# B&R Automation Studio project TD52 (part 84)

### Modul_EngCtr.typ - Package data types
```iecst
(********************************************************************
 * COPYRIGHT -- INNIO Company
 ********************************************************************
 * Package: Opstate_Pkg
 * File: module_Opstate.typ
 * Author: Mario Graus
 * Created: October 19, 2011
 ********************************************************************
 * Data types of package Opstate_Pkg
 ********************************************************************)

TYPE
	IN_EngCtr_Struct : 	STRUCT
		iSt_OpMode : UDINT; (* engine operation mode *) (*OldName: new PV; Cycle:2; *)
		rN_Set_Norm : REAL; (* speed setpoint speed controller related to rN_Nom *) (*OldName: n_soll; Cycle:2;*)
		rN_Set_Norm_TC5 : REAL; (* speed setpoint speed controller related to rN_Nom *) (*OldName: n_soll; Cycle:5;*)
		rP_Act_Norm : REAL; (* actual power related to rP_Nom *) (* OldName: ssPowerEx ; Cycle:2; *)
		rP_Act_Norm_TC5 : REAL; (* actual power related to rP_Nom *) (* OldName: ssPowerEx ; Cycle:5; *)
		bDSyLine : BOOL; (* demand synchline *) (* OldName: M_SYL ; Cycle:2; *)
		bSynchDem : BOOL; (* synchronization demanded *) (* OldName: SynchAnf ; Cycle:2; *)
		rP_Set_Norm : REAL; (* power setpoint related to rP_Nom *) (* OldName: new PV; Cycle:2; *)
		rP_Set_Norm_TC5 : REAL; (* power setpoint related to rP_Nom *) (* OldName: new PV; Cycle:5; *)
		rNOxS_Eng_NOx_Act : REAL; (* actual NOx [ppm] *) (* OldName: usNOx ; Cycle:2; *)
		rNOxS_Eng_Act : REAL; (* actual NOx@x%O2 [mg] *) (* OldName: usNOx_mg ; Cycle:2; *)
		bKLS98_MSF : ARRAY[0..24]OF BOOL; (* knocking sensor measuring signal failure *) (* OldName: bKLS98Fault; Cycle:2; *)
		rKno_IP_Red : REAL; (* timing reduction by knocking *) (* OldName: klreg_dz; Cycle:2; *)
		rCA_Knck_Red : ARRAY[0..24]OF REAL; (* cylinder timing reduction by knocking *) (* OldName: ssKlRegdZZP; Cycle:2; *)
		iIdx_Cyl_Knck_Max : INT; (* cylinder with highest knock signal *) (* OldName: ucKlopfMxZyl; Cycle:2; *)
		rKnck_Intgr : ARRAY[0..24]OF REAL; (* integrated cylinder knock values *) (* OldName: IntKlopf; Cycle:2; *)
		rP_Act_Norm_Filt : REAL; (* actual power related to rP_Nom filtered T=1s  *) (* OldName: PN_GASART; Cycle:2; *)
		rP_Act_Norm_Filt_TC5 : REAL; (* actual power related to rP_Nom filtered T=1s  *) (* OldName: PN_GASART; Cycle:5; *)
		tAB2EC : AmmBase2MM; (* 0 *) (* OldName: new PV; Cycle:2; *)
		tAB2EC_TC5 : AmmBase2MM; (* 0 *) (* OldName: new PV; Cycle:5; *)
		bIgn_Dem : BOOL; (* demand ignition *) (* OldName: ZUEND; Cycle:5; *)
		bIgn_Run : BOOL; (* Ignition system running *) (* OldName: ZIB; Cycle:2; *)
		tOMSS_MAT : HALioDo_Type; (* operation mode selector switch - MANUAL/AUTO/TEST *) (* OldName: BWS_HA; Cycle:2; *)
		rN_IgnIC_Act : REAL; (* Engine speed measured by ignition IC *) (* OldName: ZDGSpeed; Cycle:1; *)
		rN_IgnSAFI_Act : REAL; (* Engine speed measured by ignition SAFI *) (* OldName: ZDGSpeed; Cycle:2; *)
		rT_EG_Cyl : ARRAY[0..24]OF REAL; (* cylinder exhaust gas temperatures *) (* OldName: t_zyl; Cycle:5; *)
		bEng_Dem_Bloc : BOOL; (* blocking release of engine *) (* OldName: ANFBLO; Cycle:2; *)
		tPB2MM : ParaBase2MM_type; (* Messages from parametercheck module parameter are OK *) (* OldName: new PV; Cycle:5; *)
		rP_Nom : REAL; (* nominal electric power [kW], depends on gastype *) (* OldName: PN_GASART; Cycle:2; *)
		rP_Nom_TC6 : REAL; (* nominal electric power [kW], depends on gastype *) (* OldName: PN_GASART; Cycle:6; *)
		rKno_T2s_Red : REAL; (* mixture temp. red. by knocking *) (* OldName: klreg_dt2 ; Cycle:2; *)
		iIdx_Gtyp_Dem : INT; (* actual gassort 1..4 *) (* OldName: gasart; Cycle:2; *)
		iIdx_Gtyp_Dem_TC5 : INT; (* actual gassort 1..4 *) (* OldName: gasart; Cycle:5; *)
		bGasMixingActive : BOOL; (*Gas mixing active for Tecjets *) (* OldName: 	bCrossOver	; Cyclic: ; *)
		tP_Act : ARRAY[0..2]OF HALioAi_Type; (* actual electric power [kW] *) (* OldName: P_IST_OF; Cycle:2; *)
		tSafetyLoop_Eng : HALioDi_Type; (* DI: Safety loop engine *) (* OldName: RUHE; Cycle:5; *)
		tActuator_Ok : HALioDi_Type; (* DI: Actuator okay *) (* OldName: ST_ACT; Cycle:2; *)
		tActuator_Ok_TV1A : HALioDi_Type; (* DI: Actuator okay throttle valve 1A *) (* OldName: DI_F_ACT_TV1A; Cycle:2; *)
		tActuator_Ok_TV1B : HALioDi_Type; (* DI: Actuator okay throttle valve 1B *) (* OldName: DI_F_ACT_TV1B; Cycle:2; *)
		tActuator_Ok_TV2A : HALioDi_Type; (* DI: Actuator okay throttle valve 2A *) (* OldName: DI_F_ACT_TV2A; Cycle:2; *)
		tActuator_Ok_TV2B : HALioDi_Type; (* DI: Actuator okay throttle valve 2B *) (* OldName: DI_F_ACT_TV2B; Cycle:2; *)
		tGCB_On : HALioDi_Type; (* DI generator circuit breaker closed *) (* OldName: GCB_ON ; Cycle:2; *)
		tPr_Ch_P2bFA : HALioAi_Type; (* actual charge pressure before throttle valve, before Flame Arrester*) (* OldName: P2 ; Cycle:2; *)
		tPr_Ch_P2 : HALioAi_Type; (* actual charge pressure before throttle valve *) (* OldName: P2 ; Cycle:2; *)
		tT_EG_Cyl : ARRAY[0..24]OF HALioAi_Type; (* AI cylinder exhaust gas temperatures *) (* OldName: t_zyl; Cycle:2; *)
		tActuator_Ok_CBV1 : HALioDi_Type; (* DI: Actuator okay compressor bypass valve 1 *) (* OldName: DI_F_TBV; Cycle:2; *)
		tActuator_Ok_CBV2 : HALioDi_Type; (* DI: Actuator okay compressor bypass valve 2 *) (* OldName: DI_F_TBV2; Cycle:2; *)
		tActuator_Ok_DAI_A : HALioDi_Type; (* DI: Actuator okay DAI control valve bank A M.05-YCI-104 *)
		tActuator_Ok_DAI_B : HALioDi_Type; (* DI: Actuator okay DAI control valve bank B M.05-YCI-204*)
		tGV1_Open : HALioDo_Type; (* DO: open gas valve 1 *) (* OldName: GASV1; Cycle:2; *)
		tGV2_Open : HALioDo_Type; (* DO: open gas valve 2 *) (* OldName: GASV2; Cycle:2; *)
		tT_EO : HALioAi_Type; (* AI: Engine oil temperature *) (* OldName: OTP_WE; Cycle:2; *)
		rT_Ch_T1LP_Avg : REAL; (*average charge temperature before low-pressure turbocharger (= engine intake air) [deg.C]*) (*OldName:ssIATemp,ANA_ZLTP,tT_InAirER; Cycle:5;*) (* V04.04.00.00 *)
		bAMM_T_Ch_T1LP_Avg : BOOL; (*collective warning - average charge temp. before low-pressure TC (= engine intake air)*) (* V04.04.00.00 *)
		tT_AirIn : HALioAi_Type; (* AI: intake air temperature of humidity sensor [deg.C]*) (* OldName: FEUCHTE_TEMP_WE; Cycle:2; *)
		tHumidity_AirIn : HALioAi_Type; (* AI: intake air relative humiidty of humidity sensor, normed value [0...1]*) (* OldName: FEUCHTE_WE; Cycle:2; *)
		bEng_Dem : BOOL; (* demand engine *) (*OldName:M_AGFD;Cycle:2;*)
		rN_EngAct : REAL; (* *) (* OldName: ; Cycle:2; *)
		rCA_IgnP_CylOffset : ARRAY[0..24]OF REAL; (* Cylinder individual ignition timing point OFFSET *) (* OldName: ZZP_CYL; Cycle: 5;*)
		tPos_Act_WG : HALioAi_Type; (*Wastegate single valve position*)
		tPos_Act_WG_A : HALioAi_Type; (*Wastegate A valve position*) (* OldName: AI_WasteGate_y_Ist_A; Cycle:2; *)
		tPos_Act_WG_B : HALioAi_Type; (*Wastegate B valve position*) (* OldName: AI_WasteGate_y_Ist_A; Cycle:2; *)
		tPF_Act : ARRAY[0..2]OF HALioAi_Type; (* actual cos phi value TC1*) (*ssCosPhi_TC1; Cycle:2; *)
		tI_L1 : ARRAY[0..2]OF HALioAi_Type := [3(0)]; (*Phase current generator I1 *) (*OldName:ssIL1_fast ; Cycle:2; *)
		tI_L2 : ARRAY[0..2]OF HALioAi_Type := [3(0)]; (*Phase current generator I2 *) (*OldName:ssIL2_fast ; Cycle:2; *)
		tI_L3 : ARRAY[0..2]OF HALioAi_Type := [3(0)]; (*Phase current generator I3 *) (*OldName:ssIL3_fast ; Cycle:2; *)
		tF_MMD : ARRAY[0..2]OF HALioAi_Type; (*actual generator frequence *) (* OldName:usFreq_TC1; Cycle:2; *)
		tF_MMD_BusBar : ARRAY[0..2]OF HALioAi_Type; (*frequency busbar*) (*OldName:usSynch2Frequency; Cycle:2*)
		tU_Avg : ARRAY[0..2]OF HALioAi_Type := [3(0)]; (* actual generator average voltage*) (* OldName:ssUAvg_TC1; Cycle:2; 	*)
		tI_Avg : ARRAY[0..2]OF HALioAi_Type := [3(0)]; (* actual generator average current*) (* OldName:ssIAvg_TC1; Cycle:2; 	*)
		tU_L1L2 : ARRAY[0..2]OF HALioAi_Type := [3(0)]; (*generator voltage phase 1_2 [V] *) (*OldName:ssUL1L2 ; Cycle:2; *)
		tU_L2L3 : ARRAY[0..2]OF HALioAi_Type := [3(0)]; (*generator voltage phase 2_3 [V] *) (*OldName: ssUL2L3 ; Cycle:2; *)
		tU_L3L1 : ARRAY[0..2]OF HALioAi_Type := [3(0)]; (*generator voltage phase 3_1 [V] *) (*OldName:ssUL3L1 ; Cycle:2; *)
		tU_L1N : ARRAY[0..2]OF HALioAi_Type := [3(0)]; (*generator voltage phase 1_N [V] *) (*OldName:ssUL1N ; Cycle:2; *)
		tU_L2N : ARRAY[0..2]OF HALioAi_Type := [3(0)]; (*generator voltage phase 2_N [V] *) (*OldName:ssUL2N ; Cycle:2; *)
		tU_L3N : ARRAY[0..2]OF HALioAi_Type := [3(0)]; (*generator voltage phase 3_N [V] *) (*OldName:ssUL3N ; Cycle:2; *)
		rN_IgnSAFI_LastValOK : REAL; (* last sent speed value from one of the SAFI devices *) (* OldName:n_lastValOK; Cycle:1 *)
		tT_Ch_T1HP : HALioAi_Type; (*charge temperature before high pressure TC [deg.C]*) (*OldName: new PV; Cycle:2;*)
		tPr_Ch_P1HP : HALioAi_Type; (*charge pressure p1 before high pressure TC [bar]*) (*OldName: new PV; Cycle:2;*)
		tN_TCHP : HALioAi_Type; (*high pressure turbocharger speed [rpm]*) (*OldName: new PV; Cycle:2;*)
		tN_TCLP : HALioAi_Type; (*low pressure turbocharger speed [rpm]*) (*OldName: new PV; Cycle:2;*)
		tT_EGaTC : HALioAi_Type; (*AI exhaust gas temperature after turbo charger T4 [deg.C] (M.02-TI-001)*) (*OldName:VABK_WE;Cycle:2;*)
		tT_EGbTC : HALioAi_Type; (*AI exhaust gas temperature before turbo charger T3 [deg.C]*) (*OldName:T3_WE;Cycle:2;*)
		tLam_Act : HALioAi_Type; (*actual Lambda value*) (*OldName: new PV; Cycle:2;*)
		iPassLevel : INT; (*pass level actual*) (*OldName:ucPassLevel; Cycle:5;*)
		iCnt_OpHours : DINT; (* operating hours counter *) (*OldName:betrieb_h;Cycle:2;*)
		bP_Ramp_Target_Reached : BOOL; (* ramp of power set value has reached the target value *) (*OldName:new PV;Cycle:2;*)
		tEng_Run : HALioDo_Type; (* engine running *) (*OldName:BTRB,M_BTRB;Cycle:2;*)
		tPos_Act_TV : HALioAi_Type; (* throttle valve position *) (* OldName: AI_Drkl_y_Ist; Cycle:2; *)
		tPos_Act_TV_A1 : HALioAi_Type; (* throttle valve position A1 *) (* OldName: AI_Drkl_y_Ist_A1; Cycle:2; *)
		tPos_Act_TV_A2 : HALioAi_Type; (* throttle valve position A2 *) (* OldName: AI_Drkl_y_Ist_A2; Cycle:2; *)
		tPos_Act_TV_B1 : HALioAi_Type; (* throttle valve position B1 *) (* OldName: AI_Drkl_y_Ist_B1; Cycle:2; *)
		tPos_Act_TV_B2 : HALioAi_Type; (* throttle valve position B2 *) (* OldName: AI_Drkl_y_Ist_B2; Cycle:2; *)
		tPos_Act_CBV_A1 : HALioAi_Type; (* compressor bypass valve position A1 *) (* OldName: AI_Turbo_y_Ist_A1; Cycle:2; *)
		tPos_Act_CBV_A2 : HALioAi_Type; (* compressor bypass valve position A2 *) (* OldName: AI_Turbo_y_Ist_A2; Cycle:2; *)
		tPos_Act_CBV_B1 : HALioAi_Type; (* compressor bypass valve position B1 *) (* OldName: AI_Turbo_y_Ist_B1; Cycle:2; *)
		tPos_Act_CBV_B2 : HALioAi_Type; (* compressor bypass valve position B2 *) (* OldName: AI_Turbo_y_Ist_B2; Cycle:2; *)
		rGT_QualMix_1_2_TC2 : REAL; (*Mixture ratio bet. gas 1 and 2 [%], e.g. value 0.75 =75%*) (* OldName: 	ssMisch1_2	; Cyclic:2; *)
		rGT_QualMix_1_2 : REAL; (*Mixture ratio bet. gas 1 and 2 [%], e.g. value 0.75 =75%*) (* OldName: 	ssMisch1_2	; Cyclic:5; *)
		rGT_RatioMix_TC2 : REAL; (*Gas mixture rate after ramp fub [%], e.g. 0.5 = 50%*) (* OldName: 	ssRatioMix	; Cyclic:2; *)
		rGT_RatioMix : REAL; (*Gas mixture rate after ramp fub [%], e.g. 0.5 = 50%*) (* OldName: 	ssRatioMix	; Cyclic:5; *)
		bDualTJ : BOOL; (*Gas mixing with two TecJets*) (*OldName: bDualTJ; Cycle:2; *)
		rGT_MixSet : REAL; (*Set point for gas mixture rate [0..100%], old	 ssSetMix *) (* OldName: 	ssSetMix	; Cycle:2; *)
		bAMM_Pr_AirStarter_Tank_Lo : BOOL; (* warning starter tank pressure low trigger *)
		bGasTyp1_Act : BOOL; (* gas type 1 active *) (*OldName:AN_GAS1,AW_ZZP1;Cycle:2;*)
		bGasTyp2_Act : BOOL; (* gas type 2 active *) (*OldName:AN_GAS2,AW_ZZP2;Cycle:2;*)
		bGasTyp3_Act : BOOL; (* gas type 3 active *) (*OldName:AN_GAS3,AW_ZZP3;Cycle:2;*)
		bGasTyp4_Act : BOOL; (* gas type 4 active *) (*OldName:AN_GAS4,AW_ZZP4;Cycle:2;*)
		bGasTypMix1_2_Act : BOOL; (* gas type mix 1-2 active *) (*OldName:AN_GAS1_2,AW_ZZP1_2;Cycle:2;*)
		rCA_Ign_Avg : REAL; (*Actual ignition point average*) (*OldName:ZZPAvg; Cycle:;*)
		rKnck_Intgr_Max : REAL; (* maximum integrated knock value *) (* OldName: IntKlopfMx ; Cycle: 2 *)
		tN2_ScavGV_CoOpen : HALioDo_Type; (*DO N2 Gas Valves vommand open*) (*OldName:N2_GASV;Cycle:2*)
		tTBMode : HALioDi_Type; (* DI test bench mode *) (*OldName:CIRCUITUS; Cycle:5;*)
		tGV_Rel : HALioDo_Type; (* DO: Release gas valves *) (*OldName:FG_GASV;Cycle:2;*)
		bGV_On : BOOL; (*Gas valves On*) (*OldName:M_GASV;Cycle:2;*)
		rP_Set_Unred_Norm : REAL; (* unreduzed power setpoint related to rP_Nom *) (* OldName: P_UNRED; Cycle:2; *)
		bPBCSensErr : ARRAY[0..24]OF BOOL; (* error info for PBC *) (* OldName: bPBCSensErr; Cycle:2; *)
		bPBCCompLineCheck : ARRAY[0..24]OF BOOL; (* error info for PBC *) (* OldName: bPBCCompLineCheck; Cycle:2; *)
		bPBCNegVoltCheck : ARRAY[0..24]OF BOOL; (* error info for PBC *) (* OldName: bPBCNegVoltCheck; Cycle:2; *)
		bPBCNegPresCheck : ARRAY[0..24]OF BOOL; (* error info for PBC *) (* OldName: bPBCNegPresCheck; Cycle:2; *)
		bPBCPresSlopeCheck : ARRAY[0..24]OF BOOL; (* error info for PBC *) (* OldName: bPBCPresSlopeCheck; Cycle:2; *)
		bPBCSlowDriftCheck : ARRAY[0..24]OF BOOL; (* error info for PBC *) (* OldName: bPBCSlowDriftCheck; Cycle:2; *)
		bPBCConfNotOK : ARRAY[0..12]OF BOOL; (* error info for PBC *) (* OldName: bPBCConfNotOK; Cycle:2; *)
		bPBCMemBurst : ARRAY[0..24]OF BOOL; (* error info for PBC *) (* OldName: bPBCMemBurst; Cycle:2; *)
		bPBCInvalidPar : ARRAY[0..12]OF BOOL; (* error info for PBC *) (* OldName: bPBCInvalidPar; Cycle:2; *)
		tDAI_V_Opened : HALioDi_Type; (* DAI shut off valve position opened M.05-YCS-001 *)
		tDAI_V_Opened_TC1 : HALioDi_Type; (* DAI shut off valve position opened for task cyclic 1 M.05-YCS-001 *)
		tDAI_V_Closed : HALioDi_Type; (* DAI shut off valve position closed M.05-YCS-001 *)
		tPos_DAI_Act_A : HALioAi_Type; (* AI: Position feedback DAI control valve bank A M.05-YCI-104*)
		tPos_DAI_Act_B : HALioAi_Type; (* AI: Position feedback DAI control valve bank B M.05-YCI-204*)
		tDAI_CB_On : HALioDi_Type; (* DI: DAI curcuit breaker feedback signal *)
		tMS_PBC0 : ARRAY[0..12]OF _tSAFImdatas; (* Pressure based control measuring data 0 *) (* OldName:DMR_md0; Cycle:2 *)
		tMS_PBC1 : ARRAY[0..12]OF _tSAFImdatas; (* Pressure based control measuring data 1 *) (* OldName:DMR_md1; Cycle:2 *)
		tMS_PBC2 : ARRAY[0..12]OF _tSAFImdatas; (* Pressure based control measuring data 2 *) (* OldName:DMR_md2; Cycle:2 *)
		tMS_PBC3 : ARRAY[0..12]OF _tSAFImdatas; (* Pressure based control measuring data 3 *) (* OldName:DMR_md3; Cycle:2 *)
		tMS_PBC4 : ARRAY[0..12]OF _tSAFImdatas; (* Pressure based control measuring data 4 *) (* OldName:DMR_md4; Cycle:2 *)
		tMS_PBC5 : ARRAY[0..12]OF _tSAFImdatas; (* Pressure based control measuring data 5 *) (* OldName:DMR_md5; Cycle:2 *)
		tMS_PBC6 : ARRAY[0..12]OF _tSAFImdatas; (* Pressure based control measuring data 6 *) (* OldName:DMR_md6; Cycle:2 *)
		tMS_PBC7 : ARRAY[0..12]OF _tSAFImdatas; (* Pressure based control measuring data 7 *) (* OldName:DMR_md7; Cycle:2 *)
		tMS_PBC8 : ARRAY[0..12]OF _tSAFImdatas; (* Pressure based control measuring data 8 *) (* OldName:DMR_md8; Cycle:2 *)
		tMS_PBC9 : ARRAY[0..12]OF _tSAFImdatas; (* Pressure based control measuring data 9 *) (* OldName:DMR_md9; Cycle:2 *)
		tMS_PBC10 : ARRAY[0..12]OF _tSAFImdatas; (* Pressure based control measuring data 10 *) (* OldName:DMR_md10; Cycle:2 *)
		tMS_PBC11 : ARRAY[0..12]OF _tSAFImdatas; (* Pressure based control measuring data 11 *) (* OldName:DMR_md11; Cycle:2 *)
		tMS_PBC12 : ARRAY[0..12]OF _tSAFImdatas; (* Pressure based control measuring data 12 *) (* OldName:DMR_md12; Cycle:2 *)
		tMS_PBC13 : ARRAY[0..12]OF _tSAFImdatas; (* Pressure based control measuring data 13 *) (* OldName:DMR_md13; Cycle:2 *)
		tMS_PBC14 : ARRAY[0..12]OF _tSAFImdatas; (* Pressure based control measuring data 14 *) (* OldName:DMR_md14; Cycle:2 *)
		tMS_PBC15 : ARRAY[0..12]OF _tSAFImdatas; (* Pressure based control measuring data 15 *) (* OldName:DMR_md15; Cycle:2 *)
		tMS_PBC16 : ARRAY[0..12]OF _tSAFImdatas; (* Pressure based control measuring data 16 *) (* OldName:DMR_md16; Cycle:2 *)
		tMS_PBC17 : ARRAY[0..12]OF _tSAFImdatas; (* Pressure based control measuring data 17 *) (* OldName:DMR_md17; Cycle:2 *)
		tMS_PBC18 : ARRAY[0..12]OF _tSAFImdatas; (* Pressure based control measuring data 18 *) (* OldName:DMR_md18; Cycle:2 *)
		tMS_PBC19 : ARRAY[0..12]OF _tSAFImdatas; (* Pressure based control measuring data 19 *) (* OldName:DMR_md19; Cycle:2 *)
		tMS_PBC20 : ARRAY[0..12]OF _tSAFImdatasExtend; (* Pressure based control measuring data 20*) (* OldName:DMR_md19; Cycle:2 *)
		tMS_PBC21 : ARRAY[0..12]OF _tSAFImdatasExtend; (* Pressure based control measuring data 21*) (* OldName:DMR_md19; Cycle:2 *)
		tT_GR : HALioAi_Type; (* gas rail temperature *) (* OldName: AI_GRTP; Cycle:2; *)
		tMCB_On : HALioDi_Type; (* DI mains circuit breaker closed *) (*OldName:DI_MCB_ON; Cycle:2;*)
		bScavFinished_TC2 : BOOL; (* scavenging cycle finished  *) (*OldName:SPUEL_AB;Cycle:2;*)
		bScavFinished : BOOL; (* scavenging cycle finished  *) (*OldName:SPUEL_AB;Cycle:5;*)
		iIdx_RSS : INT; (*Index of request selector switch - 0..OFF, 1..ON, 2..REMOTE*)
		iIdx_OMSS : INT; (* inex of operation mode selector switch - 0..OFF, 1..MAN, 2..AUTO, 3..TEST, 4..SCAVENGING *) (*OldName:new PV;Cycle:2;*)
		tT_DAI : HALioAi_Type; (* Air temperature before DAI shut off valve [deg.C] M.05-TI-003*)
		tT_EO_Preheating : HALioAi_Type; (*AI: Oil temperature preheating *) (*OldName: OIL_temp_preheating, AI_M_03_TI_078; Cycle:2*)
		tT_ECW : HALioAi_Type; (* cooling water temperature *) (*OldName:ANA.KWT;Cycle:2;*)
		tT_Ch_T1HP_A : HALioAi_Type; (*charge temperature before high pressure TC A [deg.C]*) (*OldName: ; Cycle: 2;*)
		tT_Ch_T1HP_B : HALioAi_Type; (*charge temperature before high pressure TC B [deg.C]*) (*OldName: ; Cycle: 2;*)
		tPr_Ch_P1HP_A : HALioAi_Type; (*charge pressure p1 before high pressure TC A [bar]*) (*OldName: ; Cycle: 2;*)
		tPr_Ch_P1HP_B : HALioAi_Type; (*charge pressure p1 before high pressure TC B [bar]*) (*OldName: ; Cycle: 2;*)
		tPr_DAI_A : HALioAi_Type; (* Pressure before DAI control valve bank A [bar] M.05-PI-101 *)
		tPr_DAI_B : HALioAi_Type; (* Pressure before DAI control valve bank B [bar] M.05-PI-201 *)
		tPr_DAI_In : HALioAi_Type; (* Pressure before DAI shut off valve [bar] M.05-PI-002 *)
		tPr_EGbHPTC_A : HALioAi_Type; (* AI: Exhaust gas pressure before high-pressure turbocharger A (M.02-PI-152) *) (* OldName: AI_M_02_PI_152	; Cyclic: 2; *)
		tPr_EGbHPTC_B : HALioAi_Type; (* AI: Exhaust gas pressure before high-pressure turbocharger B (M.02-PI-252) *) (* OldName: AI_M_02_PI_252	; Cyclic: 2; *)
		tPr_EGaHPTC_A : HALioAi_Type; (* AI: Exhaust gas pressure after high-pressure turbocharger A  (M.02-PI-153) *) (* OldName: AI_M_02_PI_153	; Cyclic: 2; *)
		tPr_EGaHPTC_B : HALioAi_Type; (* AI: Exhaust gas pressure after high-pressure turbocharger B  (M.02-PI-253) *) (* OldName: AI_M_02_PI_253	; Cyclic: 2; *)
		tPr_EGaLPTC_A : HALioAi_Type; (* AI: Exhaust gas pressure after low-pressure turbocharger A  (M.02-PI-154) *) (* OldName: AI_M_02_PI_154	; Cyclic: 2; *)
		tPr_EGaLPTC_B : HALioAi_Type; (* AI: Exhaust gas pressure after low-pressure turbocharger B  (M.02-PI-254) *) (* OldName: AI_M_02_PI_254	; Cyclic: 2; *)
		tT_EGbHPTC_A : HALioAi_Type; (* AI: Exhaust gas temperature before high-pressure turbocharger A  (M.02-TI-166) *) (* OldName: AI_M_02_TI_166	; Cyclic: 2; *)
		tT_EGbHPTC_B : HALioAi_Type; (* AI: Exhaust gas temperature before high-pressure turbocharger B  (M.02-TI-266) *) (* OldName: AI_M_02_TI_266	; Cyclic: 2; *)
		tT_EGaHPTC_A : HALioAi_Type; (* AI: Exhaust gas temperatur after high-pressure turbocharger A  (M.02-TI-167) *) (* OldName: AI_M_02_TI_167	; Cyclic: 2; *)
		tT_EGaHPTC_B : HALioAi_Type; (* AI: Exhaust gas temperatur after high-pressure turbocharger A  (M.02-TI-267) *) (* OldName: AI_M_02_TI_267	; Cyclic: 2; *)
		tN_TCHP_A : HALioAi_Type; (*high pressure turbocharger speed A [rpm]*) (*OldName: ssTurboSpdA_WE, TRB1_WE, ssTurboSpdA; Cycle: 2;*)
		tN_TCHP_B : HALioAi_Type; (*high pressure turbocharger speed B [rpm]*) (*OldName: ssTurboSpdB_WE, TRB2_WE, ssTurboSpdB; Cycle: 2;*)
		tN_TCLP_A : HALioAi_Type; (*low pressure turbocharger speed A [rpm]*) (*OldName: ssTurboSpd_LP_A_WE, AI_TurboSpd_LP_A, ssTurboSpd_LP_A; Cycle: 2;*)
		tN_TCLP_B : HALioAi_Type; (*low pressure turbocharger speed B [rpm]*) (*OldName: ssTurboSpd_LP_B_WE, AI_TurboSpd_LP_B, ssTurboSpd_LP_B; Cycle: 2;*)
		tF_MMD_Synch2 : ARRAY[0..2]OF HALioAi_Type; (* *) (*OldName:usSynch2Frequency;Cycle:2;*)
		rP_Ramp_IncGrad_All_Norm : REAL; (*gradient for increase of power ramp in grid mode [1/s]*) (*OldName:t_upALL; Cycle:2;*)
		rP_Set_GEN2_Norm : REAL; (* power setpoint for GEN2 *) (*OldName:ssSetpointPowerkW_BDC; Cycle:2;*)
		tFastStartReq : HALioDi_Type; (* DI: Fast Start Required *) (* OldName: DI_FastStartReq; Cycle:2; *)
		tVeryFastStartReq : HALioDi_Type; (* DI: Fast Start Required *) (* OldName: DI_FastStartReq; Cycle:2; *)
		rCA_PI_Dur_COffset : ARRAY[0..24]OF REAL; (* custom PI duration offset *) (* OldName: ssTestBenchOffset; Cycle:2; *)
		tT_EO_Pan : HALioAi_Type; (*engine oil temperature oil pan, M.03-TI-002*) (*OldName:AI_t_OilPan; Cycle:2*)
		rT_Ch_T2s_Avg : REAL; (*filtered 1s Average charge temperature t2' [deg.C]*) (* OldName: new PV ; Cycle: 2 *)
		rT_Ch_T2s_A : REAL; (*filtered 1s charge temperature t2' bank A [deg.C]*) (* OldName: new PV ; Cycle: 2 *)
		rT_Ch_T2s_B : REAL; (*filtered 1s charge temperature t2' bank B [deg.C]*) (* OldName: new PV ; Cycle: 2 *)
		rPr_Ch_P2s_Avg : REAL; (*filtered 1s Average charge pressure p2' [bar]*) (* OldName: new PV ; Cycle: 2 *)
		rPr_Ch_P2s_A : REAL; (*filtered 1s charge pressure p2' bank A [bar]*) (* OldName: new PV ; Cycle: 2 *)
		rPr_Ch_P2s_B : REAL; (*filtered 1s charge pressure p2' bank B [bar]*) (* OldName: new PV ; Cycle: 2 *)
		rPr_Ch_P2s_Avg_UF : REAL; (*unfiltered Average charge pressure p2' [bar]*) (* OldName: new PV ; Cycle: 2 *)
		rPr_Ch_P2s_A_UF : REAL; (*unfiltered Average charge pressure p2' bank A [bar]*) (* OldName: new PV ; Cycle: 2 *)
		rPr_Ch_P2s_B_UF : REAL; (*unfiltered Average charge pressure p2' bank B [bar]*) (* OldName: new PV ; Cycle: 2 *)
		rPr_GR_UF : REAL; (*unfiltered Average gas rail pressure [bar]*) (* OldName: new PV ; Cycle: 2 *)
		rT_Ch_T2s_Avg_UF : REAL; (*unfiltered Average charge temperature t2' [deg.C]*) (* OldName: new PV ; Cycle: 2 *)
		tActuator_Ok_CBV_A : HALioDi_Type; (* DI: Actuator okay compressor by pass valve 1A *) (* OldName: DI_F_ACT_TBV_A; Cycle:2; *)
		tActuator_Ok_CBV_B : HALioDi_Type; (* DI: Actuator okay compressor by pass valve 1B *) (* OldName: DI_F_ACT_TBV_B; Cycle:2; *)
		bDeflagrationPrct : BOOL; (*Deflagration protection*) (* OldName: 	PUFF	; Cyclic: 2; *)
		tPr_Ch_P2s : HALioAi_Type; (*charge pressure p2' after throttle valve [bar]*) (*OldName: AI_PressP2_TC1, ssPressP2WE, pl_ist, LDRIST, ANA.LDRIST; Cycle: 1;*)
		tPr_Ch_P2s_A : HALioAi_Type; (*charge pressure p2' after throttle valve A [bar]*) (*OldName: AI_PressP2s_A_TC1, AIPressP2s_A, ssPressP2s_A, rPressP2s_A; Cycle: 1;*)
		tPr_Ch_P2s_B : HALioAi_Type; (*charge pressure p2' after throttle valve B [bar]*) (*OldName: AI_PressP2s_B_TC1, AIPressP2s_B, ssPressP2s_B, rPressP2s_B; Cycle: 1;*)
		tPr_GR_II : HALioAi_Type; (*AI Gas Pressure in Gas Rail number 2 [bar]*) (* OldName: AIPressGasRail2_TC1; Cyclic: 1; *)
		tPr_GR_I : HALioAi_Type; (*AI Gas Pressure in Gas Rail number 1 [bar] *) (* OldName: AIPressGasRail	; Cyclic: 1; *)
		tActuator_Ok_WG : HALioDi_Type; (* DI: Actuator okay wastegate valve*)
		tActuator_Ok_WG_A : HALioDi_Type; (* DI: Actuator okay wastegate valve A *) (* OldName: DI_F_ACT_EGBV_A; Cycle:2; *)
		tActuator_Ok_WG_B : HALioDi_Type; (* DI: Actuator okay wastegate valve B *) (* OldName: DI_F_ACT_EGBV_B; Cycle:2; *)
		rPr_Knck_Filt : ARRAY[0..24]OF REAL; (* filtred knock signal with containment V2*) (* OldName: knockFilt; Cycle 2;*)
		bMMD_GenAlarmTestOn : BOOL; (*MMD_Gen alarm test On*) (*OldName:newPv; Cycle:2;*)
		tPr_CC : HALioAi_Type; (* AI pressure crank case [bar] *) (*OldName:AI_KGD; Cycle:5*)
		rGMU_Pos_Valve_Prom : ARRAY[0..4]OF REAL; (*Valve Position [%]*) (*OldName: ssTJPos; Cycle: 5*)
		iState_RKS : ARRAY[0..24]OF USINT; (* state for every cylinder, 1 = PBC, 2 = RKS, 3= FTC *) (* OldName: 0; Cycle:2; *)
		rPr_P2s_Knck_Offs : REAL; (* Offset for charge pressure due Knock *) (* OldName: 0; Cycle:2; *)
		rPmax_Knck_Red : ARRAY[0..24]OF REAL; (* cylinder PI duration reduction by knocking *) (* OldName: 0 ; Cycle: 2 *)
		bFastPowRed : BOOL; (* fast power reduction, due knock or glowign *) (*OldName:newPV; Cycle:2;*)
		rPr_Baro_Internal : REAL; (*Internal value for barometric pressure [bar (abs)]*)
		tT_EGaLPTC_A : HALioAi_Type; (*exhaust gas temperature after low pressure turbo charger A (M.02-TI-168)*) (*OldName:t_EGaLPTC_A;Cycle:5*)
		tT_EGaLPTC_A_TC2 : HALioAi_Type; (*exhaust gas temperature after low pressure turbo charger A (M.02-TI-168)*) (*OldName:t_EGaLPTC_A;Cycle:5*)
		tT_EGaLPTC_B : HALioAi_Type; (*exhaust gas temperature after low pressure turbo charger B (M.02-TI-268)*) (*OldName:t_EGaLPTC_B;Cycle:5*)
		tT_EGaLPTC_B_TC2 : HALioAi_Type; (*exhaust gas temperature after low pressure turbo charger B (M.02-TI-268)*) (*OldName:t_EGaLPTC_B;Cycle:5*)
		bT_ECW_RelLoad : BOOL; (*temperature engine cooling water release load*)
		szEng_Motorversion : STRING[17]; (*Engine version *) (*V04.04.00.00*)
		rPr_Leanox_ManSet_Cust : REAL; (*LINK POINT for Jenbacher Technologx Testbench*)
		rLam_Eng_LL_ManSet_Cust : REAL; (*LINK POINT for Jenbacher Technologx Testbench*)
		bLeanox_Man_Cust : BOOL; (*LINK POINT for Jenbacher Technologx Testbench*)
		bPreL_FS_EngStaRel : BOOL; (*prelubrication engine fast start release*)
		rP2s_red_1 : REAL; (*power reduction boost pressure of the limited power of nominal power  *)
		bPreL_FS_Act : BOOL; (*prelubrication engine fast start activated*)
		rAng_MMD_Diff : ARRAY[0..2]OF REAL;
		iIdx_SyOMSS : INT; (* synchronization operating mode selection *) (*OldName:new PV;Cycle:5;*)
		bSimWinMOD_Active : BOOL; (* WinMode simulation active *) (* OldName:new PV; Cycle:5*)
		bSimWinMOD_FastStart : BOOL; (* WinMode fast start of engine*) (* OldName:new PV; Cycle:5*)
		bAMM_Pr_Baro_Internal : BOOL; (*TRUE= don't use IN_EC.rPr_Baro_Internal*) (*V04.05.00.00*)
		bUseCtrCust2_4HumidityCtr : BOOL; (*! new V4.5 2017 !  Option to use CtrCust2 as LLTP controller with humidity function *)
		rCtr_Cust2_W_set : REAL; (*! new V4.5 2017 !  Setpoint Ctr Cust 2 for Japan Option for humidity function *)
		rGMU_Pr_DiffGas : ARRAY[0..4]OF REAL; (*Differential Pressure over device [mbar*10]*)
		bPRamp_GrC_SetErr : BOOL; (* Slow increase power ramp after mains failure active *)
		bFastStartReq_Bus : BOOL; (* TRUE = Command: get ready for fast start *)
		bVeryFastStartReq_Bus : BOOL; (* TRUE = Command: get ready for very fast start *)
		bGT1_SafeDevOK : BOOL; (* release from Gas train 1 *)
		bGT2_SafeDevOK : BOOL; (* release from Gas train 2 *)
		bPCGT_SafeDevOK : BOOL; (* release from prechamber gas train *)
		rP_Ramp_DecGrad_All_Norm : REAL; (*gradient for decrease of power ramp in grid mode [1/s]*)
		bEng_Bloc : BOOL; (* blocking engine *) (*OldName:M_BLOCK;Cycle:2;*)
		bGEN2_UseFastRamp : BOOL; (*Force GEN2 to a faster decreasing Ramp*)
		bServiceMode : BOOL; (*service mode*) (*OldName:bServiceBegin; Cycle:2;*)
		bMainsReturn : BOOL; (* mains return *) (*OldName:NWK; Cycle:5*)
		bT_EOP_RelFS : BOOL; (*Oil temperature release fast start*)
		tPr_Ch_P2HP : HALioAi_Type; (*charge pressure after high-pressure turbocharger [bar] (E.08-PI-004)*)
		tMnsOk : HALioDi_Type; (*DI mains ok	*) (*OldName:DI_MNS_OK;Cycle:2*)
		rU_Ign_Max : REAL; (* Maximum Ignition voltage *) (*OldName:AvgVolt; Cycle:;*)
		tT_SCR_CatOut : HALioAi_Type; (*SCR exhaust temperature CAT outlet [deg.C] (P.02-TI-102) (fix prefix data type, changes by HeKo)*) (*OldName: tT_SCR_Out; Cycle: 5;*) (*V04.05.00.00*)
		rNOx_NOxS_EngOut_Avg : REAL; (*NOx sensor at engine outlet average - actual NOx value [ppm]*) (*OldName: newPV; Cycle: 5*)
		bAMM_NOx_NOxS_EngOut_Avg : BOOL; (*NOx feedback signal fault check*)
		rNOx_Em_CatOut_Set : REAL; (*NOx emissions at CAT outlet - setpoint [ppm]*) (*OldName: new PV; Cycle:5*) (*V04.07.00.00*)
		rNOx_Em_EngOut_Set : REAL; (*NOx Setpoint [ppm]*)
		rNOx_NOxS_CatOut_cor : REAL; (*NOx sensor at catalyst outlet - actual NOx value with offset and CEMS correction [ppm]*) (*OldName: new PV; Cycle:5*) (*V04.05.01.00*)
		tFlow_SCR_UreaDosingOut : HALioAi_Type; (*SCR Urea flow rate after dosing [l/h] (P.29-FI-001)*) (*OldName: tFlow_Urea; Cycle: 5;*) (*V04.05.00.00*)
		bSCR_NH3SlipDetected : BOOL; (*NH3 slip out of SCR catalyst detected if = TRUE (-)*)
		bRel_SCR_UDC : BOOL := FALSE; (*SCR Release urea dosing controller (UDC)*) (*V04.05.00.00*)
		rIntSignal : REAL; (*Knockintegrator level KLS90*)
		bRelSy_Customized : BOOL; (*Freigabe Syncronisierungl vo Customized Modul*)
		bGEN2_UsePowtraj_LFSM : BOOL; (*Force GEN2 to faster reaction time in case of FSM/LFSM*)
		tGCB_RT : HALioDo_Type; (* generator circuit breaker release trip  *) (*OldName:DO_GCB_RT; Cycle:5;*)
		bTExh_Mon_UseNarrowWindow : ARRAY[0..24]OF BOOL; (*use narrow threshold for exh temp mon*)
		bSA_VCD_Active : BOOL; (*Enable visualization of VCD parameters for legacy versions*)
		bPBCCPSSat : ARRAY[0..24]OF BOOL; (* Cylinder pressure sensor saturation flag for cyl X *) (* new PV; Cycle: 2*)
		rU_Ign_Max_LimHi : REAL; (* Maximum ignition voltage high limit *)
		tGCB_OGP : HALioDi_Type; (* DI: other generators parallel*)
		bMMD_BB_AlarmTestOn : BOOL; (*MMD_BB  alarm test On*) (*OldName:newPv; Cycle:2;*)
		rU_Ign_Cyl : ARRAY[0..24]OF REAL; (*Ignition voltage for each cylinder*)
		tT_SCR_CatIn_TC2 : HALioAi_Type; (*SCR Exhaust temperature CAT inlet TC2 [degC] (P.02-TI-101)*) (*OldName: new PV; Cycle:5*) (*V04.10.00.00*)
		tT_SCR_CatOut_TC2 : HALioAi_Type; (*SCR Exhaust temperature CAT outlet TC2 [degC] (P.02-TI-102)*) (*OldName: new PV; Cycle:5*) (*V04.10.00.00*)
		tT_EGaCat : HALioAi_Type; (*OXIcat outlet temperature sensor [degC] (P.02-TI-047)*)
		tT_EGbCat : HALioAi_Type; (*OXIcat inlet temperature sensor [degC] (P.02-TI-046)*)
		b_FilterScav_Active : BOOL; (* Activation signal of FGQC from customer *)
		bNoExtendedPrelube : BOOL; (*Extended prelubrication (allows 5min start)*)
		rN_TCHP_HiHi : REAL; (*Interpolated high-pressure turbocharger speed maximum - trip [rpm]*)
		rN_TCLP_HiHi : REAL; (*Interpolated low-pressure turbocharger speed maximum - trip [rpm]*)
		iSource_F_N_OffsSet : INT; (* F/N Setpoint: 0= no setpoint, 1= Droop, 2= External, 3= LSL *)
		rPr_P2s_demand_PCGT : REAL; (* Boost pressure demand for power reduction PCGT [bar(abs)] *)
		rIHR : ARRAY[0..24]OF REAL; (*Integrated heat release [kJ/m2]*)
		bThR_Active : BOOL; (* Thermal reactor active *)
		tThR_Contactor : HALioDo_Type; (* Thermal reactor - Heat transfer from engine status *)
		bThR_RelGas_Tmin : BOOL; (* Thermal reactor - minimum temperature for aux. gas injection reached *)
		bSA_PBCFrozenAltern : ARRAY[0..24]OF BOOL; (*DMR knock signal or IMEP frozen or alternating*)
		iT_EG_CylFault : ARRAY[0..24]OF UINT; (*0 = No fault / bit0 = SAFI re-para active / bit1 = Exhaust gas temperature signal frozen or alternating*) (* new PV; Cycle: 5*)
		iAggrekoEngineVersion : INT; (* engine Version for Agrekko calibration 1 = B, 2 = C, 3 = E *)
		iAggrekoTCConfig : INT; (* engine TA configuration for Agrekko calibration 1 = TA40, 2 = TA45, 3 = TA65, 4 = TA70 *)
		rH2 : REAL; (* Hydrogen concentration volumetric *)
		rH2_Comp : REAL; (* Hydrogen concentration volumetric for H2 compensation function *)
		rHum_GasIn_Abs : REAL; (* absolute humidity gas via customer BUS [g H2O/kg dry gas] *)
		tU_Set_Norm : HALioAo_Type; (* voltage output for island mode [%Unom] *)
		tQ_Act : ARRAY[0..2]OF HALioAi_Type; (*actual reactive power [kVar] *)
		tU_Gen_Exc : HALioAi_Type; (*actual excitation voltage signal, filtered and scaled*)
		bMsg9318_Set : BOOL; (* W9318 cylinder pressure sensor saturation is set *)
		bFS_Rdy_STT_StPurge : BOOL; (*purge state and starter temperature readiness for fast start*)
		iMissfCyl_PurgeCrk : UDINT; (*skip fire order for all cylinders while purging*)
		bEleStarter_Dem_PurgeCrkCylFS : BOOL; (*starter demand during purge cranking cycle for FS preparation*)
		iCAN_WG_us_ident : UDINT; (*CAN WG interface user identifier*)
	END_STRUCT;
	OUT_EngCtr_Struct : 	STRUCT
		tEC2AB : MM2AmmBase; (* 0 *) (* OldName: new PV; Cycle:   *)
		bMisfSend : BOOL; (* TRUE =send misfire CAN message *) (* OldName: 0; Cycle:2; *)
		rP_Red_Misf_Norm : REAL; (* power reduction by misfire *) (* OldName: 0; Cycle:2; *)
		rP_Red_EGT_Norm : REAL; (* power reduction by exhaust gas temp. *) (* OldName: abgas_dp; Cycle:2; *)
		rPos_TV : REAL; (* throttle valve position *) (* OldName: drkl_y; Cycle:2; *)
		rPos_CBV : REAL; (* compressor bypass valve position *) (* OldName: turbo_y; Cycle:2; *)
		bMisfCOn : BOOL; (* Misfire Command On *) (* OldName: 0; Cycle:2; *)
		rRatioMix : REAL; (* gas mixture rate after ramp fub *) (* OldName: 0; Cycle:2; *)
		ulGasFlowN : ARRAY[0..4]OF UDINT; (* setpoint gasflow one gas inject valve *) (* OldName: ulGasFlowN; Cycle:2; *)
		bLeanox_Man : BOOL; (* TRUE = leanox controller in manual *) (* OldName: l_einst_a ; Cycle:2; *)
		rPos_GM_Set_Norm : REAL; (* set point for the gasmixer *) (* OldName: ssPosGasmixerNominal; Cycle:2; *)
		rLam_Eng_LL_Set : REAL; (* Leanox Lambda set point *) (* OldName: ssPosGasmixerNominal; Cycle:2; *)
		rPos_Eng_Gm_Stepper_Set : REAL; (* rated gasmixer position *) (* OldName: usStepperRatedPos ; Cycle:2; *)
		rCA_IgnP_Set : REAL; (* ignitoin timing set point *) (* OldName: W_ZZP ; Cycle:2; *)
		bIP_Red_Reset : BOOL; (* reset of the  ignitoin timing set point reduction *) (* OldName: bResetTimingRed ; Cycle:2; *)
		bSCO_Active : BOOL; (* safety cut out gas valves glow ignition prevention *) (* OldName: SICH_SCHL; Cycle:5; *)
		rT_EPU_EG : ARRAY[0..24]OF REAL; (* engine power unit exhaust gas temperatures *) (* OldName: t_zyl; Cycle:2; *)
		rP_Red_Leanox_Norm : REAL; (* power reduction by leanox *) (* OldName: leanox_dp; Cycle:2; *)
		bLeanox_Active : BOOL; (* TRUE = leanox controller is active *) (* OldName: bLeanoxActive; Cycle:2; *)
		tEC2PB : MM2ParaBase_type; (* Data exchange structure to ParaBase *) (* OldName: new PV; Cycle:5; *)
		tPIopenH : ARRAY[0..12]OF tPIopen; (* PI open point and open duration for high cylinder *) (* OldName: SAFI.tPI.tPIopenH; Cycle:2; *)
		tPIopenL : ARRAY[0..12]OF tPIopen; (* PI open point and open duration for low cylinder *) (* OldName: SAFI.tPI.tPIopenL; Cycle:2; *)
		iMisfCyl : UDINT; (* cylinder misfire parameter *) (* OldName: MissfCyl; Cycle:1; *)
		bMsg3583 : BOOL; (* Warning: Cylinder exhaust gas temperature absolute value high  *) (* OldName: new PV; Cycle:2; *)
		bMsg3584 : BOOL; (*  Warning: Cylinder exhaust gas temperature deviation from average value *) (* OldName: new PV; Cycle:2; *)
		bSCO_Rel_GV1 : BOOL; (* TRUE = Release for gas valve 1 by glow ignition prevention (safety cut out) *) (* OldName: M_GASV1_1; Cycle:2; *)
		bSCO_Rel_GV2 : BOOL; (* TRUE = Release for gas valve 2 by glow ignition prevention (safety cut out) *) (* OldName: M_GASV1_2; Cycle:2; *)
		rT_ChC_Ctr_Wex : REAL; (* temperature charge cooler controler external setpoint *) (* OldName: Wex_GEMREG; Cycle:5; *)
		rCA_Ign_Act : ARRAY[0..24]OF REAL; (*  actual cylinder ignition point  *) (* OldName: ActTiming / ZZPCyl; Cycle:2; *)
		rT_EG_Min : REAL; (* cylinder temperature minimal value [deg.C] *) (* OldName: 0; Cycle:5; *)
		rT_EG_Avg : REAL; (* cylinder temperature average [deg.C] *) (* OldName: 0; Cycle:5; *)
		rT_EG_Max : REAL; (* cylinder temperature maximal value [deg.C] *) (* OldName: 0; Cycle:5; *)
		iNum_Msg3238 : INT; (* Cylinder information for the message 3238 *) (* OldName: new PV; Cycle:5; *)
		iNum_Msg3239 : INT; (* Cylinder information for the message 3239 *) (* OldName: new PV; Cycle:5; *)
		iNum_Msg3285 : INT; (* Cylinder information for the message 3285 *) (* OldName: new PV; Cycle:5; *)
		iNum_Msg3295 : INT; (* Cylinder information for the message 3295 *) (* OldName: new PV; Cycle:5; *)
		tActuator_Rel : HALioDo_Type; (* DO: Actuator release command *) (* OldName: ACTUATOR; Cycle:2; *)
		tActuator2_Rel : HALioDo_Type; (* DO: Actuator release command *) (* OldName: ACTUATOR2; Cycle:2; *)
		tPos_TV : HALioAo_Type; (* throttle valve position *) (* OldName: drkl_y; Cycle:2; *)
		tPos_TV_A1 : HALioAo_Type; (* throttle valve position A1 *) (* OldName: ssDrkl_y_Soll_A1; Cycle:2; *)
		tPos_TV_A2 : HALioAo_Type; (* throttle valve position A2 *) (* OldName: ssDrkl_y_Soll_A2; Cycle:2; *)
		tPos_TV_B1 : HALioAo_Type; (* throttle valve position B1 *) (* OldName: ssDrkl_y_Soll_B1; Cycle:2; *)
		tPos_TV_B2 : HALioAo_Type; (* throttle valve position B2 *) (* OldName: ssDrkl_y_Soll_B2; Cycle:2; *)
		tPos_CBV : HALioAo_Type; (* compressor bypass valve position *) (* OldName: turbo_y; Cycle:2; *)
		tPos_CBV34 : HALioAo_Type; (* compressor bypass valve position *) (* OldName: turbo_y; Cycle:2; *)
		tPos_CBV_A1 : HALioAo_Type; (* compressor bypass valve position A1 *) (* OldName: ssTurbo_y_Soll_A1; Cycle:2; *)
		tPos_CBV_A2 : HALioAo_Type; (* compressor bypass valve position A2 *) (* OldName: ssTurbo_y_Soll_A2; Cycle:2; *)
		tPos_CBV_B1 : HALioAo_Type; (* compressor bypass valve position B1 *) (* OldName: ssTurbo_y_Soll_B1; Cycle:2; *)
		tPos_CBV_B2 : HALioAo_Type; (* compressor bypass valve position B2 *) (* OldName: ssTurbo_y_Soll_B2; Cycle:2; *)
		rP_Red_HiCtr_Norm : REAL; (* power reduction by high level controller related to rP_Nom  *) (* OldName: new PV; Cycle:5; *)
		rP_Red_Hum_Norm : REAL; (* power redutcion by humidity related to rP_Nom  *) (* OldName: new PV; Cycle:5; *)
		rP_Red_PBC_Norm : REAL; (* power redutcion by PBC related to rP_Nom  *) (* OldName: ssPowerRedDMR; Cycle:2; *)
		ulMonGasFlow : ARRAY[0..4]OF UDINT; (* minimum flow for monitoring *) (* OldName: ulMonGasFlow; Cycle: 2 *)
		mp_a : ARRAY[0..4]OF _tMeasurePoint; (* leanox line meassure point 1 *) (* OldName: mp_a; Cycle: 2 *)
		rPos_Set_WG_Norm : REAL; (* normed position setpoint for wastegate *) (* OldName: ssPos_WG; Cycle: 2 *)
		tWG_Dem : HALioDo_Type; (* waste gate position *)
		tWG_A_Dem : HALioDo_Type; (* waste gate position A *) (* OldName: DO_Act_WG1; Cycle:2; *)
		tWG_B_Dem : HALioDo_Type; (* waste gate position B *) (* OldName: DO_Act_WG2; Cycle:2; *)
		tPos_Set_WG : HALioAo_Type; (* waste gate valve position A *)
		tPos_Set_WG_A : HALioAo_Type; (* waste gate valve position A *) (* OldName: ssPos_WG; Cycle:2; *)
		tPos_Set_WG_B : HALioAo_Type; (* waste gate valve position B *) (* OldName: ssPos_WG; Cycle:2; *)
		r_PhaseAng : REAL := 0.0; (*mechanical phase angle in degree*) (*OldName: fPhaseAngle;*)
		bGrC_Event : BOOL; (* Grid Code Event*) (*OldName: bGridCodeEvent;*)
		rLam_EKF_Est : REAL; (* estimated lambda from ekf *)
		tGrC_DCon : HALioDo_Type; (* DO: FALSE = Disconnect from Grid due to GridCode Event*) (* OldName: bDO_GRIDCODE_DCON_TC1; Cycle:2; *)
		rP_Red_Knck_Opti_Norm : REAL; (* power redutcion by  timing point optimizing related to rP_Nom  *) (* OldName: klreg_opti_dp; Cycle:2; *)
		bMsg3586 : BOOL; (*Warning: Mains failure maintenance request *)
		bGrC_HBErr_AUS : BOOL := FALSE; (*TRUE = Stoerung HB A1129 deaktiviert ueber GCEvent*) (*OldName: bGC_HBErr_AUS;*)
		bSG_FPR : BOOL; (* Special Gas: Fast Power Reduction *) (* OldName: bPredMessage; Cycle:2; *)
		rP_Red_SG_Norm_Pred : REAL; (* power reduction by glow ignition max number exceeded*)
		rP_Red_SG_Norm_FPR : REAL; (* power reduction by glow ignition*)
		bSG_Eng_Block_EGT : BOOL; (* W3529 - Blockierung für x[min] nach 30min Betrieb (Sondergas) *) (* OldName: bBLOCK_ABGTEMP; Cycle:2; *)
		bFastStart : BOOL; (*Engine stopped and ready for fast start*) (* OldName: bFastStart; Cycle:5; *)
		bBDC_Emergency_OFF : BOOL; (* Trip: BDC emergency OFF*) (* OldName: bBDC_Emergency_OFF; Cycle:2; *)
		rP_GEN2_Norm : REAL; (* normed power trajectory from Gen2 controller *) (* Oldname: P_d; Cycle: *)
		iIdx_ContGen : INT; (*Controller generation 1=Standard / 2=NTI *) (* Oldname: ucContGen; Cycle: *)
		ti_MisfShutDown : TIME; (* Engine is shuting down in X second because of misfire*) (* Oldname: new PV; Cycle: 2 *)
		bGen2_Act : BOOL; (* TRUE = Gen2 Controller active*) (* Oldname: BDC_ON; Cycle: 2 *)
		bTrip_IPC_MSF : BOOL; (* Trip: A2214 Cylinder pressure sensor measuring signal failure Prio2*) (* OldName: bAKnockSigErr_DMR; Cycle:2; *)
		bIPC_MSF : ARRAY[0..24]OF BOOL; (* in-cylinder pressure sensor measuring signal failure *) (* OldName: bDMRFault; Cycle: 2 *)
		rPr_CPP : ARRAY[0..24]OF REAL; (* cylinder peak pressure *) (* OldName: DruckMax; Cycle: 2 *)
		rPr_49bfTDC : ARRAY[0..24]OF REAL; (* cylinder pressure 49deg. before TDC *) (* OldName: rP_49bfTDC; Cycle: 2 *)
		rPr_49afTDC : ARRAY[0..24]OF REAL; (* cylinder pressure 49deg. after TDC *) (* OldName: rP_49afTDC; Cycle: 2 *)
		rPr_Knck : ARRAY[0..24]OF REAL; (* knock pressure *) (* OldName: Klopfen; Cycle: 2 *)
		rPr_IMEP : ARRAY[0..24]OF REAL; (* Indicated Mean Effective Pressure *) (* OldName: IndiMitDr; Cycle: 2 *)
		rCA_MFBvar : ARRAY[0..24]OF REAL; (* 50% of fuel mass burned *) (* OldName: UmsatzpunktL; Cycle: 2 *)
		rCA_PI_Dur : ARRAY[0..24]OF REAL; (* PI duration *) (* OldName: new PV ; Cycle: 2 *)
		bGlowIgn : ARRAY[0..24]OF BOOL; (* glow ignition *) (* OldName: Gluehzuend; Cycle: 2 *)
		bMisf_I : ARRAY[0..24]OF BOOL; (* missfire detection 10deg. after TDC *) (* OldName: Aussetzer; Cycle: 2 *)
		bMisf_II : ARRAY[0..24]OF BOOL; (* missfire detection 40deg. after TDC *) (* OldName: Misf_II; Cycle: 2 *)
		rPr_Leanox_Set : REAL; (* Setpoint boost pressure *) (* Oldname: pl_soll; Cycle: 2*)
		bEng_Bloc_EC : BOOL; (* blocking engine from EC Modul *) (*OldName: new PV;Cycle:2;*)
		bLimpHomeCyl : ARRAY[0..24]OF BOOL; (* Cylinder in Limp Home *) (* OldName: bLimpHomeCyl; Cycle: 2 *)
		bTimingRedActMx : ARRAY[0..24]OF BOOL; (* *) (* OldName: bTimingRedActMx; Cycle: 2 *)
		bPBC_Event_GC : BOOL; (* PBCMem trigger for GridCode event *) (* OldName: new PV; Cycle:2; *)
		bPBC_Event_Misf : BOOL; (* PBCMem trigger for Misfire event *) (* OldName: new PV; Cycle:2; *)
		bGrC_VoltageLow : BOOL; (* TRUE if voltage is below limit *) (* OldName: bGridCodeVoltageLow; Cycle:5; *)
		bGrC_CurrentChange : BOOL; (* TRUE if generator current change is above limit *) (* OldName: bGridCodeCurrentChange; Cycle:2; *)
		bGrC_SpeedChange : BOOL; (* TRUE if Grid Code event speed change is detected *) (* OldName: bGridCodeSpeedChange; Cycle:2; *)
		rDur_Map_Offs : ARRAY[0..24]OF REAL; (* Duration Map offset *) (* OldName: new PV; Cycle: 2 *)
		rDur_PID_Offs : ARRAY[0..24]OF REAL; (* Duration controller offset *) (* OldName: new PV; Cycle: 2 *)
		rCQ : ARRAY[0..24]OF REAL; (* Combustion Quality*) (* OldName: new PV; Cycle: 2 *)
		rCQ_Max : ARRAY[0..24]OF REAL; (* Combustion Quality*) (* OldName: new PV; Cycle: 2 *)
		bFastRamp_Rel : BOOL; (* release fast load ramp  *) (* OldName: bFreigabeSchnelleRampe; Cycle:2; *)
		bLR_GasStop : BOOL; (*close gas valve to react on a load rejection by the GCB and force  actuators (open CBP, close TV)*)
		rPmax_Offset_Coef_a : REAL; (* coefficient for the pmax offset calculation*)
		rPmax_Offset_Coef_b : REAL; (* coefficient for the pmax offset calculation*)
		iNum_KnckFiltEngCyc : INT; (* Engine cycles for knock containment V2*) (* OldName: newPV; Cycle: 2;*)
		bType6_Update_Rel : BOOL; (* Enables Type6 Engine controls Update (100% Loadrejection, Island mode etc..) *) (*OldName:newPv; Cycle:5;*)
		iIdx_PI_Bal_State : USINT; (* State of Balancer *) (* OldName: ucBal_State; Cycle: 2 *)
		rDur_BAL_SumCor : REAL; (* Balancer: sum correction of PI Duration in [deg.CA]*) (* OldName: new PV; Cycle: 2 *)
		rPr_PMaxOffs_BAL_SumCor : REAL; (* Balancer: sum correction of PMax Offset in [%]*) (* OldName: new PV; Cycle: 2 *)
		bFreezeOptiCyl : ARRAY[0..24]OF BOOL; (* optimizer frozen *) (* OldName: new PV; Cycle: 2 *)
		bPBC_Mon_Active : BOOL; (* monitoring for sensor failure active? *) (* OldName: new PV; Cycle: 2 *)
		bPBC_SensF : ARRAY[0..24]OF BOOL; (* Sensor failure *) (* OldName: new PV; Cycle: 2 *)
		bHiContrCyl : ARRAY[0..24]OF BOOL; (* HiCtr interference on cylinder *) (* OldName: bHiContrCyl; Cycle: 2 *)
		rT_EG_LimMax : REAL; (* exhaust gas temperature limit *) (* OldName: new PV; Cycle: 2 *)
		rVol_TotalGas_Norm : REAL; (*Total gas volume flow [Nm3/h]*) (* OldName: new PV; Cycle: 2 *)
		rPr_CPP_Filt : ARRAY[0..24]OF REAL; (* filtred cylinder peak pressure containment V3 *) (* OldName: newPV; Cycle: 2;*)
		tiSFIKW_OffDelay : TIME; (* Hold On Delay for SFIKW Bit, default 100ms*) (* OldName: newPV; Cycle: 2;*)
		bTripCyl : ARRAY[0..24]OF BOOL; (* Cylinder Trip Information *) (* OldName: newPV; Cycle: 2 *)
		bSkipCylAct : ARRAY[0..24]OF BOOL; (* Cylinder Skip Information *) (* OldName: newPV; Cycle: 2 *)
		rP_Ramp_FS_Norm : REAL; (* gas specific fast start ramp from EC *) (*OldName:new PV;Cycle:2;*)
		bLimpHomeCylTrip : ARRAY[0..24]OF BOOL; (* Cylinder Trip because Limp Home *) (* OldName: bLimpHomeCylTrip; Cycle: 2 *)
		bPFPDR_Act : BOOL; (* PFPDR active *) (* OldName: new PV; Cycle: 2 *)
		bPFPDR_Knck_Slow : BOOL; (* PFPDR slow knock time *) (* OldName: new PV; Cycle: 2 *)
		rCA_IP_StartOffs : REAL; (* FS IP Offset *) (* OldName: newPV; Cycle: 2;*)
		rCA_IP_EGTCtr_Offs : REAL; (* FS IP Offset from EGTCtr *) (* OldName: newPV; Cycle: 2;*)
		bFS_IP_Offs_Trip : BOOL; (* fast start IP Offset trips because of EGT *) (* OldName: newPV; Cycle: 2;*)
		rCA_IP_Set_Raw : REAL; (* ignitoin timing set point raw (without 0.5deg./s ramp)*) (* OldName: newPV ; Cycle:2; *)
		bTP_GrC_Event : BOOL;
		rCoV100 : ARRAY[0..24]OF REAL; (*CoV [cylinder*)
		rCoV_Med : REAL;
		rCoV_min : REAL;
		rCoV_max : REAL;
		rCoV_Avg : REAL;
		rCoV_Set : REAL;
		rCA_MFB_Set : REAL;
		bsy_lfg_SG : BOOL;
		bGridCode_ON : BOOL; (*any dyn. GridCode function activated*)
		bPIOptiChange : BOOL; (* time pulse after a change of the PI optimizer *) (* OldName: newPV ; Cycle:2; *)
		rEta_Gen : REAL; (* eta generator *) (* OldName: rEta_Gen; Cycle: 2 *)
		rEta_Eng : REAL; (* eta engine *) (* OldName: rEta_Eng; Cycle: 2 *)
		rVE_Eng : REAL; (* Volumetric Efficiency *) (* OldName: rLieferGMotor; Cycle: 2 *)
		bPermPreLube_Dem : BOOL; (* Demand permanent prelubification to AuxiliariesGeneral *)
		rP_Ramp_max_BR6_FC : REAL; (* maximum loadramp allowed for type 6 in FC mode *)
		bFS_Act : BOOL; (* FastStart activated (enabled and required from customer) *)
		rPumpQuotient : REAL; (*korriegierte Gasmenge bezogen auf Gesamtgasmenge für Pumperkennung*)
		rP_el_max_red : REAL; (* Calculated power for power reduction GR [kW] *)
		bPBC_Active : BOOL; (* PBC is active, since activation power is reached *)
		iNum_CPP_Int : ARRAY[0..24]OF INT; (* Cylinder peak pressure integrator level *) (* OldName:new PV; Cycle: *)
		rP_Red_CppInt_Norm : REAL; (* Power reduction by Cylinder Peak Pressure Integrator *) (*OldName: newPV; Cycle: 5; *)
		rNFlow_ESC_UreaOffs : REAL; (* Urea controller offset from Emission Supervisory Controller (ESC) controller (l/h) *)
		rCF_ESC_UreaNFlow : REAL; (* Urea controller gain correction factor send from ESC (-) *)
		rNOx_ESC_CatOut_Set : REAL; (* Reference NOx at SCR output from ESC (ppm) *)
		bESC_enable : BOOL; (* enable ESC *)
		tReady4FastStart : HALioDo_Type; (* Engine ready for fast start *)
		tReady4VeryFastStart : HALioDo_Type; (* Engine ready for very fast start *)
		r_PhaseAng_Stat : REAL; (* statischer Polradwinkel [deg.el] *) (* OldName: r_PolarWheelAng_GC; Cycle: 2 *)
		bLOX_Limit_OpMsg : BOOL; (*Prevent LOX-Limit by misfire detection*)
		bBloc_SY_FS : BOOL; (* TRUE = SY Blockieren -> warten um Turbo aufzuheizen *)
		rLamSteadyState : REAL; (* Steady State Lambda - Ausgang GEN2 *)
		bGT_Check4FastStart : BOOL; (* Start gas train check to prepare for fast start *)
		bReady4VeryFastStart : BOOL; (* Ready for very fast start *)
		bReady4FastStart : BOOL; (* Ready for fast start *)
		bVeryFastStart_Prep : BOOL; (* very fast start preperation running *)
		bFastStart_Prep : BOOL; (* fast start preperation running *)
		bGen2_NetP_ena : BOOL; (* GEN2 controller for grid mode activated *)
		bGen2_island_ena : BOOL; (* GEN2 controller for island mode activated *)
		bFastStart_ready_running : BOOL; (*Engine ready for fast start (engine stopped) OR fast start in action (until target load reached for the first time) *)
		iFastStart : USINT; (* Type of Start: 0=normal start, 1=fast start, 2=very fast start, 5=5min start *)
		rCA_IgnP_Avg : REAL; (*Average ITP [deg./KW]*)
		bZylAusfallTP : BOOL; (* 1s long pulse if a cylinder starts burning again *)
		rPr_P2s_RefOffs_ESC : REAL; (*Offset for actual boost pressure reference value send to Gen2 controller to lean out and run on lower Nox levels (bar)*)
		rCA_IP_Offs_ESC : REAL; (*Offset for actual global ignition timing reference value send to IT controller to operate engine close to exhaust temperature limits for fast SCR heating during cold and warm start (CAD)*)
		bLimpHomeCylRKS : ARRAY[0..24]OF BOOL; (* Cylinders in LimpHomeRKS *) (* OldName: newPV; Cycle: 2;*)
		bEGT_Fail : ARRAY[0..24]OF BOOL; (* EGT Sensor failure *) (* OldName: MSAGT ; Cycle: *)
		rT_EO_FS_Perm : REAL; (* minimum engine oil temperature for fast start *)
		rPr_Leanox_Dev : REAL; (* leanox controller deviation [bar] *) (* OldName: ssPressLeanoxError; Cycle: 2 *)
		rMisf_Intgr : REAL; (* integrator electrical misfires [0..1] *) (* OldName: ssMisfInt; Cycle: 2 *)
		rP_Power_Dev : REAL; (* power controller deviation [kW] *) (* OldName: new PV; Cycle: 2 *)
		rN_Speed_Dev : REAL; (* speed controller deviation [rpm] *) (* OldName: new PV; Cycle: 2 *)
		tLL : _tLL_Struct; (* Leanox line for all gas types, including interpolation *)
		xGen2_dbgOut : tGen2Debug;
		tDAI_V_Dem : HALioDo_Type; (* DO: DAI shut off valve open command M.32-YCS-001*)
		tDAI_Dem : HALioDo_Type; (*DO: Demand DAI actuator bank A and B M.05-YCI-104,M.05-YCI-204*)
		tPos_DAI_Set_A : HALioAo_Type; (* AO: Position setpoint DAI control valve bank A M.05-YCI-104*)
		tPos_DAI_Set_B : HALioAo_Type; (* AO: Position setpoint DAI control valve bank B M.05-YCI-204*)
		bLX2_LGM_block : BOOL; (* Blocking signal from LX2 to disable monitoring *)
		bGT_GrC_Bloc : BOOL; (* Block main gastrain in case of grid event *)
		bFastChange : BOOL; (* Special Gas: Fast Gas Quality Change *)
		rPr_P2sGen2_GasQualOffs : REAL; (* GEN2: boost pressure offset gas quality change [bar]*)
		bGCB_DCon_EC : BOOL; (*GCB open command from EngineController *)
		bSkip_active : BOOL; (* static skipfire from Gen2 is active *)
		rP_el_max_red_PCGT : REAL; (* Calculated power for power reduction PCGT [kW] *)
		rLam_PBC : REAL; (* lambda determined by the in cylinder pressure sensor *)
		rLam_LamCtrPBC_ref : REAL; (* lambda reference from lambda controller PBC *)
		bLp_c_Enable : BOOL; (*LEANOX point at low load enabled*)
		bFRT_EPS : BOOL; (* Fault ride trough event in island operation *)
		bGridStat_GridLoss : BOOL; (* Grid status detection: grid loss detected *)
		bLR_ActSat_CBV : BOOL; (* load rejection flag for muting crankcase pressure max trip *)
		bFSync_NarrowSyncWin : BOOL; (* use narrow sync window if fast-sync controller is active *)
		usGasDensN : ARRAY[0..4]OF UINT; (*Nominal gas density for usGasDensN*)
		bLeanOut_H2 : BOOL; (* Active lean out of engine via H2 content *)
		bBlock_WG_CAN_Conf : BOOL; (*WG CAN configuration in progress*)
		rH2_Mix : REAL; (* Hydrogen concentration volumetric for H2 compensation function after gas mixing *)
		iCyl_CombAnomaly : USINT; (* Cylinder no. with combustion anomaly detection *)
		rHum_Mixture_Abs : REAL; (* absolute humidity mixture [g/kg] *)
		bType6L_GEN1_Island : BOOL; (*Activation of T6 GEN1 island controller improvements for L-version SSTC 23bar BMEP*)
		bLR_Act_DBOV : BOOL; (* load rejection flag for activating dome blow off valve *)
		rFlow_VR_TJ : REAL; (*Volume change V-room for pre chamber gas bypass valve [m3/s]*)
		tPos_WG_B : Pos_WG;
		tPos_WG_A : Pos_WG;
		tPos_WG : Pos_WG;
	END_STRUCT;
	Gtyp_Struct : 	STRUCT
		mp_a : ARRAY[0..4]OF _tMeasurePoint; (* leanox line meassure point 1 *) (* OldName: mp_a; Cycle: 2 *)
		mp_b : ARRAY[0..4]OF _tMeasurePoint; (* leanox line meassure point 2 *) (* OldName: mp_b; Cycle: 2 *)
		mp_c : ARRAY[0..4]OF _tMeasurePoint; (* leanox line meassure point 3 *) (* Cycle: 2 *)
		rT_T2_Set : ARRAY[0..4]OF REAL; (* setpoint charge temperature *) (* OldName: tg_soll ; Cycle: 2 *)
		rPr_P2_Dev_Lim : ARRAY[0..4]OF REAL; (* boost perssure deviation maximum *) (* OldName: l_limit ; Cycle: 2 *)
		tLeanox_CDS_Pos : ARRAY[0..4]OF tSimPID_DS_typ; (* PID setting for Leanox *) (* OldName: l_prop / I_int / l_diff / l_tot; Cycle: 2 *)
		tLeanox_CDS_Lam : ARRAY[0..4]OF tSimPID_DS_typ; (* PID setting for Leanox TECJET *) (* OldName: l_prop / I_int / l_diff / l_tot; Cycle: 2 *)
		rP_Ramp_IncGrad_Norm : ARRAY[0..4]OF REAL; (* gradient for increase of power ramp in grid mode *) (* OldName: t_up ; Cycle: 2 *)
		rP_Ramp_DecGrad_Norm : ARRAY[0..4]OF REAL; (* gradient for decrease of power ramp in grid mode *) (* OldName: t_down ; Cycle: 2 *)
		rPos_TV_Opt : ARRAY[0..4]OF REAL; (* optimum throttle valve position *) (* OldName: ssDKOpt ; Cycle: 2 *)
		rPos_Gm_Power_Offs : ARRAY[0..4]OF REAL; (* gasmixer position offset for power mode *) (* OldName: ssPOffs ; Cycle: 2 *)
		rPos_Gm_Speed_Offs : ARRAY[0..4]OF REAL; (* gasmixer position offset for speed mode *) (* OldName: ssNPOffs ; Cycle: 2 *)
		rGm_CR_Speed : ARRAY[0..4]OF REAL; (* gasmixer control range for idle controller *) (* OldName: gm_pos_dif ; Cycle: 2 *)
		rLam_CR_Speed : ARRAY[0..4]OF REAL; (* Para: Lambda control range for idle controller *) (* OldName: gm_pos_dif ; Cycle: 2 *)
		rP_Nom_Gastype : ARRAY[0..4]OF REAL; (* engine nominal power *) (* OldName: p_nenn ; Cycle: 2 *)
		tgm_zltp_st : ARRAY[0..4]OF _tRLinear; (* scale gasmixer pos. dep. airtemp. *) (* OldName: gm_zltp_st ; Cycle: 2 *)
		tlam_zltp_st : ARRAY[0..4]OF _tRLinear; (* scale lambda pos. dep. airtemp. *) (* OldName: gm_zltp_st ; Cycle: 2 *)
		tgm_olt_st : ARRAY[0..4]OF _tRLinear; (* scale gasmixer pos. dep. oiltemp. *) (* OldName: 0; Cycle: 2 *)
		tlam_olt_st : ARRAY[0..4]OF _tRLinear; (* scale lambda pos. dep. oiltemp. *) (* OldName: 0; Cycle: 2 *)
		rPr_Leanox_Offset_Isand : ARRAY[0..4]OF REAL; (* boost pressure offset for island mode *) (* OldName: 0; Cycle: 2 *)
		rCA_Ign_OP_Start : ARRAY[0..4]OF REAL; (*  ingnition point for start mode *) (* OldName: zzp_start ; Cycle: 2 *)
		rCA_Ign_OP_Power : ARRAY[0..4]OF REAL; (* ingnition point for power mode *) (* OldName: zzp ; Cycle: 2 *)
		rCA_Ign_OP_Speed : ARRAY[0..4]OF REAL; (* ingnition point for speed mode *) (* OldName: zzp_insel ; Cycle: 2 *)
		rGEN2_ITislandLoLoad : ARRAY[0..4]OF REAL; (* ignition point for low loads w. GEN2 control*)
		rCA_Ign_OP_Min : ARRAY[0..4]OF REAL; (* minimum allowed ingnition point *) (* OldName: kl_zzp ; Cycle: 2 *)
		rCA_Ign_OP_Max : ARRAY[0..4]OF REAL; (* maximum allowed ingnition point *) (* OldName: ssMinKlZZP; Cycle: 2 *)
		rCA_Ign_OP_Delta_KL : ARRAY[0..4]OF REAL; (* maximum allowed delta ingnition point for knocking *) (* OldName: ssDZZPKL ; Cycle: 2 *)
		rCA_Ign_OP_Delta_Opt : ARRAY[0..4]OF REAL; (* maximum allowed delta ingnition point for knocking *) (* OldName: ssDZZPOpt ; Cycle: 2 *)
		rLam_TJ_Power_Offs : ARRAY[0..4]OF REAL; (* lambda offset for power mode *) (* OldName: ssPOffs ; Cycle: 2 *)
		rLam_TJ_Speed_Offs : ARRAY[0..4]OF REAL; (* lambda offset for speed mode *) (* OldName: ssNPOffs ; Cycle: 2 *)
		rLam_Start_Offs : ARRAY[0..4]OF REAL; (* Para: Lambda start offset *) (* OldName: ssStartLambdaOffset; Cycle: 2 *)
		rLHV : ARRAY[0..4]OF REAL; (* Para: Lower Heating Value *) (* OldName: rHu; Cycle: 2 *)
		rStdGD : ARRAY[0..4]OF REAL; (* Para: Standard Gas Density *) (* OldName: rRohgas; Cycle: 2 *)
		rMinAirReq : ARRAY[0..4]OF REAL; (* Para: Minimal Air Required *) (* OldName: rlmin; Cycle: 2 *)
		rHCR : ARRAY[0..4]OF REAL; (* Para: Heat Capacity Ratio *) (* OldName: rKappa; Cycle: 2 *)
		rP_Leanox_Act_SP : ARRAY[0..4]OF REAL; (* Leanox activation switching point *) (* OldName: lox_st ; Cycle: 2 *)
		rMin_Air_Ratio : ARRAY[0..4]OF REAL; (* min. required air rate of gassort  *) (* OldName: uslmin ; Cycle: 2 *)
		usHu : ARRAY[0..4]OF UINT; (* caloric value of gassort *) (* OldName: usHu; Cycle: 2 *)
		rPr_P2s_Set_LX_0kW : ARRAY[0..4]OF REAL; (* Para: Charging pressure setpoint at 0kW *) (*OldName: ssResPara198; Cycle:2*)
		rP_Red_Leanox_Start : ARRAY[0..4]OF REAL; (* Start of power reduction LEANOX deviation *)
		rCA_SCR_IP_Max_Offset : ARRAY[0..4]OF REAL; (*SCR Inlet Temperature IP Control - Maximum IP advanced offset gas type [num gastype] [degCA]*)
		usGasDensN : ARRAY[0..4]OF UINT; (*Nominal gas density *)
		rLam_Start_Min : REAL; (* Para: Lambda start minimum *)
	END_STRUCT;
	Para_Struct : 	STRUCT  (* eng_ctr *)
		bMisfCont : BOOL; (*PARA [11063]: TRUE = misfire control active *) (* OldName: bMisfCont ; Cycle: 2 *)
		bLIVC : BOOL; (*PARA [11062]: TRUE = Release LIVC controller *) (* OldName: bLIVC ; Cycle: 2 *)
		tCBV_CDS_Idle : tSimPID_DS_typ; (*PARA [11204..11207,12392,12393]: PID setting for compressor bypass valve: Idle *) (* OldName: 0; Cycle: 2 *)
		tCBV_CDS_Power : tSimPID_DS_typ; (*PARA [11208..11211,12394,12395]: PID setting for compressor bypass valve: Power *) (* OldName: tp; Cycle: 2 *)
		tCBV_CDS_Speed : tSimPID_DS_typ; (*PARA [11214..11217,12396,12397]: PID setting for compressor bypass valve: Speed *) (* OldName: tnp ; Cycle: 2 *)
		tTV_CDS_Idle : tSimPID_DS_typ; (*PARA [11277..11280,12385,12386,12437]: PID setting for throttle valve: Idle *) (* OldName: n ; Cycle: 2 *)
		tTV_CDS_Power : tSimPID_DS_typ; (*PARA [11281..11284,12387,12389]: PID setting for throttle valve: Power *) (* OldName: p ; Cycle: 2 *)
		tTV_CDS_Speed : tSimPID_DS_typ; (*PARA [11285..11288,12388,12390]: PID setting for throttle valve: Speed *) (* OldName: np ; Cycle: 2 *)
		rN_EngNom : REAL; (*PARA [12128]: nominal speed *) (* OldName: n_nenn ; Cycle: 2 *)
		bTSTC_Exist : BOOL; (*PARA [10018]: TRUE = two stage turbo charger is assembled *) (* OldName: 0; Cycle: 2 *)
		bTJ_Exist : BOOL; (*PARA [11400]: TRUE=gas inject valves are active *) (* OldName: bTecJetOn ; Cycle: 2 *)
		rMin_Air_Ratio : ARRAY[0..4]OF REAL; (*PARA [11156..11159]: min. required air rate of gassort  *) (* OldName: uslmin ; Cycle: 2 *)
		iN_GMU_Devices : INT; (*PARA [11352]: Number of installed gas metering devices*) (*OldName: ucNrOfTJ; Cycle: 5*)
		mp_a : ARRAY[0..4]OF _tMeasurePoint; (*PARA: leanox line meassure point 1 *) (* OldName: mp_a; Cycle: 2 *)
		mp_b : ARRAY[0..4]OF _tMeasurePoint; (*PARA: leanox line meassure point 2 *) (* OldName: mp_b; Cycle: 2 *)
		mp_c : ARRAY[0..4]OF _tMeasurePoint; (*PARA: leanox line meassure point 3 *) (* Cycle: 2 *)
		rT_T2_Set : ARRAY[0..4]OF REAL; (*PARA [11195..11198]: setpoint charge temperature *) (* OldName: tg_soll ; Cycle: 2 *)
		scDreh : SINT; (*PARA [11201]: factor for speed compensation *) (* OldName: scDreh; Cycle: 2 *)
		ucLiefer : USINT; (*PARA [11289]: volumetric efficiency *) (* OldName: ucLiefer; Cycle: 2 *)
		rP_Eng_Frict : REAL; (*PARA [11161]: engine friction power *) (* OldName: ssPreib ; Cycle: 2 *)
		rN_Start_Trig : REAL; (*PARA [12092]: start up speed trigger value *) (* OldName: n_start; Cycle: 2 *)
		usHu : ARRAY[0..4]OF UINT; (*PARA [11291..11294]: caloric value of gassort *) (* OldName: usHu; Cycle: 2 *)
		rGen_Inertia : REAL; (*PARA [11131]: generator inertia *) (* OldName: JGenerator ; Cycle: 2 *)
		rPr_P2_Dev_Lim : ARRAY[0..4]OF REAL; (*PARA [11183..11186]: boost perssure deviation maximum *) (* OldName: l_limit ; Cycle: 2 *)
		rP_Leanox_Act_SP : ARRAY[0..4]OF REAL; (*PARA [11163..11166]: Leanox activation switching point *) (* OldName: lox_st ; Cycle: 2 *)
		tLeanox_CDS : ARRAY[0..4]OF tSimPID_DS_typ; (*PARA: PID setting for Leanox *) (* OldName: l_prop / I_int / l_diff / l_tot; Cycle: 2 *)
		tLeanox_CDS_TJ : ARRAY[0..4]OF tSimPID_DS_typ; (*PARA: PID setting for Leanox TECJET *) (* OldName: l_prop / I_int / l_diff / l_tot; Cycle: 2 *)
		rP_Ramp_IncGrad_Norm : ARRAY[0..4]OF REAL; (*PARA 12104..12107[]: gradient for increase of power ramp in grid mode *) (* OldName: t_up ; Cycle: 2 *)
		rP_Ramp_DecGrad_Norm : ARRAY[0..4]OF REAL; (*PARA [12100..12103]: gradient for decrease of power ramp in grid mode *) (* OldName: t_down ; Cycle: 2 *)
		rPos_TV_Opt : ARRAY[0..4]OF REAL; (*PARA [11179..11182]: optimum throttle valve position *) (* OldName: ssDKOpt ; Cycle: 2 *)
		bDrehzkorr : BOOL; (*PARA [11049]: TRUE=speed compensation on *) (* OldName: bDrehzkorr ; Cycle: 2 *)
		rPos_Gm_Power_Offs : ARRAY[0..4]OF REAL; (*PARA [11169..11172]: gasmixer position offset for power mode *) (* OldName: ssPOffs ; Cycle: 2 *)
		rPos_Gm_Speed_Offs : ARRAY[0..4]OF REAL; (*PARA [11173..11176]: gasmixer position offset for speed mode *) (* OldName: ssNPOffs ; Cycle: 2 *)
		bLeanox_Speed_Exist : BOOL; (*PARA [11060]: TRUE=leanox in island mode active *) (* OldName: lox_np_akt ; Cycle: 2 *)
		rGm_CR_Speed : ARRAY[0..4]OF REAL; (*PARA [11132..11135]: gasmixer control range for idle controller *) (* OldName: gm_pos_dif ; Cycle: 2 *)
		rLam_CR_Speed : ARRAY[0..4]OF REAL; (*PARA [12447..12450]: Lambda control range for idle controller *) (* OldName: gm_pos_dif ; Cycle: 2 *)
		rP_Nom_Gastype : ARRAY[0..4]OF REAL; (*PARA [12096..12099]: engine nominal power *) (* OldName: p_nenn ; Cycle: 2 *)
		rLeanoxRamp : REAL; (*PARA [11290]: Ramp for Leanox deviation power reduction *) (* OldName: ucPerLeanoxRamp; Cycle: 2 *)
		bZZPKorr : BOOL; (*PARA [11066]: TRUE = timing point controller on *) (* OldName: 0; Cycle: 2 *)
		bt2Korr : BOOL; (*PARA [11065]: TRUE = mixture temp. comp. On *) (* OldName: 0; Cycle: 2 *)
		bSKompFact : BOOL; (*PARA [11064]: TRUE = special speed compensation on *) (* OldName: 0; Cycle: 2 *)
		ssnKompFact : INT; (*PARA [11202]: Correction factor for Leanox speed compensation *) (* OldName: 0; Cycle: 2 *)
		rP_P2sRedIP_SP_Norm : REAL; (*PARA [11203]: switch point power p2`comp.via ITP *) (* OldName: ssPZZPmin; Cycle: 2 *)
		bLeanoxPRED : BOOL; (*PARA [11061]: TRUE = power reduction is activ *) (* OldName: 0; Cycle: 2 *)
		rNOxS_Eng_Set : REAL; (*PARA [????]: set point NOx@x%O2 [mg] *) (* OldName: ssNOX_SOLL ; Cycle: 2 *)
		rTD_LeanoxC_PowerMode : REAL; (*PARA [11199]: time delay for leanox controller after switching to power mode *) (* OldName: LLDT2 ; Cycle: 2 *)
		rTD_LeanoxC_Start : REAL; (*PARA [11200]: time delay for leanox controller after start *) (* OldName: LLDT1 ; Cycle: 2 *)
		rP2s_Comp_Act_SP : REAL; (*PARA [11167]: P2s compensation activation switching point *) (* OldName: ssPtMin ; Cycle: 2 *)
		rT_Eng_Oel_Min : REAL; (*PARA [11194]: minimum Oiltemperatur for Pre-Leanox Operation *) (* OldName: toelmin ; Cycle: 2 *)
		rT_Eng_Oel_Max : REAL; (*PARA [11193]: maximum Oiltemperatur for Pre-Leanox Operation *) (* OldName: toelmax ; Cycle: 2 *)
		rT_Eng_AI_Min : REAL; (*PARA [11192]: minimum Airinlettemperatur for Pre-Leanox Operation *) (* OldName: 0; Cycle: 2 *)
		rT_Eng_AI_Max : REAL; (*PARA [11191]: maximum Airinlettemperatur for Pre-Leanox Operation *) (* OldName: 0; Cycle: 2 *)
		tgm_zltp_st : ARRAY[0..4]OF _tRLinear; (*PARA: scale gasmixer pos. dep. airtemp. *) (* OldName: gm_zltp_st ; Cycle: 2 *)
		tlam_zltp_st : ARRAY[0..4]OF _tRLinear; (*PARA: scale lambda pos. dep. airtemp. *) (* OldName: gm_zltp_st ; Cycle: 2 *)
		tgm_olt_st : ARRAY[0..4]OF _tRLinear; (*PARA: scale gasmixer pos. dep. oiltemp. *) (* OldName: 0; Cycle: 2 *)
		tlam_olt_st : ARRAY[0..4]OF _tRLinear; (*PARA: scale lambda pos. dep. oiltemp. *) (* OldName: 0; Cycle: 2 *)
		rPr_Leanox_Offset_Isand : ARRAY[0..4]OF REAL; (*PARA [13374..13377]: boost pressure offset for island mode *) (* OldName: 0; Cycle: 2 *)
		rCA_Ign_OP_Start : ARRAY[0..4]OF REAL; (*PARA [11127..11130]: ingnition point for start mode *) (* OldName: zzp_start ; Cycle: 2 *)
		rCA_Ign_OP_Power : ARRAY[0..4]OF REAL; (*PARA [11119..11122]: ingnition point for power mode *) (* OldName: zzp ; Cycle: 2 *)
		rCA_Ign_OP_Speed : ARRAY[0..4]OF REAL; (*PARA [11123..11126]: ingnition point for speed mode *) (* OldName: zzp_insel ; Cycle: 2 *)
		rCA_Ign_OP_Min : ARRAY[0..4]OF REAL; (*PARA [11115..11118]: minimum allowed ingnition point *) (* OldName: kl_zzp ; Cycle: 2 *)
		rCA_Ign_OP_Max : ARRAY[0..4]OF REAL; (*PARA [11111..11114]: maximum allowed ingnition point *) (* OldName: ssMinKlZZP; Cycle: 2 *)
		rCA_Ign_OP_Delta_KL : ARRAY[0..4]OF REAL; (*PARA [11103..11106]: maximum allowed delta ingnition point for knocking *) (* OldName: ssDZZPKL ; Cycle: 2 *)
		rCA_Ign_OP_Delta_Opt : ARRAY[0..4]OF REAL; (*PARA [11107..11110]: maximum allowed delta ingnition point for knocking *) (* OldName: ssDZZPOpt ; Cycle: 2 *)
		bIng_IP_Global_Exist : BOOL; (*PARA [11059]: TRUE = global ignition point is used *) (* OldName: bZZPglobal ; Cycle: 2 *)
		rP_Eng_KC_Act_Lim : REAL; (*PARA [11162]: activation power for knock controller *) (* OldName: klopf_akt; Cycle: 2 *)
		bIng_CBVOpt_Exist : BOOL; (*PARA [11058]: TRUE = ignition timing point optimisation for CBV active *) (* OldName: bZZPOpt ; Cycle: 2 *)
		rPos_CBVOpt_Set : REAL; (*PARA [11168]: setpoint for CBV optimisation *) (* OldName: ssTurboOpt ; Cycle: 2 *)
		bKLS98_Active : BOOL; (*PARA [12071]: TRUE = KLS98 active *) (* OldName: kls98_vis; Cycle: 2 *)
		bIgnP_Opt_Exist : BOOL; (*PARA [11057]: TURE =  igniton timing point optimisation is active *) (* OldName: bCylOpt; Cycle: 2 *)
		iMisf_Intgr_Down : INT; (*PARA [11067]: misfire down integrator *) (* OldName: ssMisfDown ; Cycle: 2 *)
		iMisf_Intgr_Up : INT; (*PARA [11068]: misfire up integrator  *) (* OldName: ssMisfUp ; Cycle: 2 *)
		rMisf_Intgr_Limit : REAL; (*PARA [11160]: limit for misfire warning *) (* OldName: Auss_w ; Cycle: 2 *)
		iMisf_Ramp_Grad : INT; (*PARA [11069]: max. power decrease [kW/sec] *) (* OldName: aussetz_li ; Cycle: 2 *)
		bPr_Ch_P2_Exist : BOOL; (*PARA [10134]: TRUE = boost pressure sensor after throttle valve active *) (* OldName: bP2_Act; Cycle: 2 *)
		bSA_Ign_Active : BOOL; (*PARA [12117]: TRUE = SAFI ignition function is enabled/active *) (* OldName: bSAFIIgn_Act; Cycle: 2 *)
		bSA_EG_Active : BOOL; (*PARA [12115]: TRUE = SAFI exh. temp. measur. is enabled/active *) (* OldName: bSAFIExhT_Act; Cycle: 2 *)
		bSA_Active : BOOL; (*PARA [12114]: TRUE = SAFI is enabled/active *) (* OldName: bSAFI_Act; Cycle: 2 *)
		rKno_T2s_Red_Max : REAL; (*PARA [11147]: maximum t2s reduction by knocking   *) (* OldName: kl_dt2; Cycle: 2 *)
		rT_EG_Dev_Lo : REAL; (*PARA [11190]: cylinder temperatur negativ deviation limit *) (* OldName: t_zyl_gr1; Cycle: 2 *)
		rT_EG_Dev_Hi : REAL; (*PARA [11189]: cylinder temperatur positiv deviation limit *) (* OldName: t_zyl_gr2; Cycle: 2 *)
		rT_EG_Abs_Hi_UPR : REAL; (*PARA [11187]: cylinder temperatur maximum upper power range   *) (* OldName: t_zyl_gr3; Cycle: 2 *)
		rT_EG_Abs_Hi_LPR : REAL; (*PARA [11188]: cylinder temperatur maximum lower power range *) (* OldName: t_zyl_gr4; Cycle: 2 *)
		bEGT_Exist : BOOL; (*PARA [11052]: exhaust gas monitoring active *) (* OldName: abgas_a; Cycle: 2 *)
		bEGT_Abs_Hi_Exist : BOOL; (*PARA [11050]: TRUE = exhaust gas temperature maximum monitoring active *) (* OldName: zyl_max_a ; Cycle: 2 *)
		bEGT_Dev_Exist : BOOL; (*PARA [11051]: TRUE = exhaust gas temperature deviation monitoring active *) (* OldName: zyl_abw_a; Cycle: 2 *)
		rLam_TJ_Power_Offs : ARRAY[0..4]OF REAL; (*PARA [11148..11151]: lambda offset for power mode *) (* OldName: ssPOffs ; Cycle: 2 *)
		rLam_TJ_Speed_Offs : ARRAY[0..4]OF REAL; (*PARA [11152..11155]: lambda offset for speed mode *) (* OldName: ssNPOffs ; Cycle: 2 *)
		bSA_PBC_Active : BOOL; (*PARA [12119]: TRUE = SAFI PBC function is enabled/active  *) (* OldName: bSAFIDMR_Act; Cycle: 2 *)
		bSA_KLS_Active : BOOL; (*PARA [12118]: TRUE = SAFI KLS function is enabled/active *) (* OldName: bSAFIKLS_Act; Cycle: 2 *)
		iEng_Motortype : INT; (* PARA: Engine Type *) (* OldName: 0; Cycle: 2 *)
		b_IgnIC_900Active : BOOL; (*PARA [12063]: TRUE = CAN ignition system is used *) (* OldName: 0; Cycle: 0 *)
		bHum_Act : BOOL; (*PARA [12310]: HUMIDITY/LOX COMPENSATION ON/OFF *) (* OldName: bHum_Act; Cycle:2; *)
		bHum_T_Offs_Act : BOOL; (*PARA [12311]: MIXTURE TEMP. OFFSET HUM ACT.  *) (* OldName: bHum_T_Offs_Act; Cycle:2; *)
		bHum_Pred_Act : BOOL; (*PARA [12312]: P REDUCTION HUMIDITY ON/OFF *) (* OldName: bHum_Pred_Act; Cycle:2; *)
		rP_Red_Hum_Lim_Norm : REAL; (*PARA [12313]: P RED. LIMIT FOR HUMIDITY *) (* OldName: iP_Red_Hum_Lim; Cycle:2; *)
		rPr_Offs_Hum_Pactive : REAL; (*PARA [12314]: COMP. VALUE AT P KNOCK MON START *) (* OldName: iPr_Offs_Hum_Pactive; Cycle:2; *)
		rPr_Offs_Hum_Pnom : REAL; (*PARA [12315]: COMPENSATION VALUE AT P NOMINAL *) (* OldName: iPr_Offs_Hum_Pnom; Cycle:2; *)
		rP_Offs_Hum_Pred_Norm : REAL; (*PARA [12316]: HUMIDITY OFFSET *) (* OldName: iP_Offs_Hum_Pred_Norm; Cycle:2; *)
		rT_Hum_Inc_Lim : REAL; (*PARA [12317]: MIXTURE TEMP. MAX RAISE HUM. *) (* OldName: iT_Hum_Inc_Lim; Cycle:2; *)
		rT_Hum_Dev_Tmix_Ticw : REAL; (*PARA [12318]: DEVIATION MIXT.TEMP TO ICWRT *) (* OldName: iT_Hum_Dev_Tmix_Ticw; Cycle:2; *)
		tiTime_Hum_T_Offs : TIME; (*PARA [12319]: MIXT. T. RAISE DEVIATION TIME *) (* OldName: iTime_Hum_T_Offs; Cycle:2; *)
		rPr_Ch_P2sScalMin : REAL; (*PARA [11805]: measure range start charge pressure signal *) (* OldName:anp_pl.y1; Cycle: *)
		rPr_Ch_P2sScalMax : REAL; (*PARA [11804]: measure range end charge pressure signal *) (* OldName:anp_pl.y2; Cycle: *)
		tLeanox_Comp_IgnP : _tRLinear; (*PARA [11273..11276]: leanox setpoint compenstation because of ignition point changes  *) (* OldName: ScaleDZZP; Cycle: 2 *)
		rPos_TV_LimMax : REAL; (*PARA [????]: Throttle valve limit for the maximum position *) (* OldName: ; Cycle:  *)
		rPos_TV_LimMin : REAL; (*PARA [????]: Throttle valve limit for the minimum position *) (* OldName: ; Cycle:  *)
		bExistWasteGate : BOOL; (*PARA [11053]: activation flag for static wastegate control *) (* OldName: bExistWasteGate; Cycle: 2 *)
		rPos_Set_Man_WG_Norm : REAL; (*PARA (saved but no real para) : setpoint of position of the wastegate for the manual adjustment *) (* OldName: ss2stageTC_WG_Set; Cycle: 2 *)
		tLeanox_Comp_ChTmp : _tRLinear; (*PARA [11269..11272]: leanox setpoint compenstation because of charge temperature *) (* OldName: ScaleDPT; Cycle: 2 *)
		bGridCode_Active : BOOL; (*PARA [11055]: Gride Code active *) (* OldName:bGridCode; Cycle: *)
		bGridCodeMonitoringOnly : BOOL; (*PARA [11056]: Grid Code monitoring only active *) (* OldName:bGridCodeMonitoringOnly; Cycle: 2 *)
		rGrC_SpeedChange_Lim : REAL; (*PARA [11141]: Net /Grid Code/Change in speed limit [rpm / s] *) (* OldName: ssGridCodeSpeedChangeLimitsec; Cycle: 2 *)
		rGrC_CurrentChange_Lim : REAL; (*PARA [11137]: Net /Grid Code/Limit current rise [%Inom/s] *) (* OldName: ssGridCodeCurrentChangeLimit; Cycle: 2 *)
		rI_GenNom : ARRAY[0..2]OF REAL; (*PARA [11750..11751]: nominal current generator [1], nominal current grid access point [2] [0..65kA] *) (* OldName:usINennGen; Cycle: 2 *)
		rU_Gen_Nom : ARRAY[0..2]OF REAL; (*PARA [11597..11598]: nominal voltage generator [1], nominal voltage grid access point [2] [70V..65kV] *) (* OldName:usUNennGen; Cycle: 2 *)
		rGrC_Voltage_Lim : REAL; (*PARA [11142]: Grid Code/Undervoltage threshold [0.1%Unom] *) (* OldName: ssGridCodeVoltageLimit; Cycle: 2 *)
		rF_Nom : ARRAY[0..2]OF REAL; (*PARA [11736..11737]: nominal frequency [48..62Hz] *) (* OldName: usFreqNenn[1]; Cycle: 2 *)
		rGrC_AngleSum_Lim : REAL; (*PARA [11136]: Limit angle sum static + dynamic [deg.]*) (* OldName:fAngleSumLIMIT ; Cycle: 2 *)
		rGrC_PoleSlip_Lim : REAL; (*PARA [11140]: Grid Code pole slip limit [rpm/s]*) (* OldName:ssPoleSlipLimit ; Cycle: 2 *)
		rGrC_PolarWheelAngle_Lim : REAL; (*PARA [11139]: Limit Static angle [deg.] *) (* OldName:fPolarWheelAngleLIMIT ; Cycle: 2 *)
		rGrC_XqGen : REAL; (*PARA [11143]: Grid Code generator quadrature-axis reactance (Querreaktanz)*) (* OldName: fXqGen; Cycle: 2  *)
		rGrC_PNom_Lim : REAL; (*PARA [11138]: Limit nominal Power --> if the Power falls below open the GCB *) (* OldName:ssGC_PPROM_LIMIT ; Cycle: 2 *)
		bGrC_CapStop : BOOL; (*PARA [11054]: TRUE = Disconnect from grid at Gridcode-Event when capacitive mode*) (* OldName: ; Cycle: 2 *)
		rKnck_Intgr_Lim : REAL; (*PARA [11146]: Knock integrator limit [%] *) (* OldName: ssTimingRedLimit; Cycle: 2 *)
		rIgnP_Ada_Intv : REAL; (*PARA [11144]: ignition point adaption / interval [deg.CA] *) (* OldName: ssDeltaZZPCylRed; Cycle: 2 *)
		tiIgnP_Red_MI : TIME; (*PARA [11252]: Monitoring interval [min] *) (* OldName: slTimingRedChk; Cycle: 2 *)
		tiIgnP_Opt_Reset : TIME; (*PARA [11250]: Reset time of optimizing [min] *) (* OldName: slZZPCylResetHours; Cycle: 2 *)
		rIgnP_Ada_P : REAL; (*PARA [11145]: Power adaption / interval [%P] *) (* OldName: ssDeltaPELCylRed; Cycle: 2 *)
		tiIgnP_OptP_Reset : TIME; (*PARA [11251]: Reset time of optimizing point red [min] *) (* OldName: slPELCylResetHours; Cycle: 2 *)
		rIgnP_Intgr_Inc : REAL; (* PARA [????]: Increase integration time [s] *) (* OldName: int_up_CylOpt; Cycle: 2 *) (* ======= E *)
		rPr_P2s_CtrLim : REAL; (*PARA [12444]: limit for TV relase *)
		rT_EG_Avg_Dev_Hi : REAL; (*PARA [12297]: cylinder temperatur  average positiv deviation limit [deg.C] *) (* OldName: ssExhTemp_PRed_Lim; Cycle: 2 *)
		bMap_VolEff_Activ : BOOL; (*PARA [12323]: Characteristic map for volumetric efficiency active *) (* OldName: bMap_VolEff; Cycle: 2 *)
		rCBV_Comp_TC : REAL; (*PARA [12324]: time constant for compressor bypass valve compensation *) (* OldName: ustkorr; Cycle: 2 *)
		rCBV_Comp_Amt : REAL; (*PARA [12325]: amount for compressor bypass valve compensation *) (* OldName: ssankorr_no; Cycle: 2 *)
		rCBV_Comp_RedAmt : REAL; (*PARA [12326]: amount reduced for compressor bypass valve compensation *) (* OldName: ssankorr_re; Cycle: 2 *)
		rDN_Up_Lambda_Trig : REAL; (*PARA [12327]: upper engine-speed-delta triggervalue for lambda adaption *) (* OldName: rDN_TRIG_UP_LAMBDA; Cycle: 2 *)
		rDN_Low_Lambda_Trig : REAL; (*PARA [12328]: lower engine-speed-delta triggervalue for lambda adaption *) (* OldName: rDN_TRIG_LOW_LAMBDA; Cycle: 2 *)
		rDP_Up_Lambda_Trig : REAL; (*PARA [12329]: upper power-delta triggervalue for lambda adaption *) (* OldName: rDP_TRIG_UP_LAMBDA; Cycle: 2 *)
		rDP_Low_Lambda_Trig : REAL; (*PARA [12330]: lower power-delta triggervalue for lambda adaption *) (* OldName: rDP_TRIG_LOW_LAMBDA; Cycle: 2 *)
		rCorrFac_DN_NegLambda : REAL; (*PARA [12331]: factor for negative adjustment of lambda via engine-speed-delta *) (* OldName: iK_FACT_DN_NEG_LAMBDA; Cycle: 2 *)
		rCorrFac_DN_PosLambda : REAL; (*PARA [12332]: factor for positive adjustment of lambda via engine-speed-delta *) (* OldName: iK_FACT_DN_POS_LAMBDA; Cycle: 2 *)
		rCorrFac_DP_NegLambda : REAL; (*PARA [12333]: factor for negative adjustment of lambda via power-delta *) (* OldName: iK_FACT_DP_NEG_LAMBDA; Cycle: 2 *)
		rCorrFac_DP_PosLambda : REAL; (*PARA [12334]: factor for positive adjustment of lambda via power-delta *) (* OldName: iK_FACT_DP_POS_LAMBDA; Cycle: 2 *)
		rP_Knck_Act_Hy : REAL; (*PARA [12082]: hyst power start knock control   *) (* OldName: klopf_hys ; Cycle:   *)
		rLam_Start_Offs : ARRAY[0..4]OF REAL; (*PARA [12766..12769]: Lambda start offset *) (* OldName: ssStartLambdaOffset; Cycle: 2 *)
		rLHV : ARRAY[0..4]OF REAL; (*PARA [12750..12753]: Lower Heating Value *) (* OldName: rHu; Cycle: 2 *)
		rStdGD : ARRAY[0..4]OF REAL; (*PARA [12754..12757]: Standard Gas Density *) (* OldName: rRohgas; Cycle: 2 *)
		rMinAirReq : ARRAY[0..4]OF REAL; (*PARA [12758..12761]: Minimal Air Required *) (* OldName: rlmin; Cycle: 2 *)
		rHCR : ARRAY[0..4]OF REAL; (*PARA [12762..12765]: Heat Capacity Ratio (Kappa) *) (* OldName: rKappa; Cycle: 2 *)
		bSA_PI_Active : BOOL; (*PARA [12120]: TRUE = SAFI port injection is enabled/active  *) (* OldName: bSAFIPI_Act; Cycle: 2 *)
		bSel_N2 : BOOL; (*PARA [11312]: Nitrogen scavanging (N2) *) (* OldName: sel_N2; Cycle: 2 *)
		bSel_TwoN2Valves : BOOL; (*PARA [11313]: Two N2 Valves *) (* OldName: sel_TwoN2Valves; Cycle: 2 *)
		bIgn2_Sel_Para : BOOL; (*PARA [12063]: Two ignition systems *) (* OldName: sel_2ignition ; Cycle: 2 *)
		bSG_BackFirePrev : BOOL; (*PARA [12524]: TRUE = backfire prevention activ *) (* OldName: bBackfireIMEP_Pel; Cycle: 2 *)
		bGlowIgnPrevActive : BOOL; (*PARA [12089]: TRUE = glow ignition prevention activ *) (* OldName: sel_GlowIgnPrevent; Cycle: 2 *)
		rLam_SG_Offs : REAL; (*PARA [12495]: Lambda Offset during Fast Power Reduction *) (* OldName: ssSG_lambda_offset  ; Cycle: 2 *)
		rCA_SG_IP_Step : REAL; (*PARA [12496]: Step ITP-Reduction at Pmax detection PBC [deg.CA] *) (* OldName: ssSG_ZZP_step ; Cycle: 2 *)
		ti_SG_EngBlock : TIME; (*PARA [12497]: Block module after run [min] *) (* OldName: ssSG_Blockrun_min; Cycle: 2 *)
		bSG_FPR_Active : BOOL; (*PARA [12498]: Fast power reduction engine (FPR) *) (* OldName: bSG_FPR_aktiv ; Cycle: 2 *)
		bSG_FPR_PBC_Active : BOOL; (*PARA [12499]: Fast power reduction PBC (FPR) *) (* OldName: bSG_DMR_FPR_aktiv; Cycle: 2 *)
		rP_SG_FPR_ActiveLim : REAL; (*PARA [12500]: Power FPR active [kW] *) (* OldName: ssSG_FPR_Paktiv ; Cycle: 2 *)
		rP_SG_FPR_DiffNorm : REAL; (*PARA [12501]: Power difference for detection [%Pnom] *) (* OldName: ssSG_FPR_Peinbruch ; Cycle: 2 *)
		ti_SG_FPR_Diff : TIME; (*PARA [12502]: Time difference for detection [s] *) (* OldName: ssSG_FPR_Teinbruch ; Cycle: 2 *)
		rPr_SG_FPR_P2s_DltLim : REAL; (*PARA [12503]: Limit boost pressure discrepancy [bar/s] *) (* OldName: ssSG_FPR_GW_p2s ; Cycle: 2 *)
		rPos_SG_FPR_TV : REAL; (*PARA [12504]: Throttle flap position FPR *) (* OldName: ssSG_FPR_DKPos ; Cycle: 2 *)
		ti_SG_FPR_TV : TIME; (*PARA [12505]: Time duration FPR [s] *) (* OldName: ssSG_FPR_T ; Cycle: 2 *)
		iNum_SG_FPR_Max : INT; (*PARA [12506]: Max. number FPR during 15min *) (* OldName: ssSG_FPR_max_anz; Cycle: 2 *)
		rP_SG_FPR_LvlNorm : REAL; (*PARA [12507]: Savety Power level when max numbers is exceeded [%Pnom] *) (* OldName: ssSG_FPR_Psave; Cycle: 2 *)
		ti_SG_FPR_PLvlDur : TIME; (*PARA [12508]: Time duration savety power [min] *) (* OldName: ssSG_FPR_T_Psave; Cycle: 2 *)
		bSG_SCO_Active : BOOL; (*PARA [12509]: Emergency Shutdown Engine (ESHUT) *) (* OldName: bSG_SS_aktiv; Cycle: 2 *)
		bSG_SCO_PBC_Active : BOOL; (*PARA [12510]: Emergency Shutdown PBC *) (* OldName: bSG_DMR_SS_aktiv; Cycle: 2 *)
		bSG_SCO_SQ_Ena : BOOL; (*PARA [12523]: Self-reset after shutdown caused by glow ignition *) (* OldName: bSG_SS_SQ ; Cycle: 2 *)
		rP_SG_SCO_ActiveLim : REAL; (*PARA [12511]: Power ESHUT active [kW] *) (* OldName: ssSG_SS_Paktiv; Cycle: 2 *)
		rSG_SCO_SGasMinLim : REAL; (*PARA [12512]: Limit special gas minimum content *) (* OldName: ssSG_SS_minSG; Cycle: 2 *)
		rT_SG_SCO_EG_DevLim : REAL; (*PARA [12513]: Limit positive temperature deviation [deg.C] *) (* OldName: ssSG_SS_Tabw_MW; Cycle: 2 *)
		rT_SG_SCO_EG_DltLim : REAL; (*PARA [12514]: Limit delta Cyl-temperature [deg.C/s] *) (* OldName: ssSG_SS_GWdT; Cycle: 2 *)
		ti_SG_SCO_Dur : TIME; (*PARA [12515]: Time duration gasvalves closed ESHUT [s] *) (* OldName: ssSG_SS_TGASV ; Cycle: 2 *)
		ti_SG_SCO_DurMonDis : TIME; (*PARA [12516]: Time duration monitoring deactivation [s] *) (* OldName: ssSG_SS_TUEBW ; Cycle: 2 *)
		rPos_SG_SCO_TV : REAL; (*PARA [12517]: Throttle flap position ESHUT *) (* OldName: ssSG_SS_DKPos ; Cycle: 2 *)
		ti_SG_SCO_TV : TIME; (*PARA [12518]: Time duration fix throttle flap position [s] *) (* OldName: ssSG_SS_TDKPos ; Cycle: 2 *)
		iNum_SG_SCO_Max : INT; (*PARA [12519]: Max. number of emergency shutdowns *) (* OldName: ssSG_SS_max_anz1 ; Cycle: 2 *)
		ti_SG_SCO_Max : TIME; (*PARA [12520]: Time for max. number of emergency shutdowns [min] *) (* OldName: ssSG_SS_T_max_anz1 ; Cycle: 2 *)
		iNum_SG_SCO_Max_DltT : INT; (*PARA [12521]: Max. number of emergency shutdowns during (30s =dT) *) (* OldName: ssSG_SS_max_anz30s ; Cycle: 2 *)
		ti_SG_SCO_Block : TIME; (*PARA [12522]: ESHUT block time after limit (30s) is exceeded [min] *) (* OldName: ssSG_SS_Tblock_max_anz30s ; Cycle: 2 *)
		iSA_PIValveType : INT; (*PARA [12147]: valve type (1=(BR9) Woodward, 2=(BR9) Hoerbiger, 3=(BR6) Sogav 43, 4=(BR6) Sogav 36), 5= GV40H *) (* OldName: ucPIValveType, bPI_Ventil_Hersteller ; Cycle: 2 *)
		rKno_IP_Red_StP : REAL; (*PARA [12077]: start point for ignition point reduction for knocking *) (* OldName: kl_dz_li; Cycle: 2 *)
		rPr_PBC_Knck_Lim : REAL; (*PARA [12776]: Knock Limit Pressure *) (* OldName: KlopfLimitDMR; Cycle: 2 *)
		rP_PBC_PRed_Norm : REAL; (*PARA [12727]: power reduction PBC sensor failure *) (* OldName: ssDMR_PRed; Cycle: 2 *)
		rPr_CPP_DevLim : REAL; (*PARA [12726]: cylinder peak pressure positive deviation from average*) (* OldName: ssDMR_GWPmaxMW; Cycle: 2 *)
		rPr_CPP_AbsLim : REAL; (*PARA [12728]: limit for cylinder peak pressure *) (* OldName: ssGWPmax; Cycle: 2 *)
		rPr_CPP_AbsLimHi : REAL; (*PARA [14181]: absolute limit for cylinder peak pressure *) (* OldName: ssGWPmax; Cycle: 2 *)
		rPr_CPP_AvgLim : REAL; (*PARA [12738]: mean value limit for cylinder peak pressure *) (* OldName: usMW_Pmax_Limit; Cycle: 2 *)
		iNum_CPP_CycDevLim : INT; (*PARA [12729]: Number stress cycles for pos. Deviation of cylinder peak pressure *) (* OldName: ucAnzCycPmax; Cycle: 2 *)
		iNum_CPP_CycDevLimOK : INT; (*PARA [12730]: Number recovery cycles for pos. Deviation of cylinder peak pressure *) (* OldName: ucAnzCycPmaxOK; Cycle: 2 *)
		rPr_CPP_MSS : REAL; (*PARA [12737]: cylinder peak pressure measurement signal failure lower limit*) (* OldName: usDMRMSS; Cycle: 2 *)
		rPr_IMEP_DevLimMisf : REAL; (*PARA [12731]: mean value deviation limit for IMEP Misfire *) (* OldName: ssParaAbwMWPi_MIS; Cycle: 2 *)
		rPr_IMEP_NegDevLim : REAL; (*PARA [12734]: mean value negative deviation limit for IMEP *) (* OldName: ssParaAbwMWPi; Cycle: 2 *)
		rPr_IMEP_PosDevLim : REAL; (*PARA [12732]: mean value positive deviation limit for IMEP *) (* OldName: ssParaAbwMWPi_Pos; Cycle: 2 *)
		iNum_IMEP_Misf_Lim : INT; (*PARA [12736]: limit for max count of misfire per minute *) (* OldName: ucAnzMisCyl_min; Cycle: 2 *)
		iNum_IMEP_PosDevMax : INT; (*PARA [12733]: Number of engine cycles over IMEP limit *) (* OldName: ucParaAbwPiPosLimit; Cycle: 2 *)
		iNum_IMEP_NegDevMax : INT; (*PARA [12735]: Number of engine cycles below IMEP limit *) (* OldName: ucParaAbwPiNegLimit; Cycle: 2 *)
		rN_EngStart_LimHi : REAL; (* PARA [11296]: speed engine start limit high *) (*OldName:GW_DREHZ; Cycle:5*)
		rN_EngStart_LimHiHi : REAL; (* PARA [11508]: speed engine start limit high high *) (*OldName:GW_HDREHZ; Cycle:5*)
		rMisfCyl_Max_Norm : REAL; (*PARA [12771]: Maximum misfiring cylinders before shutdown [% of cylindernumber]*) (*OldName: ssResPara62, ssResPara199; Cycle:2*)
		ti_OpTi_MisfCyl : TIME; (*PARA [12772]: Maximum operating time with misfiring cylinder *) (*OldName: ssResPara63, ssResPara200; Cycle:2*)
		rP_MisfCtr_SP_Norm : REAL; (*PARA [12773]: Misfire control activation switching point *) (*OldName: ssResPara65 ,ssResPara194; Cycle:2*)
		rP_MisfCtr_Hys_Norm : REAL; (*PARA [12774]: Misfire control deactivation hysterese *) (*OldName: ssResPara66, ssResPara195; Cycle:2*)
		rPr_P2s_Set_LX_0kW : ARRAY[0..4]OF REAL; (*PARA [14201..14204]: Charging pressure setpoint at 0kW *) (*OldName: ssResPara198; Cycle:2*)
		rLam_Start_Min : REAL; (*PARA [12806]: Lambda start minimum *) (*OldName: iLambda_start_min; Cycle:2*)
		bGrC_Prof_Active : ARRAY[0..2]OF BOOL; (*PARA [12874], [12875]: Gridcode voltage profile active *) (*OldName: new PV; Cycle:2*)
		rU_GrC_Prof_Norm : ARRAY[0..2]OF REAL; (*PARA [12877], [12878]: Gridcode voltage profile normalized *) (*OldName: new PV; Cycle:2*)
		ti_GrC_Prof : ARRAY[0..2]OF TIME; (*PARA [12880], [12881]: Gridcode voltage profile time delay *) (*OldName: new PV; Cycle:2*)
		bMFB50Contr_Ena : BOOL; (*PARA [12882]: Enables MFB50 Controller *) (*OldName: new PV; Cycle:2*)
		bP_LoadReject_Active : BOOL; (*PARA [12890]: Load rejection funcitons active *) (*OldName:newPv; Cycle:2;*)
		rP_el_LockTV_Norm : REAL; (*PARA [12884]: ab 4.04 nicht mehr verwendet - Power trigger value to lock the throttle valve in island mode in upper load range *) (*OldName:newPv; Cycle:2;*)
		rP_el_ReleaseTV_Norm : REAL; (*PARA [12885]: ab 4.04 nicht mehr verwendet - Power trigger value to release the throttle valve in island mode *) (*OldName:newPv; Cycle:2;*)
		rPr_CBV_Lock : REAL; (*PARA [12886]: boost pressure to lock the compressor bypass valve in island mode in lower load range *) (*OldName:newPv; Cycle:2;*)
		rPr_CBV_Release : REAL; (*PARA [12887]: boost pressure to release the compressor bypass valve in island mode *) (*OldName:newPv; Cycle:2;*)
		rP_Rot_Norm_Lam_Trig : REAL; (*PARA [12888]: normed rotational power trigger value to trigger the lambda adaption function for type 6 engines *) (*OldName:newPv; Cycle:2;*)
		rKp_P_Rot_Lam : REAL; (*PARA [12889]: proportional gain for the lambda adaption function for type 6 engines *) (*OldName:newPv; Cycle:2;*)
		rPos_CBV_Ref_WG : REAL; (*PARA [13190]: setpoint of position turbobypass valve for wastegate control *) (*OldName:ssPOS_TBPV_SP_WG, rPOS_TBPV_SP_WG; Cycle:2;*)
		bWG_Man : BOOL; (*PARA [13191]: flag for manual adjustment of the wastegate*) (*OldName:bMAN_WG; Cycle:2;*)
		bWG_Check_Ena : BOOL; (*PARA [13404]: Waste gate check anabled *) (*OldName:newPv; Cycle:2;*)
		rPID_EGT_P : REAL; (*PARA [13372]: Exhaust gas temperature controller proportional part *) (*OldName:newPv; Cycle:2;*)
		rPID_EGT_I : REAL; (*PARA [13394]: Exhaust gas temperature controller integral part *) (*OldName:newPv; Cycle:2;*)
		PFPDR : tPFPDR_P; (*PARA [13502..13509]: Peak Fire Pressure Detection Run *) (*OldName:newPv; Cycle:2;*)
		SS : tSS_P; (*PARA [13411..13422]: Steady State Conditions *) (*OldName:newPv; Cycle:2;*)
		FS : tFS_P; (*PARA [13406..13410,13423..13428,14186,14187,14205..14207]: Fast Start *) (*OldName:newPv; Cycle:2;*)
		rCA_AdvTimeLim : REAL; (*PARA [12066]: Advanced ignition timing limit*) (*OldName:AdvTimLi; Cycle:;*)
		rCA_RetTimeLim : REAL; (*PARA [12066]: Retard ignition timing limit*) (*OldName:RetTimLi; Cycle:;*)
		rP_PBC_Act_SP : REAL; (*PARA [13401]: PBC activation switching point *) (*OldName:newPv; Cycle:2;*)
		rP_PBC_Act_Hys : REAL; (*PARA [13402]: PBC activation hysterese *) (*OldName:newPv; Cycle:2;*)
		tiWG_SS_Del : TIME; (*PARA [13405]: State Delay for Wastegate application *) (*OldName:newPv; Cycle:2;*)
		rKno_Int_MinLim : REAL; (*PARA [13460]: lower knock integrator limit for PI Engines *) (*OldName:newPv; Cycle:2;*)
		rN_LamOffs_x1 : REAL; (*PARA [13614]: lambda speed offset, low speed point *) (*OldName:xLCCurve_dLambda_start_tab[1].x; Cycle:2;*)
		rN_LamOffs_x2 : REAL; (*PARA [13615]: lambda speed offset, high speed point *) (*OldName:xLCCurve_dLambda_start_tab[2].x; Cycle:2;*)
		rCA_MFB50_set50 : REAL; (*PARA [13187]: MFB50 setpoint at Pset = 50%Pnom *)
		rCA_MFB50_set100 : REAL; (*PARA [13186]: MFB50 setpoint at Pset = 100%Pnom *)
		rCA_MFB50_ITPOfs_late : REAL; (*PARA [13188]: MFB50 ITP Offset late *)
		rCA_MFB50_ITPOfs_early : REAL; (*PARA [13189]: MFB50 ITP Offset early *)
		rMFB50Ctr_kp : REAL; (*PARA [13323]: MFB50 controller - P component *)
		rMFB50Ctr_ki : REAL; (*PARA [13635]: MFB50 controller - I component *)
		rMFB50_ITP_ratio : REAL; (*PARA [13636]: Ratio ITP/MFB50*)
		bCoVCtr_Act : BOOL; (*PARA [13649]: Activate CoV controller *)
		rCoV_Set50 : REAL; (*PARA [13651]: CoV setpoint at Pset = 50%Pnom *)
		rCoV_Set100 : REAL; (*PARA [13650]: CoV setpoint at Pset = 100%Pnom *)
		rPr_CoV_p2s_Range : REAL; (*PARA [13652]: max. Boost pressure offset CoV controller [mbar]*)
		rCoVCtr_kp : REAL; (*PARA [13653]: CoV controller - P component *)
		rCoVCtr_ki : REAL; (*PARA [13654]: CoV controller - I component *)
		iCBV34_Fun : INT; (*PARA [13655]: choose CBV34 function*)
		rCBV34_Set : REAL; (*PARA [13656]: CVB34 controller - set point *)
		rCBV34_min : REAL; (*PARA [13657]: CVB34 controller - Y min *)
		rCBV34Ctr_kp : REAL; (*PARA [13658]: CVB34 controller - P component *)
		rCBV34Ctr_ki : REAL; (*PARA [13659]: CVB34 controller - I component *)
		rPos_Gm_SG_Offs : REAL; (*PARA [13670]: Gasmixer Offset during fast power reduction or safty cut out *)
		rPos_SG_FPR_CBV : REAL; (*PARA [13669]: CBV Position during fast power reduction *)
		rPos_SG_SCO_CBV : REAL; (*PARA [13671]: CBV Position during safty cut out *)
		iFPRGasRedOpt : INT; (*PARA [13666]: Gas amount reduction at  fast power reduction *)
		rFPRGasRed : REAL; (*PARA [13667]: Gas amount reduction*)
		rFPRGasRedTime : REAL; (*PARA [13668]: Length of reduction of gas amount *)
		bGT_SpecGasActive : BOOL; (* PARA [11374]: Sondergas *)
		bLLLCtr_act : BOOL; (*PARA [13637]: Activate boost pressure idle mode lambda controller *)
		rLLLCtr_delay_Trip : REAL; (*PARA [13645]: Maximum time Lambda limit *)
		rPr_p2s_Win_sy_lfg : REAL; (*PARA [13642]: Boost pressure band for synchronization *)
		rPr_p2s_LLCtr : ARRAY[0..4]OF REAL; (*PARA [13638..13641]: Boost pressure set point for idle mode [bar] [Gastype] *)
		rLLCtr_kp : REAL; (*PARA [13643]: boost pressure idle mode lambda controller - P component *)
		rLLCtr_ki : REAL; (*PARA [13644]: boost pressure idle mode lambda controller - I component *)
		bGridCode_Prof23_Active : BOOL; (*PARA [13185]: Dynamic Grid Code (Profile 2/3) *)
		rKp_LeanoxC_TJ : REAL; (*PARA [13685]: P component idle lambda controller for tecjet engines*)
		rKi_LeanoxC_TJ : REAL; (*PARA [13686]: I component idle lambda controller for tecjet engines*)
		rKp_LeanoxC_GM : REAL; (*PARA [13687]: P component idle lambda controller for gasmixer engines*)
		rKi_LeanoxC_GM : REAL; (*PARA [13688]: I component idle lambda controller for gasmixer engines*)
		rPos_GM_RunUpOffset : REAL; (*PARA [13826]: gas mixer offset for engine start*)
		rN_Eng_RunUpLim : REAL; (*PARA [13825]: speed limit for gas mixer offset*)
		bGEN2_preM_Act : BOOL; (*PARA [13672]: GEN2 controller active pre-mixed engines *)
		rCA_GEN2_fastSt : REAL; (*PARA [13673]: Ignition timing point for cold engine [deg.CA] *)
		rGEN2_PowCtrl_Kp : REAL; (*PARA [13676]: GEN2 controller P component *)
		rGEN2_PowCtrl_Ki : REAL; (*PARA [13677]: GEN2 controller I component *)
		usGasDensN : ARRAY[0..4]OF INT; (*PARA [11353..11356]: Nominal gas density *) (*OldName: usGasDensN; Cycle: 5*)
		bT_EGaLPTC_B_Active : BOOL; (*PARA [11320]: exhaust gas temperature after low pressure turbo charger active*)
		bT_EGaLPTC_A_Active : BOOL; (*PARA [11319]: exhaust gas temperature after low pressure turbo charger active*)
		bSGM_Active : BOOL; (*PARA [12362]: Special Gas Mixer (SGM) active*) (*OldName: bSpecGM; Cycle: 5;*)
		bRej2houseload : BOOL; (*PARA [14079]: Fangen im Eigenbedarf aktiv?*)
		bP2s_Comp_LeanoxDrift : BOOL; (*PARA [13972]: general activation of leanox drift compensation*)
		rP_P2s_Comp_LeanoxDrift_SP : REAL; (*PARA [13977]: leanox drift compensation activation switching point  *)
		tP2s_Comp_LeanoxDrift : _tRLinear; (*PARA [13973..13976]: leanox setpoint compensation because of leanox drift*)
		iOpH_P2s_Comp_LeanoxDrift_Reset : DINT; (*PARA [13978]: reset time of leanox drift function*)
		rCoeff_P2s_Comp_Sector2 : REAL; (*PARA [13979]: dividing factor for second area of leanox drift *)
		iOpH_P2s_Comp_LeanoxDrift_Sec2 : DINT; (*PARA [13980]: operating hours for start second area *)
		iOpH_Nox_Measure_recommend : DINT; (*PARA [13981]: leanox measuremnet recommend *)
		iOpH_Nox_Measure_mandatory : DINT; (*PARA [13982]: leanox measuremnet mandatory *)
		bFastStart_Act : BOOL; (* PARA [14184]: Fast Start package activated *)
		rT_ECW_LimRelLoad : REAL; (*PARA [11945]: temperature engine cooling water limit release load [deg.C]*) (*OldName:GW_LFG; Cycle:5;*)
		rGEN2_BDC_CBV_Kp : REAL; (*PARA [14199]: GEN2 controller BDC CBV P component *)
		rGEN2_BDC_CBV_Ki : REAL; (*PARA [14200]: GEN2 controller BDC CBV I component *)
		rGEN2_BDC_TV_Kp : REAL; (*PARA [14197]: GEN2 controller BDC TV P component *)
		rGEN2_BDC_TV_Ki : REAL; (*PARA [14198]: GEN2 controller BDC TV I component *)
		rScal_Lam_Lean : REAL; (*PARA [14319]: GEN2 scaling magnitude of lean limit*)
		rScal_Lam_Enrich : REAL; (*PARA [14192]: GEN2 scaling magnitude of enrichment*)
		bLam_Offs_Act : BOOL; (*PARA [14193]: GEN2 activation of automatic lambda map offset*)
		bLam_Mon_Act : BOOL; (*PARA [14193]: GEN2 activation OF Lambda monitoring trip*)
		rScal_Lam_Mon_Limit : REAL; (*PARA [14195]: GEN2 Scaling of Lambda monitoring Trip Threshold*)
		rScal_Lam_Mon_Delay : REAL; (*PARA [14196]: GEN2 Lambda monitoring activation delay*)
		iNumCBV : INT; (*PARA [14214]: Number of CBV valves *)
		rOffs_WS_Actuators : REAL; (*PARA [14218]: Offset Worksplit Actuators *)
		bScavBeStart_Active : BOOL; (*PARA [12777]: exhaust gas scavenging before engine start active*) (*OldName:new pv;Cycle:5*)
		bPr_Ch_P2bFA_Exist : BOOL; (*PARA [13478]: sensor charge pressure before flame arrester exist*)
		bPr_Ch_P2HP_Exist : BOOL; (*PARA [13481]: sensor charge pressure after high-pressure turbocharger exist*)
		tiMainsOkDelay : TIME; (*PARA [12216]: mains return delay *) (*OldName:PT_MNS_OK; Cycle:5;*)
		rPI_Dur_CppInt_Offset_Max : REAL; (*PARA [14215]: CPP Integrator Port Injection Duration Reduction Offset maximum [%] *)
		rCA_Ign_CppInt_Offset_Max : REAL; (*PARA [14216]: CPP Integrator CA Ignition Point Timing Reduction Offset maximum [deg.CA] *)
		rP_Red_CppInt_Norm : REAL; (*PARA [14217]: Cylinder Peak Pressure Integrator Power Reduction [% Pnom] *)
		rP_P0_FS : REAL; (*PARA [14353]: P0 for GEN2 controller in case of fast start [% Pnom]*)
		bGEN2island_Act : BOOL; (*PARA [14315]: GEN2 controller active pre-mixed engines in island mode*)
		rGEN2_Lam_offset_Low : REAL; (*PARA [14324]: offset gain lambda GEN2 island low load*)
		rGEN2_Lam_offset_Mid : REAL; (*PARA [14325]: offset gain lambda GEN2 island mid load*)
		rGEN2_Lam_offset_Hi : REAL; (*PARA [14326]: offset gain lambda GEN2 island high load*)
		rGEN2_Lam_Ti_offset : REAL; (*PARA [14327]: offset time constant enrichment GEN2 island *)
		rGEN2_BDC_CBV_Kp_island : REAL; (*PARA [14320]: GEN2 controller BDC CBV P component island *)
		rGEN2_BDC_CBV_Ki_island : REAL; (*PARA [14321]: GEN2 controller BDC CBV I component island*)
		rGEN2_BDC_TV_Kp_island : REAL; (*PARA [14322]: GEN2 controller BDC TV P component island*)
		rGEN2_BDC_TV_Ki_island : REAL; (*PARA [14323]: GEN2 controller BDC TV I component island*)
		rGEN2_OffsetTVLimit : REAL; (*PARA [14341]: GEN2 Offset surge limit for throttle limit*)
		bGEN2_KF_speed : BOOL; (*PARA [????]: turn on / off Kalman filter for speed noise reduction*)
		bGEN2_ActIdle : BOOL; (*PARA [14433]: Gen2 controller active in idle mode after Grid Parallel / Island*)
		bGEN2_250Nox : BOOL; (*PARA [14318]: <250mg/Nm3 NOx version (false: 500mg/Nm3)*)
		rGEN2_fact_Adapt : REAL; (*PARA [14329]: GEN2 island - gain for learning function*)
		rGEN2_fact_Q0 : REAL; (*PARA [14328]: GEN2 island - agressiveness factor*)
		rGEN2_ITislandLoLoad : ARRAY[0..4]OF REAL; (*PARA [14330..14333]: ignition point for low loads w. GEN2 control*) (* OldName: zzp_insel ; Cycle: 2 *)
		rGEN2_ITCtransDelta : REAL; (*PARA [14370]: offset of ignition timing point during transients to avoid knocking*)
		rF_StartIPRed_Norm : REAL; (*PARA [14365]: Start IP reduction due to low frequency [%fnom-norm]*)
		rCA_DeltaIPRed_perHz : REAL; (*PARA [14366]: IP reduction per 1Hz below limit [deg.CA/Hz]*)
		rPowCtrl_rKaw : REAL; (*PARA [14373]: GEN2 controller anti wind up gain*)
		rGEN2_ResetKe : REAL; (*PARA [14372]: Reset of GEN2 island model gain learning function*)
		rGEN2_NthrshSkip : REAL; (*PARA [14371]: Start of skipfire at GEN2: Nominal speed + rGEN2_NthrshSkip *)
		rGen2_fact_LS_FF : REAL; (*PARA [14381]: factor feedforward speed ref to power in GEN2 island control for load sharing*)
		rGen2_delay : REAL; (*PARA [14369]: estimated delay time of gas dosage*)
		rGEN2_fact_R1 : REAL; (*PARA [14368]: GEN2 island - agressiveness factor R[1]*)
		rGEN2_BDC_TV_Kp_island_scalGS : REAL; (*PARA [14342]: GEN2 controller BDC TV P component island - scale Gain Scheduling [0...2]*)
		rGEN2_BDC_CBV_Kp_island_scalGS : REAL; (*PARA [14367]: GEN2 controller BDC CBV P component island - scale Gain Scheduling [0...2]*)
		bLX2_enable : BOOL; (*PARA [14305]: LX2 Main enabling switch parameter*)
		tiLX2_Ctrl_Tn : TIME; (*PARA [14334]: I-time of LX2 Controller [sec]*)
		tiFilterConst_NOx : TIME; (*PARA [14355]: Filter coefficient PT1 - NOx act [sec]*)
		rLX2_SteadyStateFactor : REAL; (*PARA [14356]: LX2 steady state factor*)
		rPr_LX2_OffsetLimit : REAL; (*PARA [14337]: LX2 charge pressure offset limit [mbar]*)
		bDAI_Active : BOOL; (*PARA [14393]: DAI Activate intake assist part (14393) *)
		bDAI_Active_Start : BOOL; (*PARA [14394]: DAI Activate intake assist part (14394) *)
		bDAI_Active_PowRamp : BOOL; (*PARA [14395]: DAI DAI active during load ramp (14395) *)
		bDAI_Active_NetP : BOOL; (*PARA [14396]: DAI active in grid mode (14396) *)
		bDAI_Active_Island : BOOL; (*PARA [14397]: DAI active in isolated mode (14397) *)
		rN_DAI_On : REAL; (*PARA [14398]: DAI activation speed [rpm] *)
		rN_DAI_Off : REAL; (*PARA [14399]: DAI da-activation speed [rpm] *)
		rGain_DAI_Start : REAL; (*PARA [14400]: DAI gain mass flow speed ramp *)
		rGain_DAI : REAL; (*PARA [14401]: DAI gain mass flow *)
		rPr_DAI_In_Hi : REAL; (*PARA [14402]: DAI maximum inlet pressure [bar] *)
		rTExhBound_SensScal : REAL; (*PARA [14424]: Sensitivity factor for tolerace band*)
		bTExhMon_Activation : BOOL; (*PARA [14418]: Exhaust temperature inclination monitoring active*)
		tiDelay_nLPow_dTExhMonAct : TIME; (*PARA [14423]: Delay for reactivation after low load operation*)
		rdT2Exp_MaxDev : REAL; (*PARA [14422]: Maximum positive deviation from median*)
		rFiltTimeCnt_TexhMon : REAL; (*PARA [14421]: Filter constant operation point detection*)
		rdT_Ref_Max_TripNormal : REAL; (*PARA [14420]: Limit for positive deviation from expected value*)
		tiDelay_nGCB_dTExhMonAct : TIME; (*PARA [14419]: Delay for activation after GCB on*)
		rF_OverMp : REAL; (*PARA [14435]: Over frequency in mains parallel operation *)
		tiF_OverMpDel : TIME; (*PARA [14436]: Over frequency delay in mains parallel operation *)
		rF_UnderMp : REAL; (*PARA [14437]: Under frequency in mains parallel operation *)
		tiF_UnderMpDel : TIME; (*PARA [14438]: Under frequency delay in mains parallel operation *)
		rN_Factor_UF_MinP : REAL; (*PARA [14439]: Speed compensation factor underfrequency at half load *)
		rN_Factor_UF_MaxP : REAL; (*PARA [14440]: Speed compensation factor underfrequency at full load *)
		rN_Factor_OF_MinP : REAL; (*PARA [14441]: Speed compensation factor overfrequency at half load *)
		rN_Factor_OF_MaxP : REAL; (*PARA [14442]: Speed compensation factor overfrequency at full load *)
		rT1LP_CBV_Ref_WG_Start : REAL; (* PARA [14455]: start intake temperature for compressor bypass reserve compensation *)
		rGain_T1LP_CBV_Ref_WG : REAL; (* PARA [14456]: gain factor for intake temperature compensation for compressor bypass reserve *)
		rP_Red_Leanox_Start : ARRAY[0..4]OF REAL; (* Start of power reduction LEANOX deviation *)
		bFastGasChange_Active : BOOL; (*PARA [14462]: Fast Gas Quality Change *)
		tiGasQualChange_Delay : TIME; (*PARA [14463]: Time Delay between N2-purging to activation of Fast-Gas-Quality-Change_Function *)
		tiGasQualChange_GlowIgn_Dur : TIME; (*PARA [14464]: Time interval deactivation of Glow-Ignition-Monitoring *)
		tiGasQualChange_CtrFreeze_Dur : TIME; (*PARA [14465]: Timeframe of Fast-Gas-Quality-Change-Function *)
		rLambda_Offset_GasQualChange : REAL; (*PARA [14466]: Lambda offset for Fast-Gas-Quality-Change-Function *)
		bAct_Gen2KeEstimator : BOOL; (* PARA [14498] Activation of Gen2 Ke Estimator for model gain learning*)
		bAct_Gen2KeEstimator_GridP : BOOL; (* PARA [14499] Activation of Gen2 Ke Estimator during GridP Operation for model gain learning*)
		bAct_Gen2TransDetectionKeEst : BOOL; (* PARA [14500] GEN2-island: Activation transient detection for engine model estimation function *)
		rCA_Ign_Act_GrC : REAL; (*PARA [14511]: IP during an FRT event [deg.CA]*)
		ti_TOF_Ign_Act_GrC : TIME; (*PARA [14512]: IP during an FRT event; time duration [s]*)
		rGasFlowDec_MaxP_Prct_GrC : REAL; (*PARA [14513]: Gas dosage multiplication factor at full load druing an FRT event [-]*)
		rGasFlowDec_MinP_Prct_GrC : REAL; (*PARA [14514]: Gas dosage multiplication factor at half load druing an FRT event [-]*)
		tiGasFlowDec_HoldTime_GrC : TIME; (*PARA [14515]: Gas dosage multiplication factor; hold time [ms]*)
		rGasFlowDec_Ramp_GrC : REAL; (*PARA [14516]: Recovery time of gas dosage adaption during an FRT event [ms]*)
		rGasFlowInc_Prct_GrC : REAL; (*PARA [14517]: Gas dosage multiplication factor after an FRT event [-]*)
		rGasFlowInc_Ramp_GrC : REAL; (*PARA [14518]: Recovery time of gas dosage adaption after an FRT event [ms]*)
		bT_SCR_CatIn_Exist : BOOL; (*PARA [13899]: SCR Exhaust temperature CAT inlet active*)
		bT_SCR_CatOut_Exist : BOOL; (*PARA [13902]: SCR Exhaust temperature CAT outlet active*)
		bT_OXIcat_In_Exist : BOOL; (*PARA [14117]: Oxidation Catalyst inlet temperature sensor active*)
		bT_EGaTC_Active : BOOL; (*PARA [11321]: Turbocharger outlet temp. measuring active*)
		rT_SCR_CatIn_Hi : REAL; (*PARA [13900]: SCR Exhaust temperature CAT inlet maximum  [degC]*)
		rT_SCR_bOXI_aTC_Hi : REAL; (*PARA [14942]: SCR Temperature Limit when before OXIcat or after TC sensor used [degC]*)
		bSCR_Active : BOOL; (*PARA [13961]: SCR active*) (*OldName: new PV; Cycle:5*)
		rKp_SCRTCtr : REAL; (* PARA [14563]: SCR Inlet temperature controller proportional factor *)
		rT_SCRTCtr_margin : REAL; (* PARA [14564]: SCR Inlet temperature controller margin [degC]*)
		rF_Under : ARRAY[0..2]OF REAL; (* Para: monitoring limit under frequency *) (* OldName:usUFreq; Cycle: *)
		bN_SpdSetRed_Overload : BOOL; (* PARA [14607] Overload Protection Isolated Operation: Activation Reduction Speed Reference*)
		bCA_ITP_Red_F_Island : BOOL; (* PARA [14611] Overload Protection Isolated Operation: Activation IP adaptation Island *)
		bCorr_LX_GR_Island : BOOL; (* PARA [14612] Activation speed compensation for isolated operation *)
		iSource_F_N_OffsSet : INT; (* PARA [14300] F/N Setpoint: 0= no setpoint, 1= Droop, 2= External, 3= LSL *)
		bGen2_LamMinSy : BOOL; (* PARA [14619] GEN2 lambda limit adaptation after idle operation*)
		bGen2_LamOffsNotSteady : BOOL; (* PARA [14620] GEN2 activation of automatic lambda map offset (non-stationary)*)
		rPr_Gen2P2s_GasQualFactorMax : REAL; (* PARA [14621] GEN2 scaling maximal boost pressure offset for gas quality changes *)
		rPr_Gen2dPTVoffs_x2 : REAL; (* PARA [14633] GEN2 Offset worksplit actuators for transition region *)
		rGen2_FactorRiLQR : REAL; (* PARA [14643] GEN2-island: reduction factor aggressiveness actuators *)
		bLp_c_Ena : BOOL; (* PARA [14575]: LEANOX point at low load enabling switch parameter *)
		iIdx_Ign_LoadProfileOpt : INT; (* PARA [14593]: IP Type9 load dependent profile option: 1=Default, 2=IP retarded in part load for HC interim emission solution *)
		bLamCtrPBC_active : BOOL; (* PARA [14644]: lambda controller PBC activation bit *)
		rGain_LamCtr_Kp : REAL; (* PARA [14645]: proportional gain lambda controller PBC *)
		rGain_LamCtr_Ki : REAL; (* PARA [14646]: integral gain lambda controller PBC *)
		rGain_LamCtr_KAW : REAL; (* PARA [14647]: anti windup gain lambda controller PBC *)
		rLam_LamCtrPBC_Offset_Lim : REAL; (* PARA [14648]: upper and lower limit for lambda controller PBC *)
		rGain_LamPBC_global : REAL; (* PARA [14649]: global coefficient lambda estimation PBC *)
		rGain_LamPBC_power : REAL; (* PARA [14650]: power coefficient lambda estimation PBC *)
		bTrStRed_Ena : BOOL; (*PARA [14613]: TrStRed Main enabling switch parameter*)
		rT_TrStRed_EG_Max_LimMarg : REAL; (*PARA [14615]: margin from max. cyl. temperature for controller setpoint [degC]*)
		rT_EGbTC_LimHi : REAL; (*PARA [11342]: exhaust gas temperature before turbo charger limit high [degC]*)
		bThR_woGas : BOOL; (*PARA [12225]: thermal reactor, select w/o gas injection*)
		rCA_TrStRed_LowLimit : REAL; (*PARA [14614]: control limit TrStRed function - relative ITP [degCA]*)
		rGain_TrStRed_halfLoadLim : REAL; (*PARA [14616]: half load factor for TrStRed function control limit [%]*)
		rFRT_Voltage_Lim : REAL; (* PARA [14722]: Undervoltage threshold in island operation [0.1%Unom] *)
		rFRT_CurrentChange_Lim : REAL; (* PARA [14723]: Limit current rise in island operation [%Inom/s] *)
		rFRT_SpeedChange_Lim : REAL; (* PARA [14724]: Change in speed limit in island operation [rpm/s] *)
		bFRT_Detection_Active : BOOL; (* PARA [14725]: Fault Ride Through Event (Isolated operation) *)
		b_SCR_ITCtrl_Active : BOOL; (*PARA [14636]: SCR Inlet Temperature IP Control Active*)
		rCA_T_SCR_PropGain : REAL; (*PARA [14637]: SCR Inlet Temperature IP Control - Proportional gain [degCA/degC]*)
		rP_SCR_ITCtrl_Off : REAL; (*PARA [14638]: SCR Inlet Temperature IP Control - Maximum power with advanced IP [p.u.]*)
		rCA_SCR_IP_Max_Offset : ARRAY[0..4]OF REAL; (*PARA [14639..14642]: SCR Inlet Temperature IP Control - Maximum IP advanced offset gas type [num gastype] [degCA]*)
		bGridStat_Enable : BOOL; (* PARA [14651]: Grid status dectection activation *)
		rV_Change_Lim : REAL; (* PARA [14652]: Voltage change limit [1/s] *)
		rP_Change_Lim : REAL; (* PARA [14653]: Active power change limit [1/s] *)
		rN_Change_Lim : REAL; (* PARA [14654]: Voltage change limit [rpm/s] *)
		bSEMIC_Active : BOOL; (*PARA [14519]: Ignition controller SEMIC*)
		tiFRT_PowerFix : TIME; (* PARA [14926]: Holding time of power at FRT event [s] *)
		iNum_GT : INT; (*PARA [11403]: Number of gas trains *) (* OldName: 	usNrOfGasTrains 	; Cyclic: ; *)
		bH2_Comp_Active : BOOL; (* PARA [14911]: H2 compensation active *)
		iGastrain_H2_sensor : INT; (* PARA [14912]: Gastrain with H2 sensor *)
		rH2_content_SP : REAL; (* PARA [14913]: Switching point of H2 content *)
		rITP_Comp_H2_prior : REAL; (* PARA [14914]: ITP offset via H2 content before H2 switching point *)
		rITP_Comp_H2_after : REAL; (* PARA [14915]: ITP offset via H2 content after H2 switching point *)
		rPr_P2S_Comp_H2_HL : REAL; (* PARA [14916]: Boost pressure offset via H2 content at half load *)
		rPr_P2S_Comp_H2_FL : REAL; (* PARA [14917]: Boost pressure offset via H2 content at half load *)
		rPr_P2S_Offset_25PrctH2_HL : REAL; (* PARA [14918]: Boost pressure offset at 25% H2 content at half load *)
		rPr_P2S_Offset_25PrctH2_FL : REAL; (* PARA [14919]: Boost pressure offset at 25% H2 content at full load *)
		bHum_Mixture_Act : BOOL; (* PARA [15012]: Humidity compensation plus - including absolute humidity gas *)
		rHum_GasIn_Abs_Backup : REAL; (* PARA [15013]: Absolute humidity gas backup value in case of MSF [g H2O/kg dry gas] *)
		bEng_Act_MSPC : BOOL; (* PARA [15010]: Mixture scavenged pre-chamber *)
		bGEN2_KF_Act : BOOL; (* PARA [15011]: GEN2 - island activation disturbance estimator *)
		rN_Dev_Lim : REAL; (* PARA [14957]: Grid status detection triggers if speed deviation (positive or negative) exceeds limit [%Nnom] *)
		rV_Change_Lim_afterFRT : REAL; (* PARA [14958]: Triggers grid status detection *)
		bSmooth_Isl_Det_Enable : BOOL; (* PARA [14959]: Activates the grid status detection function to detect smooth transitions from grid parallel to island *)
		iSmooth_Isl_Det_Sensitiv : INT; (* PARA [14960]: Sensitivity of grid status detection function to detect smooth transitions from grid parallel to island *)
		bSelectiveBlocking_Enable : BOOL; (* PARA [14961]: Activates the function for selective blocking of grid status detection by grid events *)
		bBypassBlocking_Enable : BOOL; (* PARA [14962]: Activates the function for bypassing the grid event blocking of the grid status detection, if speed deviation exceeds limit *)
		iSensitivity_FRTBlocking : INT; (* PARA [14963]: Sensitivity of selective grid event blocking of grid status detection *)
		rU_Gen_ExcHi : REAL; (*PARA [11592]: excitation voltage high*)
		iSel_Customer : DINT; (*PARA [14950]: 0 = no special, 1 = AB Energy, 2 = Aggreko, 3 = 2G, etc.... *)
		rT_EG_Grad_HiHi : REAL; (*PARA[14964]: Exhaust gas temp. gradient deviation maximum [degC/s]*)
		rVol_Gas_EngInlet : REAL; (* PARA [15017]: Volume between gas valves and engine fuel gas inlet [l] *)
		bRKS_Active	: BOOL; (* PARA [15046]: Redundant Knock System Active with KLS *)
		iWG_Device_Type : USINT; (* PARA [15044]: Waste gate Actuator Type: 0-Default, 1-Analog, 2-CAN *)
		iWG_Device_Qty : USINT; (* PARA [15045]: Number of installed waste gate actuators *)
		rQ_UnderExc_Lim : REAL; (*PARA [13693]: reactive power limit underexcitated [p.u.]*) (*Oldname:newPv;Cycle:5;*)
		rQ_OverExc_Lim : REAL; (*PARA [13694]: reactive power limit overexcitated [p.u.]*) (*Oldname:newPv;Cycle:5;*)
		rS_Nom : REAL; (*PARA [11571]: Nominal Aparent Power (kVA)*)
		rLam_Start_Offset_H2 : REAL; (* PARA [15048]: Start lambda offset at 25% H2 content *)
		bEng_Act_H2 : BOOL; (* PARA [tbd]: H2 engine active *)
		rP_Act_Norm_Backfire : REAL; (* PARA [tbd]: Start Backfire control *)
		rP_Act_Norm_GlowIgn : REAL; (* PARA [tbd]: Start pre-ignition control *)
		rPr_CPP_DevLim_Prct : REAL; (* PARA [tbd]: Factor for pre-ignition detection with cylinder peak fire pressure *)
		rPr_49bfTDC_DevLim_Prct : REAL; (* PARA [tbd]: Factor for pre-ignition detection with p49bTDC *)
		rP_Act_Norm_SkipMax : REAL; (* PARA [tbd]: Switching point for allowed number of skipped cylinders *)
		iNum_CylSkip_Max_P1 : INT; (* PARA [tbd]: Max. allowed number of skipped cylinders due to backfire or pre-ignition below switching point *)
		iNum_CylSkip_Max_P2 : INT; (* PARA [tbd]: Max. allowed number of skipped cylinders due to backfire or pre-ignition after switching point *)
	END_STRUCT;
	tFS_P : 	STRUCT
		ti_Desired : TIME; (* desired time from demand to full load *)
		ti_VFS_Desired : TIME; (* desired time from demand to full load *)
		bLowTransNOx_Ena : BOOL; (* enable low transient NOx *)
		bFastSync : BOOL; (* enable fast synchronization *)
		bFastSpeedUp : BOOL; (* enable fast speed up *)
		tTime_before_SY : TIME; (*Minimum time from demand to synchronisation*)
		rT_delta_Idle_SY : REAL; (*Max. cylinder temperature when waitung in idle as difference to max. limit*)
		bTiStart5min : BOOL; (*5min Start without activated FastStart*)
	END_STRUCT;
	tPFPDR_P : 	STRUCT
		bEna : BOOL; (* Peak Fire Pressure Detection Run enabled? *)
		bAuto_Ena : BOOL; (* Automatic Peak Fire Pressure Detection Run enabled? *)
		iBH_Auto : DINT; (* Automatic Peak Fire Pressure Detection Run starts every x operating hours *)
		rLam_Lim : REAL; (* Maximum allowed lambda decrease during PFPDR *)
		rCA_Offs_Lim : REAL; (* Offset limit for PFPDR Profile (±from nominal timing) *)
		rCA_IP_EGT : REAL; (* Ignition point adaptation due EGT *)
		bAdv_IP_Ena : BOOL; (* advanced IP enabled? *)
		tiSS_Del : TIME; (* State Delay for PFPDR application *) (*OldName:newPv; Cycle:2;*)
	END_STRUCT;
	tSS_P : 	STRUCT
		T2s : tSS_SubPara;
		P2s : tSS_SubPara;
		P_Norm : tSS_SubPara;
		EGT : tSS_SubPara;
		Lam : tSS_SubPara;
		N_Norm : tSS_SubPara;
		P_d_Norm : tSS_SubPara;
		IP : tSS_SubPara;
	END_STRUCT;
	tSS_SubPara : 	STRUCT
		ti_Filt : TIME;
		rAbs : REAL;
		rRel : REAL;
	END_STRUCT;
	tSimPID_DS_typ : 	STRUCT
		ssMethodType : SINT;
		P : REAL; (*Proportional gain*)
		I : REAL; (*Integral gain*)
		wxmin : LREAL; (*minimum input*)
		deadband : LREAL; (*deadband*)
		D : REAL; (*Derivative gain*)
		N : REAL; (*Filter number*)
		umax : REAL; (*Upper saturation level*)
		umin : REAL; (*Lower saturation level*)
		Kt : REAL; (*Tracking Gain*)
		wxmax : LREAL; (*maximum input*)
		mode : USINT; (*Manual*)
		u_man : REAL; (*Manual Value*)
		a : REAL; (*feed forward*)
		invert : BOOL; (*invert*)
		w : REAL; (*reference*)
		x : REAL; (*control variable*)
		reset : BOOL; (*Reset bit*)
		I0 : REAL; (*Integrator value at reset*)
		D0 : REAL; (*Filter value at reset*)
		u : REAL; (*Controller output*)
		up : REAL; (*proportional output*)
		ui : REAL; (*integral output*)
		ud : REAL; (*differential output*)
		u_tr : REAL; (*tracking output*)
		fbk_mode : USINT; (*Anti Windup Feedback Mode*)
		u_fbk : REAL; (*External Anti Windup Feedback*)
	END_STRUCT;
	_tMeasurePoint : 	STRUCT
		P : INT;
		t : REAL;
		w : INT;
		n : INT;
	END_STRUCT;
	_tLinear : 	STRUCT
		x1 : INT;
		y1 : INT;
		x2 : INT;
		y2 : INT;
	END_STRUCT;
	_tRLinear : 	STRUCT
		x1 : REAL;
		y1 : REAL;
		x2 : REAL;
		y2 : REAL;
	END_STRUCT;
	alarmP : 	STRUCT
		ENABLE : BOOL;
		SET : BOOL;
		PTON : TIME;
		RESET : BOOL;
		PRIO : INT;
		TEST : BOOL;
		Q : BOOL;
	END_STRUCT;
	tABMW_time : 	STRUCT
		time : ARRAY[0..2]OF UINT;
	END_STRUCT;
	MM2VIS_Struct : 	STRUCT  (*OPC variables from module to VIS*)
		bMsg1044 : BOOL; (* Trip: Cylinder exhaust gas temperature deviation from average value *) (* OldName: new PV; Cycle: 0 *)
		bMsg1047 : BOOL; (* Trip: Misfiring failure *) (* OldName: AUSS_A; Cycle: 0 *)
		bMsg1049 : BOOL; (* Trip: Cylinder exhaust gas temperature absolute value high *) (* OldName: new PV; Cycle: 0 *)
		bMsg1080 : BOOL; (* Trip: LEANOX controller allowed deviation exceeded *) (* OldName: new PV; Cycle: 0 *)
		bMsg2294 : BOOL; (* Trip: Lambda limit exceeded*) (* OldName: new PV; Cycle: 0 *)
		bMsg1153 : BOOL; (* Trip: Cylinder exhaust gas temperature measuring signal failure *) (* OldName: new PV; Cycle: 0 *)
		bMsg2061 : BOOL; (* Trip: Cylinder 1 exhaust gas temperature measuring signal failure *) (* OldName: new PV; Cycle: 0 *)
		bMsg2062 : BOOL; (* Trip: Cylinder 2 exhaust gas temperature measuring signal failure *) (* OldName: new PV; Cycle: 0 *)
		bMsg2063 : BOOL; (* Trip: Cylinder 3 exhaust gas temperature measuring signal failure *) (* OldName: new PV; Cycle: 0 *)
		bMsg2064 : BOOL; (* Trip: Cylinder 4 exhaust gas temperature measuring signal failure *) (* OldName: new PV; Cycle: 0 *)
		bMsg2065 : BOOL; (* Trip: Cylinder 5 exhaust gas temperature measuring signal failure *) (* OldName: new PV; Cycle: 0 *)
		bMsg2066 : BOOL; (* Trip: Cylinder 6 exhaust gas temperature measuring signal failure *) (* OldName: new PV; Cycle: 0 *)
		bMsg2067 : BOOL; (* Trip: Cylinder 7 exhaust gas temperature measuring signal failure *) (* OldName: new PV; Cycle: 0 *)
		bMsg2068 : BOOL; (* Trip: Cylinder 8 exhaust gas temperature measuring signal failure *) (* OldName: new PV; Cycle: 0 *)
		bMsg2069 : BOOL; (* Trip: Cylinder 9 exhaust gas temperature measuring signal failure *) (* OldName: new PV; Cycle: 0 *)
		bMsg2070 : BOOL; (* Trip: Cylinder 10 exhaust gas temperature measuring signal failure *) (* OldName: new PV; Cycle: 0 *)
		bMsg2071 : BOOL; (* Trip: Cylinder 11 exhaust gas temperature measuring signal failure *) (* OldName: new PV; Cycle: 0 *)
		bMsg2072 : BOOL; (* Trip: Cylinder 12 exhaust gas temperature measuring signal failure *) (* OldName: new PV; Cycle: 0 *)
		bMsg2073 : BOOL; (* Trip: Cylinder 13 exhaust gas temperature measuring signal failure *) (* OldName: new PV; Cycle: 0 *)
		bMsg2074 : BOOL; (* Trip: Cylinder 14 exhaust gas temperature measuring signal failure *) (* OldName: new PV; Cycle: 0 *)
		bMsg2075 : BOOL; (* Trip: Cylinder 15 exhaust gas temperature measuring signal failure *) (* OldName: new PV; Cycle: 0 *)
		bMsg2076 : BOOL; (* Trip: Cylinder 16 exhaust gas temperature measuring signal failure *) (* OldName: new PV; Cycle: 0 *)
		bMsg2077 : BOOL; (* Trip: Cylinder 17 exhaust gas temperature measuring signal failure *) (* OldName: new PV; Cycle: 0 *)
		bMsg2078 : BOOL; (* Trip: Cylinder 18 exhaust gas temperature measuring signal failure *) (* OldName: new PV; Cycle: 0 *)
		bMsg2079 : BOOL; (* Trip: Cylinder 19 exhaust gas temperature measuring signal failure *) (* OldName: new PV; Cycle: 0 *)
		bMsg2080 : BOOL; (* Trip: Cylinder 20 exhaust gas temperature measuring signal failure *) (* OldName: new PV; Cycle: 0 *)
		bMsg2339 : BOOL; (* Trip: Exhaust gas temperature inclination maximum at cylinder head*)
		bMsg3217 : BOOL; (* Warning: Misfiring failure *) (* OldName: new PV; Cycle: 0 *)
		bMsg3238 : BOOL; (* OP Message: Positive deviation of cylinder x from average high *) (* OldName: new PV; Cycle: 0 *)
		bMsg3239 : BOOL; (* OP Message: Negative deviation of cylinder x from average high *) (* OldName: new PV; Cycle: 0 *)
		bMsg3285 : BOOL; (* OP Message: exh. gas temp. measuring signal failure *) (* OldName: new PV; Cycle: 0 *)
		bMsg3295 : BOOL; (* OP Message: max. exhaust temperature *) (* OldName: new PV; Cycle: 0 *)
		bMsg3408 : BOOL; (* Warning: Cylinder exhaust gas temperature positive deviation from average value *) (* OldName: new PV; Cycle: 0 *)
		bMsg3409 : BOOL; (* Warning: Cylinder exhaust gas temperature negative deviation from average value *) (* OldName: new PV; Cycle: 0 *)
		bMsg3542 : BOOL; (* Warning:  Cylinder exhaust gas temperature measuring signal failure *) (* OldName: new PV; Cycle: 0 *)
		bMsg3212 : BOOL; (* Warning: Fuel gas volume too high *) (* OldName: TJ_GASO; Cycle: 0 *)
		bMsg3248 : BOOL; (* OP Message: TECJET fuel gas volume high *) (* OldName: TJ_GASO_B; Cycle: 0 *)
		iMsg3248 : INT; (* ACM:  TECJET fuel gas volume high *) (* OldName: ucTJ_GASO; Cycle: 0 *)
		bMsg3099 : BOOL; (* Trip: Step of fuel gas volume too high *) (* OldName: TJ_GASM; Cycle: 0 *)
		bMsg3247 : BOOL; (* OP Message: TECJET Step of fuel gas volume too high *) (* OldName: TJ_GASM_B; Cycle: 0 *)
		iMsg3247 : INT; (* ACM: TECJET step of gas volume high *) (* OldName: ucTJ_GASM; Cycle: 0 *)
		bMsg2084 : BOOL; (* Warning: LEANOX algorithm failure *) (* OldName: RPSW[3]; Cycle: 0 *)
		bMsg1192 : BOOL; (* Warning: Throttle valve failure *) (* OldName: ST_ACT; Cycle: 0 *)
		bMsg2514 : BOOL; (* Warning: Actuator failure throttle valve A 1 *) (* OldName: DI_F_ACT_TV1A; Cycle: 0 *)
		bMsg2515 : BOOL; (* Warning: Actuator failure throttle valve B 1 *) (* OldName: DI_F_ACT_TV1B; Cycle: 0 *)
		bMsg2516 : BOOL; (* Warning: Actuator failure throttle valve A 2 *) (* OldName: DI_F_ACT_TV2A; Cycle: 0 *)
		bMsg2517 : BOOL; (* Warning: Actuator failure throttle valve B 2 *) (* OldName: DI_F_ACT_TV2B; Cycle: 0 *)
		bMsg9246 : BOOL; (* Warning: Actuator failure waste gate valve *)
		bMsg2522 : BOOL; (* Warning: Actuator failure waste gate valve A *) (* OldName: DI_F_ACT_EGBV_A; Cycle: 0 *)
		bMsg2523 : BOOL; (* Warning: Actuator failure waste gate valve B *) (* OldName: DI_F_ACT_EGBV_B; Cycle: 0 *)
		bMisfSend : BOOL; (* TRUE =send misfire CAN message *) (* OldName: 0; Cycle: 2 *)
		rP_Red_Knck_Norm : REAL; (* power reduction by knocking *) (* OldName: 0; Cycle: 2 *)
		rP_Red_Misf_Norm : REAL; (* power reduction by misfire *) (* OldName: 0; Cycle: 2 *)
		rP_Red_EGT_Norm : REAL; (* power reduction by exhaust gas temp. *) (* OldName: 0; Cycle: 2 *)
		rPos_TV : REAL; (* throttle valve position *) (* OldName: rPos_TV; Cycle: 2 *)
		rPos_Set_TV_A1 : REAL; (* setpoint throttle valve position A1 *) (* OldName: rPos_TV_A1; Cycle: 2 *)
		rPos_Set_TV_A2 : REAL; (* setpoint throttle valve position A2 *) (* OldName: rPos_TV_A2; Cycle: 2 *)
		rPos_Set_TV_B1 : REAL; (* setpoint throttle valve position B1 *) (* OldName: rPos_TV_B1; Cycle: 2 *)
		rPos_Set_TV_B2 : REAL; (* setpoint throttle valve position B2 *) (* OldName: rPos_TV_B2; Cycle: 2 *)
		rPos_Act_TV : REAL; (* actual position throttle valve position *) (* OldName: rPos_TV; Cycle: 2 *)
		rPos_Act_TV_A1 : REAL; (* actual position throttle valve position A1 *) (* OldName: rPos_TV_A1; Cycle: 2 *)
		rPos_Act_TV_A2 : REAL; (* actual position throttle valve position A2 *) (* OldName: rPos_TV_A2; Cycle: 2 *)
		rPos_Act_TV_B1 : REAL; (* actual position throttle valve position B1 *) (* OldName: rPos_TV_B1; Cycle: 2 *)
		rPos_Act_TV_B2 : REAL; (* actual position throttle valve position B2 *) (* OldName: rPos_TV_B2; Cycle: 2 *)
		rPos_CBV : REAL; (* compressor bypass valve position *) (* OldName: rPos_CBV; Cycle: 2 *)
		rPos_Set_CBV_A1 : REAL; (* setpoint compressor bypass valve position A1 *) (* OldName: rPos_CBV_A1; Cycle: 2 *)
		rPos_Set_CBV_A2 : REAL; (* setpoint compressor bypass valve position A2 *) (* OldName: rPos_CBV_A2; Cycle: 2 *)
		rPos_Set_CBV_B1 : REAL; (* setpoint compressor bypass valve position B1 *) (* OldName: rPos_CBV_B1; Cycle: 2 *)
		rPos_Set_CBV_B2 : REAL; (* setpoint compressor bypass valve position B2 *) (* OldName: rPos_CBV_B2; Cycle: 2 *)
		rPos_Act_CBV_A1 : REAL; (* actual position compressor bypass valve position A1 *) (* OldName: rPos_CBV_A1; Cycle: 2 *)
		rPos_Act_CBV_A2 : REAL; (* actual position compressor bypass valve position A2 *) (* OldName: rPos_CBV_A2; Cycle: 2 *)
		rPos_Act_CBV_B1 : REAL; (* actual position compressor bypass valve position B1 *) (* OldName: rPos_CBV_B1; Cycle: 2 *)
		rPos_Act_CBV_B2 : REAL; (* actual position compressor bypass valve position B2 *) (* OldName: rPos_CBV_B2; Cycle: 2 *)
		bMisfCOn : BOOL; (* Misfire Command On *) (* OldName: 0; Cycle: 2 *)
		rRatioMix : REAL; (* gas mixture rate after ramp fub *) (* OldName: 0; Cycle: 2 *)
		ulGasFlowN : ARRAY[0..4]OF UDINT; (* setpoint gasflow one gas inject valve *) (* OldName: ulGasFlowN; Cycle: 2 *)
		rPos_GM_Set_Norm : REAL; (* set point for the gasmixer *) (* OldName: ssPosGasmixerNominal / bp_y; Cycle: 2 *)
		rLam_Eng_LL_Set : REAL; (* Leanox Lambda set point *) (* OldName: ssPosGasmixerNominal / bp_y; Cycle: 2 *)
		rPos_Eng_Gm_Stepper_Set : REAL; (* rated gasmixer position *) (* OldName: usStepperRatedPos; Cycle: 2 *)
		rCA_IgnP_Set : REAL; (* ignitoin timing set point *) (* OldName: W_ZZP ; Cycle: 2 *)
		bIP_Red_Reset : BOOL; (* reset of the  ignitoin timing set point reduction *) (* OldName: bResetTimingRed ; Cycle: 2 *)
		rT_EG_Min : REAL; (* cylinder temperature minimal value [deg.C] *) (* OldName: ZYL_MIN; Cycle: 2 *)
		rT_EG_Avg : REAL; (* cylinder temperature average [deg.C] *) (* OldName: ZYL_AV; Cycle: 2 *)
		rT_EG_Max : REAL; (* cylinder temperature maximal value [deg.C] *) (* OldName: ZYL_MAX; Cycle: 2 *)
		iNum_Msg3238 : INT; (* Cylinder information for the message 3238 *) (* OldName: ucZylABMWP; Cycle: 2 *)
		iNum_Msg3239 : INT; (* Cylinder information for the message 3239 *) (* OldName: ucZylABMWN; Cycle: 2 *)
		iNum_Msg3285 : INT; (* Cylinder information for the message 3285 *) (* OldName: ucZylMSAGT; Cycle: 2 *)
		iNum_Msg3295 : INT; (* Cylinder information for the message 3295 *) (* OldName: ucZylATMA; Cycle: 2 *)
		tActuator_Rel : HALioDo_Type; (* DO: Actuator release command *) (* OldName: ACTUATOR; Cycle: 2 *)
		bSCO_Active : BOOL; (* safety cut out gas valves glow ignition prevention *) (* OldName: SICH_SCHL; Cycle: 5 *)
		rT_EPU_EG : ARRAY[0..24]OF REAL; (* engine power unit exhaust gas temperatures *) (* OldName: t_zyl; Cycle: 2 *)
		rP_Red_Leanox_Norm : REAL; (* power reduction by leanox *) (* OldName: leanox_dp; Cycle: 2 *)
		bMsg3583 : BOOL; (* Warning: Cylinder exhaust gas temperature absolute value high *) (* OldName: 0; Cycle: 0 *)
		bMsg3584 : BOOL; (* Warning: Cylinder exhaust gas temperature deviation from average value *) (* OldName: 0; Cycle: 0 *)
		bMsg3564 : BOOL; (*  Warning: Actuator compressor bypass valves *) (* OldName: 0; Cycle: 0 *)
		bLeanox_Active : BOOL; (* TRUE = leanox controller is active *) (* OldName: bLeanoxActive; Cycle: 2 *)
		rPr_Leanox_Dev : REAL; (* leanox controller deviation [bar] *) (* OldName: ssPressLeanoxError; Cycle: 2 *)
		rP_Power_Dev : REAL; (* power controller deviation [kW] *) (* OldName: new PV; Cycle: 2 *)
		rN_Speed_Dev : REAL; (* speed controller deviation [rpm] *) (* OldName: new PV; Cycle: 2 *)
		rMisf_Intgr : REAL; (* integrator electrical misfires [0..1] *) (* OldName: ssMisfInt; Cycle: 2 *)
		bMisf_Blink : BOOL; (* 0 *) (* OldName: bMisfBlink; Cycle: 0 *)
		bMsg2165 : BOOL; (* B2165 Power limitation by air humidity - low limit *) (* OldName: new PV; Cycle: 0 *)
		bMsg2166 : BOOL; (* B2166 Air humidity charge temperature offset active *) (* OldName: new PV; Cycle: 0 *)
		rT_AirIn : REAL; (* Intake air temperature *)
		rHum_AirIn_Rel : REAL; (* Intake air humidity relative *)
		rHum_AirIn_Abs : REAL; (* Intake air humidity absolute (calculated) *)
		rPr_Eng_P2s_SetMax_filt : REAL; (* charge pressure maximum *)
		rPr_Eng_P2s_Filt : REAL; (* charge pressure *)
		rT_T2_HumOffset : REAL; (* charge temperature offset *)
		rP_Red_Hum_Norm : REAL; (* power reduction humidity [kW] *)
		bECS_Speed : BOOL; (* engine controller state: Speed *)
		bECS_Idle : BOOL; (* engine controller state: Idle *)
		bECS_Power : BOOL; (* engine controller state: Power *)
		rT_T2_Set : REAL; (* setpoint charge temperature *) (* OldName: W_LLTP; Cycle: 0 *)
		rCA_IgnP_Nom : REAL; (* nominal ignition timing set point *) (* OldName: W_ZZPRoh; Cycle: 0 *)
		rPos_Set_WG : REAL; (* waste gate valve position *)
		rPos_Set_WG_A : REAL; (* waste gate valve position A *) (* OldName: ssPos_WG; Cycle:2; *)
		rPos_Set_WG_B : REAL; (* waste gate valve position B *) (* OldName: ssPos_WG; Cycle:2; *)
		rPos_Act_WG : REAL; (* waste gate valve position *)
		rPos_Act_WG_A : REAL; (* waste gate valve position A *) (* OldName: AI_WasteGate_y_Ist_A; Cycle:2; *)
		rPos_Act_WG_B : REAL; (* waste gate valve position B *) (* OldName: AI_WasteGate_y_Ist_A; Cycle:2; *)
		bMsg2328 : BOOL; (*Trip: wastegate measuring signal failure*)
		bMsg3371 : BOOL; (*Trip: wastegate bank A measuring signal failure*)
		bMsg3372 : BOOL; (*Trip: wastegate bank B measuring signal failure*)
		bMsg2329 : BOOL; (*Trip: wastegate set to actual value deviation to high*)
		bMsg3373 : BOOL; (*Trip: wastegate bank A set to actual value deviation to high*)
		bMsg3374 : BOOL; (*Trip: wastegate bank B set to actual value deviation to high*)
		bMsg9392 : BOOL; (*W9392 CAN wastegate bank A actuator failure*)
		bMsg9393 : BOOL; (*W9393 CAN wastegate bank B actuator failure*)
		bMsg9394 : BOOL; (*W9394 CAN wastegate bank A system warning*)
		bMsg9395 : BOOL; (*W9395 CAN wastegate bank B system warning*)
		bMsg2380 : BOOL; (*A2380 CAN wastegate bank A CAN Communication Error*)
		bMsg2381 : BOOL; (*A2381 CAN wastegate bank B CAN Communication Error*)
		bMsg2831 : BOOL; (* B2831 Low Voltage Ride Through Event *)
		bMsg2832 : BOOL; (* B2832 Mains failure + Generator Pole slip *)
		bMsg2833 : BOOL; (* B2833 Mains failure + dynamic rotor angle maximum *)
		bMsg2834 : BOOL; (* B2834 Mains failure + static rotor angle maximum *)
		bMsg2835 : BOOL; (* B2835 Mains failure + leading power factor operation *)
		bMsg2836 : BOOL; (* B2836 Mains failure maintenance request, reserve *)
		bMsg2837 : BOOL; (* B2837 Mains failure + dynamic rotor angle minimum *)
		bMsg2838 : BOOL; (* B2838 Mains failure + electric power to low *)
		bMsg2839 : BOOL; (* B2839 x *)
		bMsg2840 : BOOL; (* B2840 x *)
		bMsg3586 : BOOL; (*Warning: Mains failure maintenance request *)
		bMsg2852 : BOOL; (* B2852 - Turbolader Pumpen*)
		bMsg2141 : BOOL; (* B2141 ignition point reduction by by knocking (diagn.msg RPS) *)
		iMsg3238 : INT; (*ACM: positive deviation from average*)
		iMsg3239 : INT; (*ACM: negative deviation from average*)
		iMsg3285 : INT; (*ACM: sensor fault*)
		iMsg3295 : INT; (*ACM: max. temperature*)
		bMsg2765 : BOOL; (* warning: PI optimizer opening duration offset in limitation *)
		bMsg9373 : BOOL; (* warning: PI-Optimization not allowed *)
		bMsg3268 : BOOL; (* operating message: PI optimizer opening duration offset in limitation *)
		iMsg3268 : INT; (* cylinder number of PI optimizer opening duration offset in limitation *)
		bMsg9078 : BOOL; (* operating message: PI-Optimization not allowed *)
		iMsg9078 : INT; (* cylinder number that blocks the PI-Optimization *)
		ParaEC : Gtyp_Struct;
		rTV_QC : REAL; (*quality criteria throttle valve noise *) (* OldName: d_dk_krit; Cycle:2; *)
		rCBV_QC : REAL; (*quality criteria compressor bypass valve noise *) (* OldName: d_ub_krit; Cycle:2; *)
		rEng_N_QC : REAL; (*quality criteria engine speed noise *) (* OldName: d_n_krit; Cycle:2; *)
		bMsg2841 : BOOL; (* B2841 Emergency shutdown on gas valves 		*)
		bMsg2842 : BOOL; (* B2842 Blocking of emergency shutdown 1 ON 	*)
		bMsg2843 : BOOL; (* B2843 Blocking of emergency shutdown 1 OFF 	*)
		bMsg2844 : BOOL; (* B2844 Blocking of emergency shutdown 2 ON 	*)
		bMsg2845 : BOOL; (* B2845 Blocking of emergency shutdown 2 OFF 	*)
		bMsg2846 : BOOL; (* B2846 Fast power reduction due to auto-ignition *)
		bMsg3585 : BOOL; (* W3585 Auto-ignition rate exceeded *)
		bMsg3529 : BOOL; (* W3529 Blockierung für x[min] nach 30min Betrieb (Sondergas) *)
		bMsg3348 : BOOL; (* A3348 Glow ignition failure *)
		bMsg2283 : BOOL; (* A2283 Backfire prevention *)
		bHiContrCyl : ARRAY[0..24]OF BOOL; (* HiCtr interference on cylinder *) (* OldName: bHiContrCyl; Cycle: 2 *)
		bLimpHomeCyl : ARRAY[0..24]OF BOOL; (* Cylinder in Limp Home *) (* OldName: bLimpHomeCyl; Cycle: 2 *)
		bLimpHomeCylTrip : ARRAY[0..24]OF BOOL; (* Cylinder Trip because Limp Home *) (* OldName: bLimpHomeCylTrip; Cycle: 2 *)
		bSkipCylAct : ARRAY[0..24]OF BOOL; (* Cylinder is skipfiring *) (* OldName: new PV; Cycle:2; *)
		bPI_Bal_Required : BOOL; (* Balancing Required *) (* OldName: bBalRequired; Cycle: 2 *)
		bPI_Opt_Done : BOOL; (* balancing for current load point is done *)
		bPI_Opt_Locked : BOOL; (* balancing for current load point is locked *)
		bPI_Bal_SteadyState : BOOL; (* Steady State  *) (* OldName: bSteadyState; Cycle: 2 *)
		bAut_Opt_Ena : BOOL; (* enable automatic optimization *)
		iIdx_PI_Bal_State : USINT; (* State of Balancer *) (* OldName: ucBal_State; Cycle: 2 *)
		iNum_Msg2814 : INT; (* Cylinder information for the message 2814 *) (* OldName: new PV; Cycle: 2 *)
		bMsg2814 : BOOL; (* B2814: Port Injection duration is too high *) (* OldName: new PV; Cycle: 2 *)
		bMsg9216 : BOOL; (* W9216: Port Injection opening duration is too high *) (* OldName: new PV; Cycle: 2 *)
		bMsg2287 : BOOL; (* A2287: Shutdown by hierarchic controller *) (* OldName: new PV; Cycle: 2 *)
		iNum_Msg2874 : INT; (* Cylinder information for the message 2874*) (* OldName: new PV; Cycle: 2 *)
		bMsg2874 : BOOL; (* B2874 Safety layer sensor failure *) (* OldName: new PV; Cycle: 2 *)
		bMsg2290 : BOOL; (* A2290 Safety layer sensor failure *) (* OldName: new PV; Cycle: 2 *)
		bMsg2262 : BOOL; (* A2262 Cylinder peak pressure high *)
		bMsg2274 : BOOL; (* A2274 Maximum positive deviation of average cylinder peak pressure *)
		bMsg2282 : BOOL; (* A2282 Average cylinder peak pressure maximum *)
		bMsg2808 : BOOL; (* B2808 Maximum positive deviation of average cylinder peak pressure *)
		iNum_Msg2808 : INT; (* B2808 Maximum positive deviation of average cylinder peak pressure *)
		bMsg2826 : BOOL; (* B2826 Cylinder peak pressure high *)
		iNum_Msg2826 : INT; (* B2826 Cylinder peak pressure high *)
		bMsg2588 : BOOL; (* W2588 Cylinder peak pressure high Warning*)
		bMsg2825 : BOOL; (* B2825 Cylinder peak pressure high Warning*)
		iNum_Msg2825 : INT; (* B2825 Cylinder peak pressure high Warning*)
		bMsg2145 : BOOL; (* B2145 Ignition point reduction PBC *)
		iNum_Msg2145 : INT; (* B2145 Cylinder Ignition point reduction PBC *)
		rPr_Knck_Max : REAL; (* Knock pressure maximum *) (* OldName: KlopfenMax; Cycle: 2 *)
		rPr_Knck_Min : REAL; (* Knock pressure minimum *) (* OldName: KlopfenMin; Cycle: 2 *)
		rPr_Knck_Avg : REAL; (* Knock pressure average *) (* OldName: KlopfenAvg; Cycle: 2 *)
		rPr_Knck : ARRAY[0..24]OF REAL; (* Knock pressure *) (* OldName: Klopfen; Cycle: 2 *)
		rPr_CPP_Min : REAL; (* cylinder peak pressure maximum *) (* OldName: PmaxMax; Cycle: 2 *)
		rPr_CPP_Max : REAL; (* cylinder peak pressure minimum *) (* OldName: PmaxMin; Cycle: 2 *)
		rPr_CPP_Avg : REAL; (* cylinder peak pressure average *) (* OldName: PmaxAvg; Cycle: 2 *)
		rPr_CPP : ARRAY[0..24]OF REAL; (* cylinder peak pressure *) (* OldName: DruckMax; Cycle: 2 *)
		rPr_IMEP_Min : REAL; (* Indicated mean pressure maximum *) (* OldName: PmiMax; Cycle: 2 *)
		rPr_IMEP_Max : REAL; (* Indicated mean pressure minimum *) (* OldName: PmiMin; Cycle: 2 *)
		rPr_IMEP_Avg : REAL; (* Indicated mean pressure average *) (* OldName: PmiAvg; Cycle: 2 *)
		rPr_IMEP : ARRAY[0..24]OF REAL; (* Indicated mean pressure *) (* OldName: IndiMiDr; Cycle: 2 *)
		rCA_MFBvar_Min : REAL; (* Mass factor burn 50% maximum *) (* OldName: PvarPMax; Cycle: 2 *)
		rCA_MFBvar_Set : REAL; (* Mass factor burn 50% setpoint*) (* OldName: PvarPMin; Cycle: 2 *)
		rCA_MFBvar_Median : REAL; (* Mass factor burn 50% median*) (* OldName: PvarPMin; Cycle: 2 *)
		rCA_MFBvar_Max : REAL; (* Mass factor burn 50% minimum *) (* OldName: PvarPMin; Cycle: 2 *)
		rCA_MFBvar_Avg : REAL; (* Mass factor burn 50% average *) (* OldName: PvarPAvg; Cycle: 2 *)
		rCA_MFBvar : ARRAY[0..24]OF REAL; (* Mass factor burn 50% *) (* OldName: UmsatzpunktL; Cycle: 2 *)
		rCA_PI_Dur_Min : REAL; (* Port Injection Duration minimum *) (* OldName: usDurationMin; Cycle: 2 *)
		rCA_PI_Dur_Max : REAL; (* Port Injection Duration maximum *) (* OldName: usDurationMax; Cycle: 2 *)
		rCA_PI_Dur_Avg : REAL; (* Port Injection Duration average *) (* OldName: usDurationAvg; Cycle: 2 *)
		rCA_PI_Dur : ARRAY[0..24]OF REAL; (* Port Injection Duration *) (* OldName: 0; Cycle: 2 *)
		rPr_Leanox_Set : REAL; (* Leanox P2' setpoint *) (* OldName: ss_p2s_leanox; Cycle: 2 *)
		iIdx_ContGen : INT; (*Controller generation 1=GEN1 (old version) / 2=GEN2 (Standard)*) (* Oldname: ucContGen; Cycle: 2 *)
		ti_Msg2876 : TIME; (* B2876 Misfire controller shutdown in X min *) (* Oldname: new PV; Cycle: *)
		bMsg2876 : BOOL; (* B2876 Misfire controller shutdown *) (* Oldname: new PV; Cycle: *)
		bMsg2583 : BOOL; (* W2583 Misfire controller shutdown *) (* Oldname: new PV; Cycle: *)
		bMsg2577 : BOOL; (* W2577 Cylinder pressure sensor measuring signal failure *)
		bMsg2802 : BOOL; (* B2802 Cylinder pressure sensor measuring signal failure*)
		iNum_Msg2802 : INT; (* B2802 Cylinder pressure sensor measuring signal failure*)
		bMsg3382 : BOOL; (* A3382 Abgastemperatur Abweichung vom Mittelwert *)
		bMsg2880 : BOOL; (* B2880 Cylinder exhaust gas temperature positive deviation from average value *)
		iNum_Msg2880 : INT; (* B2880 Cylinder exhaust gas temperature positive deviation from average value *)
		bMsg2970 : BOOL; (* B2970 Exhaust gas temperature inclination maximum at cylinder head*)
		iNum_Msg2970 : USINT; (* B2970 Exhaust gas temperature inclination maximum at cylinder head*)
		bMsg2881 : BOOL; (* B2881 Cylinder exhaust gas temperature negative deviation from average value *)
		iNum_Msg2881 : INT; (* B2881 Cylinder exhaust gas temperature negative deviation from average value *)
		bMsg2882 : BOOL; (* B2882 Balancer map deleted *)
		bMsg2883 : BOOL; (* B2883 Balancer map saved *)
		bMsg2849 : BOOL; (* B2849 Misfiring failure PBC *)
		iNum_Msg2849 : INT; (* B2849 Misfiring failure PBC *)
		bMsg2562 : BOOL; (* W2562 monitoring - Air humidity measuring signal failure *)
		bMsg2518 : BOOL; (* W2518: actuator failure turbo bypass valve HP A *)
		bMsg2519 : BOOL; (* W2519: actuator failure turbo bypass valve HP A 2, reserve *)
		bMsg2520 : BOOL; (* W2520: actuator failure turbo bypass valve HP B *)
		bMsg2521 : BOOL; (* W2521: actuator failure turbo bypass valve HP B 2, reserve *)
		iNum_SkipCyl_Act : INT; (* Skipped Cylinder by Engine Controller *) (* OldName: ssHiGlobEng_visSkipCylNr; Cycle:2; *)
		bMsg2894 : BOOL; (* B2894: Engine map is missing *)
		iNum_Msg2894 : INT; (* B2894: Engine map is missing *)
		bMsg9247 : BOOL; (* W3555: wastegate measuring signal failure*)
		bMsg3555 : BOOL; (* W3555: wastegate bank A measuring signal failure*)
		bMsg3556 : BOOL; (* W3556: wastegate bank B measuring signal failure*)
		rPr_49bfTDC_Min : REAL; (* In cylinder pressure 49deg. before TDC maximum *) (* OldName: new PV; Cycle: 2 *)
		rPr_49bfTDC_Max : REAL; (* In cylinder pressure 49deg. before TDC minimum *) (* OldName: new PV; Cycle: 2 *)
		rPr_49bfTDC_Avg : REAL; (* In cylinder pressure 49deg. before TDC average *) (* OldName: new PV; Cycle: 2 *)
		rPr_49bfTDC : ARRAY[0..24]OF REAL; (* In cylinder pressure 49deg. before TDC *) (* OldName: new PV; Cycle: 2 *)
		rCQ : ARRAY[0..24]OF REAL; (* Combustion Quality*) (* OldName: new PV; Cycle: 2 *)
		rCQ_Max : ARRAY[0..24]OF REAL; (* Combustion Quality*) (* OldName: new PV; Cycle: 2 *)
		bMsg2899 : BOOL; (* B2899: Fast start demanded - conditions not met *)
		bMsg2900 : BOOL; (* B2900: Fast start demanded - conditions met *)
		bMsg1293 : BOOL; (* B1293: Engine map automatically loaded *)
		iNum_Msg1293 : INT; (* B1293: Engine map automatically loaded *)
		bMsg9248 : BOOL; (* W3557: wastegate set - act deviation *)
		bMsg3557 : BOOL; (* W3557: wastegate bank A set - act deviation *)
		bMsg3558 : BOOL; (* W3558: wastegate bank B set - act deviation *)
		bType6_Update_Rel : BOOL; (* Enables Type6 Engine controls Update (100% Loadrejection, Island mode etc..) *) (*OldName:newPv; Cycle:5;*)
		bScavDone : BOOL; (* Scavanging done *)
		bT_EO_Ok : BOOL; (* Oil temp okay for fast start *)
		bT_ECW_Ok : BOOL; (* water temp okay for fast start *)
		rT_EGaHPTC : REAL; (* Temperature exhaust gas system *)
		rT_EG_LimMax : REAL; (* exhaust gas temperature limit *)
		rT_ECW_FS_Perm : REAL; (* minimum engine cooling water temperature for fast start *)
		rT_EO_FS_Perm : REAL; (* minimum engine oil temperature for fast start *)
		bFS_Req : BOOL; (* fast start required *)
		rOpt_Out : ARRAY[0..24]OF REAL; (* controller output from optimizer *)
		rOpt_Map : ARRAY[0..24]OF REAL; (* state of map *)
		rOpt_Out_Max : REAL; (* controller output from optimizer max *)
		rOpt_Out_Min : REAL; (* controller output from optimizer min *)
		rOpt_Out_Avg : REAL; (* controller output from optimizer average *)
		rOpt_Map_Max : REAL; (* state of map max *)
		rOpt_Map_Min : REAL; (* state of map min *)
		rOpt_Map_Avg : REAL; (* state of map average *)
		rOpt_Coef_a_Perm : REAL; (* Perm: factor a *)
		rOpt_Coef_b_Perm : REAL; (* Perm: factor b *)
		rOpt_CL_Hi_Perm : REAL; (* Perm: closed loop upper limit *)
		rOpt_CL_Lo_Perm : REAL; (* Perm: closed loop lower limit *)
		rOpt_PmaxOffset_UL_Perm : REAL; (* Perm: Pmax Offset upper limit *)
		rOpt_PmaxOffset_LL_Perm : REAL; (* Perm: Pmax Offset lower limit *)
		bP49_Source_Perm : BOOL; (* Perm: 0=Map, 1=Sensors *)
		rPr_P49_Map : ARRAY[0..24]OF REAL; (* Perm: P49 Map *)
		rPr_CPP_Targ : ARRAY[0..24]OF REAL; (* CPP target for optimizer*)
		rPr_CPP_Offs : ARRAY[0..24]OF REAL; (* CPP offset from p49 map/sensors*)
		rValue_L : REAL;
		rValue_D : REAL;
		rPr_Leanox_T2s : REAL;
		rPr_Leanox_Ign : REAL;
		rPr_Leanox_Hum : REAL;
		rLam_AbsLim : REAL;
		iLam_AbsLim : INT;
		iLam_ExtLim : INT;
		rLam_AIT_EOT : REAL;
		rLam_N_Offs : REAL;
		bMsg1294 : BOOL; (* B1294: performing WG check *)
		bMsg1299 : BOOL; (* B1299: optimizer map changed *)
		bMsg2187 : BOOL; (* B2187: Commissioning mode on *)
		bMsg2897 : BOOL; (* B2897: Boost pressure out of range*)
		bMsg2188 : BOOL; (* B2188: Commissioning mode off *)
		rTi_Targ : REAL; (* Time to reach target load *)
		bMsg2895 : BOOL; (* B2895: PFPDR started *)
		bMsg2896 : BOOL; (* B2896: PFPDR finished *)
		PFPDR : tPFPDR_MM2VIS; (* PFPDR MM2VIS structure *)
		bMsg2189 : BOOL; (* B2189: Lambda limit reached *)
		bNOx_Reached_Ena : BOOL; (* Show NOx Stuff *)
		bLamLimMisf : BOOL;
		rPos_Set_CBV_34 : REAL;
		rCoV100 : ARRAY[0..24]OF REAL; (*CoV [cylinder*)
		rCoV_Med : REAL;
		rCoV_min : REAL;
		rCoV_max : REAL;
		rCoV_Avg : REAL;
		rCoV_Set : REAL;
		rLam_min_GEN2 : REAL;
		rT_EG_Med : REAL; (*Exh Temp Median*)
		bdTExhMon_Act : BOOL; (*Valve fracture monitoring active - exhaust temperature*)
		iNum_Msg2846 : INT;
		bMsg2470 : BOOL; (* W2470: Cylinder IMEP deviation from average value *)
		bMsg2471 : BOOL; (* W2471: PI optimization required *)
		bMsg2929 : BOOL; (* B2929: Cylinder IMEP deviation from average value *)
		iNum_Msg2929 : INT; (* B2929: Cylinder IMEP deviation from average value *)
		bMsg2930 : BOOL; (* B2930: PI optimization required *)
		iNum_Msg2930 : INT; (* B2930: PI optimization required *)
		rPr_Baro_Hum : REAL; (* Barometric Pressure used for humidity functionality [bar] *)
		bMsg2487 : BOOL; (* W2487: Leanox adjustment recommend*)
		bMsg2488 : BOOL; (* W2488: Leanox adjusmtent mandatory*)
		bMsg2937 : BOOL; (* B2937: LEANOX new adjusted*)
		bMsg2938 : BOOL; (* B2938: Combustion chamber cleaning performed*)
		bFS_Ena : BOOL; (* Fast start enabled *)
		bMnsReturn : BOOL; (* Slow increase power ramp after mains failure not active *)
		rGen2_LamLim_Offset : REAL; (* automatic lambda map offset *)
		bMsg2962 : BOOL; (* B2962: Preparing for fast start *)
		bMsg2963 : BOOL; (* B2963: Preparing for very fast start *)
		bMsg2964 : BOOL; (* B2964: Ready for fast start *)
		bMsg2965 : BOOL; (* B2965: Ready for very fast start *)
		bMsg2966 : BOOL; (* B2966: Very fast start demanded - conditions not met *)
		bMsg2967 : BOOL; (* B2967: Very fast start demanded - conditions met *)
		bSS : BOOL; (*steady state for GEN2 control*)
		rPr_p2s_d : REAL; (*desired boost pressure in GEN2 control*)
		rPosTVmin : REAL; (*minimum throttle valve position in GEN2 control*)
		rErrModelGEN2 : REAL; (* indicator for model error of GEN2 island controller*)
		rLam_max_GEN2 : REAL;
		bGEN2_ParaBlocked : BOOL; (*TRUE = GEN2 Parameter nicht editierbar*)
		bMsg2960 : BOOL; (* B2960 Ignition point reduction by Cylinder Peak Pressure Integrator *)
		iNum_Msg2960 : INT; (* B2960 Cylinder Info - Ignition Point reduction by Cylinder Peak Pressure Integrator *)
		rPr_P2s_RefOffs_ESC : REAL; (*Offset for actual boost pressure reference value send to Gen2 controller to lean out and run on lower Nox levels (bar)*)
		rCA_IP_Offs_ESC : REAL; (*Offset for actual global ignition timing reference value send to IT controller to operate engine close to exhaust temperature limits for fast SCR heating during cold and warm start (CAD)*)
		bExistWasteGateSingle : BOOL; (* single flow waste gate existing *)
		bLX2_BPOC_measured : ARRAY[0..10]OF BOOL; (*LX2 BPOC - binary map of already measured points [true->measured]*)
		tiLX2_BPOC_UpdateTime : TIME; (*Update Time of BPOC [sec]*)
		tiLX2_Timer : TIME; (*Timer of Save Logic [sec]*)
		rPr_p2s_LX2 : REAL; (*LX2 boost pressure offset - delta p2s_LX2 [bar]*)
		rPr_p2s_BPOC_LX2 : REAL; (*interpolated delta_p2s from BPOC [bar]*)
		rPr_p2s_Ctrl_LX2 : REAL; (*Output of I-Controler [bar]*)
		bLX2_SS : BOOL; (*Engine in Steady State operation [true->SS]*)
		bLX2_BPOC_enable : BOOL; (*true, if BPOC is used to generate delta_p2s*)
		bLX2_Ctrl_enable : BOOL; (*true, if Controler is enabled*)
		bLX2_SaveBPOC_enable : BOOL; (*true, saveing is enabled*)
		bLX2_Leanox_Engine_Man : BOOL; (*Leanox OR Engine in Manual mode [true->manual mode]*)
		bLX2_Limit : BOOL; (*true, if LX2 is in Saturation*)
		bLX2_ESC : BOOL; (*ESC control active [true->ESC on]*)
		bLX2_active : BOOL; (*Leanox 2.0 active [true->active]*)
		rPr_LX2_BPOC_Y_ScalMin : REAL; (*Scaling minimum LX2*)
		rPr_LX2_BPOC_Y_ScalMax : REAL; (*Scaling maximum LX2*)
		rP_LX2_P_set : REAL; (*Power setpoint related to rP_Nom [%]*)
		rPr_LX2_BPOC : ARRAY[0..10]OF REAL; (*actual BPOC from Permanent Storage [bar]*)
		rPr_LX2_UpperLim : REAL;
		rPr_LX2_LowerLim : REAL;
		rPr_LX2_BPOC_gas1 : ARRAY[0..10]OF REAL; (*actual BPOC gas type 1 from Permanent Storage [bar]*)
		bLX2_BPOC_measured_gas1 : ARRAY[0..10]OF BOOL; (*LX2 BPOC gas type 1 - binary map of already measured points [true->measured]*)
		rPr_LX2_BPOC_gas2 : ARRAY[0..10]OF REAL; (*actual BPOC gas type 2 from Permanent Storage [bar]*)
		bLX2_BPOC_measured_gas2 : ARRAY[0..10]OF BOOL; (*LX2 BPOC gas type 2 - binary map of already measured points [true->measured]*)
		rPr_LX2_BPOC_gas3 : ARRAY[0..10]OF REAL; (*actual BPOC gas type 3 from Permanent Storage [bar]*)
		bLX2_BPOC_measured_gas3 : ARRAY[0..10]OF BOOL; (*LX2 BPOC gas type 3 - binary map of already measured points [true->measured]*)
		rPr_LX2_BPOC_gas4 : ARRAY[0..10]OF REAL; (*actual BPOC gas type 4 from Permanent Storage [bar]*)
		bLX2_BPOC_measured_gas4 : ARRAY[0..10]OF BOOL; (*LX2 BPOC gas type 4 - binary map of already measured points [true->measured]*)
		bMsg9253 : BOOL; (* Leanox 2 saturation - warning *)
		bMsg2986 : BOOL; (* Leanox 2 Active *)
		bMsg2987 : BOOL; (* Leanox 2 Not Active *)
		bMsg2988 : BOOL; (* Leanox 2 Map Reset *)
		bGEN2_Island_ParaBlocked : BOOL; (*TRUE = GEN2 Insel Parameter nicht editierbar*)
		bMsg9288 : BOOL; (* Measuring signal failure, temperature direct air injection *)
		bMsg9289 : BOOL; (* Measuring signal failure, pressure before direct air injection shut off valve  *)
		bMsg9290 : BOOL; (* Measuring signal failure, pressure before direct air injection control valve bank A *)
		bMsg9291 : BOOL; (* Measuring signal failure, pressure before direct air injection control valve bank B *)
		bMsg9292 : BOOL; (* Direct air injection shut off valve failure at closing *)
		bMsg9293 : BOOL; (* Direct air injection shut off valve failure at opening *)
		bMsg9294 : BOOL; (* Direct air injection circuit breaker tripped  *)
		bMsg9295 : BOOL; (* Direct air injection supply pressure below boost pressure *)
		bMsg9296 : BOOL; (* Direct air injection control valve bank A failure  *)
		bMsg9297 : BOOL; (* Direct air injection control valve bank B failure  *)
		bMsg9298 : BOOL; (* Direct air injection pressure before shut off valve high *)
		bMsg9299 : BOOL; (* Direct air injection failure *)
		bMsg9039 : BOOL; (* Direct air injection active *)
		bMsg9040 : BOOL; (* Direct air injection inactive *)
		bMsg9053 : BOOL; (* SCR inlet temperature controller active *)
		bMsg9054 : BOOL; (* SCR inlet temperature controller inactive *)
		rPr_DAI_In : REAL; (* DAI inlet pressure M.05-PI-002 *)
		rPr_DAI_A : REAL; (* DAI pressure control valve bank A M.05-PI-101 *)
		rPr_DAI_B : REAL; (* DAI pressure control valve bank B M.05-PI-201 *)
		rT_DAI : REAL; (* DAI temperature M.05-TI-003 *)
		bDAI_V_Opened : BOOL; (* DAI shut off valve opened M.05-YCS-001 *)
		bDAI_V_Close_Fault : BOOL; (* DAI shut off valve close fault M.05-YCS-001 *)
		bDAI_V_Open_Fault : BOOL; (* DAI shut off valve open fault M.05-YCS-001*)
		rPos_DAI_Act_A : REAL; (* Actual position DAI control valve bank A M.05-YCI-104 *)
		rPos_DAI_Set_A : REAL; (* Set position DAI control valve bank A M.05-YCI-104 *)
		rPos_DAI_Act_B : REAL; (* Actual position DAI control valve bank B M.05-YCI-204 *)
		rPos_DAI_Set_B : REAL; (* Set position DAI control valve bank B M.05-YCI-204 *)
		rFlow_Dem_DAI : REAL; (* Demanded mass flow DAI *)
		bTExhMon_vis : BOOL; (*Activation TExh Mon Para folder in HMI*)
		bMsg9312 : BOOL; (* W9312: Generator frequency too low in mains parallel operation *)
		bMsg9313 : BOOL; (* W9313: Generator frequency too high in mains parallel operation *)
		iCnt_PCGV_class1 : ARRAY[0..24]OF UINT; (*PCGV monitoring: class1 counter for sticking duration 1-10s*)
		iCnt_PCGV_class2 : ARRAY[0..24]OF UINT; (*PCGV monitoring: class2 counter for sticking duration 10-60s*)
		iCnt_PCGV_class3 : ARRAY[0..24]OF UINT; (*PCGV monitoring: class3 counter for sticking duration 60-300s*)
		iCnt_PCGV_class4 : ARRAY[0..24]OF UINT; (*PCGV monitoring: class4 counter for sticking duration 300-3600s*)
		rTi_PCGV_LastStickDur : REAL; (*Last PCGV sticking duration*)
		rTi_PCGV_MeanLastStickEvts : REAL; (*Sticking duration of last 10 PCGV sticking events*)
		bMsg9329 : BOOL; (* W9329: p2 sensor signal for GEN2 controller missing *)
		bMsg2975 : BOOL; (* B2975: Fast-Gas-Quality-Change-Function is running *)
		bMsg9047 : BOOL; (* OM9047: Target load reached*)
		rPr_P2sGen2_GasQualOffs : REAL; (* GEN2: boost pressure offset gas quality change [bar]*)
		bMsg9349 : BOOL; (* W9349: Grid Code FRT functionality contains wrong parameter *)
		bUseTVIdleControl : BOOL; (*TV control enabled*)
		bSav_LDat_P100_Disable : BOOL; (* Disable signal for HMI saving of Leanox reference point 1 *)
		bSav_LDat_P50_Disable : BOOL; (* Disable signal for HMI saving of Leanox reference point 2 *)
		bSav_LDat_P25_Disable : BOOL; (* Disable signal for HMI saving of Leanox reference point 3 *)
		rLam_PBC : REAL; (* Lambda estimated from in-cylinder pressure data *)
		rLam_LamCtrPBC_ref : REAL; (* Lambda reference for PI opening duration calculation *)
		rCA_TrStRed_LowLimit_Act : REAL; (* actual control limit TrStRed function - relative ITP [degCA] *)
		bTrStRed_PFPDR_dis : BOOL; (* PFPDR disable by TrStRed function *)
		bMsg9055 : BOOL; (* B9055: th. reactor start time reduction - operating cycle started *)
		bMsg9056 : BOOL; (* B9056: th. reactor start time reduction - operating cycle completed *)
		bMsg9065 : BOOL; (* B9065: Isolated operation - Grid status detection *)
		bMsg9068 : BOOL; (* B9068 Fault Ride Through Event in island operation *)
		rCA_IPOffs_SCRInTemp : REAL; (*SCR Inlet Temp IP Ctrl - Relative Offset IP*)
		bMsg9071 : BOOL; (* B9071 Low Voltage Ride Through Event simulated *)
		bTrStRed_pause_Disable : BOOL; (* Disable signal for temporary deactivation of TrStRed function from HMI *)
		bMsg2365 : BOOL; (* A2365: Generator pole slip*)
		rGT_H2_Mix : REAL; (* Hydrogen concentration volumetric for H2 compensation function after gas mixing *)
		rPr_Leanox_Offs_H2 : REAL; (* Boost pressure offset H2 content [bar] *)
		rCA_IgnP_Offs_H2 : REAL; (* ITP offset H2 content [deg.CA] *)
		bMsg2768 : BOOL; (* W2738: measuring signal failure gas humidity *)
		rHum_GasIn_Abs : REAL; (* absolute humidity gas via customer BUS [g H2O/kg dry gas] *)
		rHum_Mixture_Abs : REAL; (* absolute humidity mixture [g_H2O/kg_mix] *)
		bMsg9095 : BOOL; (* B9095: GEN2 lambda offset stopped *)
		bMsg9388 : BOOL; (*W9388 Combustion anomaly detection*)
		bMsg9092 : BOOL; (*B9092 Combustion anomaly detection*)
		iNum_Msg9092 : USINT; (*B9092 Combustion anomaly detection*)
		bMsg9407 : BOOL; (* A9407 - Maximum numbers of skipped cylinders exceeded *)
		iWG_CAN_B_SrcAdd : USINT; (*CAN wastegate actuator B source address*)
		iWG_CAN_A_SrcAdd : USINT; (*CAN wastegate actuator A source address*)
		iT_WG_CAN_B : INT;
		rPos_WG_CAN_B_Act : REAL;
		rPos_WG_CAN_B_Set : REAL;
		iSt_WG_CAN_B : USINT;
		iT_WG_CAN_A : INT;
		rPos_WG_CAN_A_Act : REAL;
		rPos_WG_CAN_A_Set : REAL;
		iSt_WG_CAN_A : USINT;
		bSt_WG_CAN_B_Warn : ARRAY[0..11]OF BOOL; (*CAN wastegate B warning information*)
		bSt_WG_CAN_B_Fail : ARRAY[0..4]OF BOOL; (*CAN wastegate B failure information *)
		bSt_WG_CAN_A_Warn : ARRAY[0..11]OF BOOL; (*CAN wastegate A warning information*)
		bSt_WG_CAN_A_Fail : ARRAY[0..4]OF BOOL; (*CAN wastegate A failure information *)
		bCANread_WG_B_Err : BOOL; (*CAN wastegate B communication error*)
		bCANread_WG_A_Err : BOOL; (*CAN wastegate A communication error*)
		iWG_CAN_A_OpH : UDINT := 0; (*CAN wastegate actuator bank A operating time [h]*)
		sWG_CAN_A_SN : STRING[10] := ''; (*CAN wastegate actuator bank A software version*)
		sWG_CAN_A_Sw : STRING[12] := ''; (*CAN wastegate actuator bank A serial number*)
		iWG_CAN_B_OpH : UDINT := 0; (*CAN wastegate actuator bank B operating time [h]*)
		sWG_CAN_B_SN : STRING[10] := ''; (*CAN wastegate actuator bank B software version*)
		sWG_CAN_B_Sw : STRING[12] := ''; (*CAN wastegate actuator bank B serial number*)
		bWG_CAN_B_Learn_On : BOOL := FALSE; (*CAN wastegate B learn state in process*)
		bWG_CAN_A_Learn_On : BOOL := FALSE; (*CAN wastegate A learn state in process*)
		bWG_CAN_B_Config_On : BOOL := FALSE; (* CAN wastegate B EEPROM configuration in progress*)
		bWG_CAN_A_Config_On : BOOL := FALSE; (* CAN wastegate A EEPROM configuration in progress*)
		bWG_CAN_A_LearnConfig_Dis : BOOL := FALSE; (*Disable CAN WG A buttons Learn and Configuration*)
		bWG_CAN_B_LearnConfig_Dis : BOOL := FALSE; (*Disable CAN WG B buttons Learn and Configuration*)
		bWG_CAN_Dem_Man_Dis : BOOL := FALSE; (*Disable CAN WG manual demand button for both banks*)
		bWG_CAN_A_Dem : BOOL := FALSE; (*Wastegate CAN A general demand*)
		bWG_CAN_B_Dem : BOOL := FALSE; (*Wastegate CAN B general demand*)
	END_STRUCT;
	tPFPDR_MM2VIS : 	STRUCT
		Data : tPFPDR_Data; (* Operating Data *)
		iNum_Prof : INT;
		rCA_IP_DR : ARRAY[0..24]OF REAL;
		rCA_IP_EGT : ARRAY[0..24]OF REAL;
		rCA_IP_Lim : ARRAY[0..24]OF REAL;
		iColor_Cyl : ARRAY[0..24]OF INT;
		rLam_Offs : REAL;
		rCA_IP_Offs : REAL;
		bEna : BOOL;
		bAuto_Ena : BOOL;
		bStart_Req : BOOL;
		bDR : BOOL;
		bEGT : BOOL;
		bSS : BOOL;
		rCA_Sum_Corr : REAL;
		iCnt_Prof : INT;
		rDone : REAL;
		iAutoStartHour : INT;
	END_STRUCT;
	VIS2MM_Struct : 	STRUCT  (*OPC variables from VIS to module*)
		rPos_Eng_Gm_ManSet : REAL; (* Gasmixer  manual set point *)
		rLam_Eng_LL_ManSet : REAL; (* Leanox Lambda manual set point *)
		bLeanox_Man : BOOL; (* TRUE = leanox controller in manual *) (* leanox *)
		bSav_LDat_P100 : BOOL; (* save data for Leanox at 100% nominal power *)
		bSav_LDat_P50 : BOOL; (* save data for Leanox at 50% nominal power *)
		bSav_LDat_P25 : BOOL; (* save data for Leanox at ~25% nominal power *)
		iCnt_TC_Surge : DINT; (* turbo charger surge counter --> opteration data *) (* OldName: ssTCSurge_Counter; Cycle:2; *)
		iCnt_GrCEvent : DINT; (* Counter for FRT event --> opteration data *) (* OldName: rCnt_GCEvent_GLOB; Cycle:2; *)
		bPI_Bal_Com : BOOL; (* Comissioning Balancer *) (* OldName: bComissioning_Bal; Cycle: 2 *)
		bPI_Bal_ResetMap : BOOL; (* Reset Duration Map *) (* OldName: bResetMap; Cycle: 2 *)
		bPI_Bal_Man_Req : BOOL; (* Request Manual Balancing *) (* OldName: ucReleaseBalancing; Cycle: 2 *)
		rPr_Leanox_Set_Man : REAL; (* Leanox P2' manual setpoint *) (* OldName: ss_p2s_cmd; Cycle: 2 *)
		rPos_TV_Man : REAL; (* Throttle valve manual setpoint *) (* OldName: new PV; Cycle: 2 *)
		rPos_CBV_Man_A : REAL; (* Compressor bypass valve manual setpoint bank A *) (* OldName: new PV; Cycle: 2 *)
		rPos_CBV_Man_B : REAL; (* Compressor bypass valve manual setpoint bank A *) (* OldName: new PV; Cycle: 2 *)
		bAct_Rel_Man : BOOL; (* Manual actuator valve release *) (* OldName: bManTBP; Cycle: 2 *)
		bRevPowTest : BOOL; (* Test bit for: reverse power *)
		bIP_Red_Reset : BOOL; (* reset of the  ignitoin timing set point reduction *) (* OldName: bResetTimingRed ; Cycle: 2 *)
		bCommMode : BOOL; (* Comm Mode for Engine Controller *)
		bSaveToPerm : BOOL; (* Comm Mode: saves adjustments to Perm *)
		bSave_P49_Map : BOOL; (* Comm Mode: save P49 Map to Perm *)
		bMapSave_Ena : BOOL; (* Comm Mode: enable optimizer map save *)
		bMFB50_On : BOOL; (* Comm Mode: enable MFB50 *)
		rOpt_Coef_a : REAL; (* Comm Mode: factor a *)
		rOpt_Coef_b : REAL; (* Comm Mode: factor b *)
		rOpt_Coef_b_IP : REAL; (* Comm Mode: factor b *)
		rOpt_Coef_c : REAL; (* Comm Mode: factor b *)
		rOpt_Coef_d : REAL; (* Comm Mode: factor d *)
		rOpt_Coef_e : REAL; (* Comm Mode: factor e *)
		rOpt_CL_Hi : REAL; (* Comm Mode: closed loop upper limit *)
		rOpt_CL_Lo : REAL; (* Comm Mode: closed loop lower limit *)
		rOpt_PmaxOffset_UL : REAL; (* Comm Mode: Pmax Offset upper limit *)
		rOpt_PmaxOffset_LL : REAL; (* Comm Mode: Pmax Offset lower limit *)
		bP49_Source : BOOL; (* Comm Mode: 0=Map, 1=Sensors *)
		rPr_P49_Set : ARRAY[0..24]OF REAL; (* Comm Mode: P49 Map *)
		bOpt_CPP_Offs_Set : ARRAY[0..24]OF BOOL; (* Comm Mode: Pmax offset overrule on*)
		rPr_CPP_Offs_Set : ARRAY[0..24]OF REAL; (* Comm Mode: Pmax offset overrule value*)
		PFPDR : tPFPDR_VIS2MM; (* PFPDR VIS2MM structure *)
		bMisfTest : BOOL;
		iCyl_MisfTest : USINT;
		bCompChamb_Clean : BOOL; (* VISU: button to be pressed after combustion chamber cleaning *)
		bLeanox_Adjust : BOOL; (* VISU: button to be pressed for confirmation of leanox adjustment *)
		bLX2_BPOC_reset : BOOL; (* VISU: button to be pressed for LX2 map reset request from HMI *)
		iCnt_DAI_Starts : UDINT; (* event counter for DAI starts --> operation data *)
		rCnt_DAI_Op_Min : REAL; (* minutes counter for DAI --> operation data*)
		rPos_DAI_Man_A : REAL; (* manual position DAI control valve bank A M.05-YCI-104 *)
		rPos_DAI_Man_B : REAL; (* manual position DAI control valve bank B M.05-YCI-204 *)
		bGrC_TestStart_Var : BOOL; (* Start FRT test with variable input *)
		bGrC_TestStart_150ms : BOOL; (* Start FRT test with duration of 150ms and 80ms ignition off *)
		bGrC_TestStart_250ms : BOOL; (* Start FRT test with duration of 250ms and 160ms ignition off *)
		iTime_GrC_Event : INT; (* Variable FRT event time for test *)
		iTime_GrC_IgnOff : INT; (* Variable FRT ignition off time for test *)
		bTrStRed_pause : BOOL; (* VISU: checkbox for temporary deactivation of TrStRed function *)
		iCnt_GrC_Event : DINT; (* Counter for unsuccessful FRT event --> opteration data *)
		bGrC_Confirmation : BOOL; (* FRT Confirmation Button *)
		bPI_Opt_Aut : BOOL; (* Automatic optimization for cylinder balancing is active *)
		bRKS_Mode : BOOL;
		bWG_CAN_B_Learn : BOOL; (*CAN wastegate B learn button *)
		bWG_CAN_A_Learn : BOOL; (*CAN wastegate A learn button *)
		bWG_CAN_B_Config : BOOL; (*CAN wastegate B configure bank address button*)
		bWG_CAN_A_Config : BOOL; (*CAN wastegate A configure bank address button*)
		bWG_CAN_A_Dem_Man : BOOL; (*CAN wastegate A manual demand button*)
		bWG_CAN_B_Dem_Man : BOOL; (*CAN wastegate B manual demand button*)
	END_STRUCT;
	tPFPDR_VIS2MM : 	STRUCT
		bStart : BOOL;
		bAbort : BOOL;
		bUp : BOOL;
		bDown : BOOL;
		bDel_Last : BOOL;
		bDel_All : BOOL;
		bShow_Act : BOOL;
	END_STRUCT;
	tPIopen : 	STRUCT
		timing : UINT;
		duration : UINT;
	END_STRUCT;
	rtctime_typ : 	STRUCT
		year : UINT;
		month : USINT;
		day : USINT;
		reserve : USINT;
		hour : USINT;
		minute : USINT;
		second : USINT;
		millisec : UINT;
		microsec : UINT;
	END_STRUCT;
	Map_Struct : 	STRUCT
		Type6 : Map_T6_Struct; (* Type6 Engine *)
		Type9 : Map_T9_Struct; (* Type9 Engine *)
		PFPDR : tPFPDR_Map; (* Peak Fire Pressure Detection Run *)
		LX2 : tLX2Map;
	END_STRUCT;
	Map_T9_Struct : 	STRUCT
		tPI_Duration_Map : ARRAY[0..24,0..15,0..10]OF REAL; (* Duration Map Data *) (* OldName: rDuraton_Map; Cycle: 2 *)
		bPI_Duration_Map : ARRAY[0..24,0..15,0..10]OF BOOL; (* Duration Map filled *) (* OldName: bFilledUp; Cycle: 2 *)
		tPI_p49_Map : ARRAY[0..24,0..15,0..10]OF REAL; (* p49 Map Data *) (* OldName: rDp49_Map; Cycle: 2 *)
		bPI_p49_Map : ARRAY[0..24,0..15,0..10]OF BOOL; (* p49 Map filled *) (* OldName: bFilledUp_p49; Cycle: 2 *)
	END_STRUCT;
	Map_T6_Struct : 	STRUCT
		xVE_MAP : MAP_REAL18; (* characterisitc map for volumetric efficiency *)
		Vers_VE_MAP : INT; (*Version of map for volumetric efficiency*)
	END_STRUCT;
	Cnt_Struct : 	STRUCT
		iCnt_TC_Surge : DINT; (* Cnt: Event Counter for turbo charger surge event *)
		iCnt_DAI_Starts : UDINT; (* Cnt: event counter for DAI starts *)
		rCnt_DAI_Op_Min : REAL; (* Cnt: operating minutes counter for DAI *)
		iCnt_GrCEvent : DINT; (* Cnt: Event Counter for grid code event *)
		iCnt_CPP_AvgEvent : ARRAY[0..24]OF UDINT; (* Cnt: Event Counter for cylinder peak pressure average reached *) (* OldName: ulPmaxAvgEventLifetime; Cycle: 2 *)
		iCnt_CPP_LimEvent : ARRAY[0..24]OF UDINT; (* Cnt: Event Counter for cylinder peak pressure limit reached *) (* OldName: new PV; Cycle: 2 *)
		iCnt_GrC_Event : DINT; (* Counter for unsuccessful FRT event *) (* OldName: ucGCEvent_Counter; Cycle:2; *)
	END_STRUCT;
	tPFPDR_Map : 	STRUCT
		iCnt : USINT; (* Counter for Ring Array *)
		tRun : ARRAY[0..9]OF tPFPDR_Run; (* Ring Array *)
	END_STRUCT;
	tPFPDR_Run : 	STRUCT
		bFilled : BOOL; (* Filled with data *)
		Data : tPFPDR_Data; (* Operating Data *)
		rCA_IP_DR_Prof : ARRAY[0..24]OF REAL; (* Ignition Offset by PFPDR *)
		rCA_IP_EGT_Prof : ARRAY[0..24]OF REAL; (* Ignition Offset by EGTSR *)
	END_STRUCT;
	tPFPDR_Data : 	STRUCT
		iOpHour : DINT; (* Operating Hours *)
		rP_Norm : REAL; (* actual load *)
		rPr_P2s : REAL; (* Charging pressure P2' *)
		rT_T2s : REAL; (* Charging temperature T2' *)
		rPr_P2 : REAL; (* Charging pressure P2 *)
		rN_TC : REAL; (* turbo charger speed *)
		rPos_TV : REAL; (* throttle valve position *)
		rPos_CBV : REAL; (* compressor bypass valve position *)
		rPos_WG : REAL; (* wastegate valve position *)
		rCA_IP_Set : REAL; (* global ignition point *)
		rT_AirIn : REAL; (* intake temperature *)
		rHum_Abs : REAL; (* intake humidity *)
		rL_Sealevel : REAL; (* sealevel *)
		rCA_IP_Act : ARRAY[0..24]OF REAL; (* actual ignition points *)
		rT_EG : ARRAY[0..24]OF REAL; (* actual exhaust gas temperatures *)
		rPr_CC : REAL; (* crank case pressure *)
		rPos_TJ : REAL; (* tecjet position *)
		rLam : REAL; (* lambda *)
		rCA_IP_Avg : REAL; (* average ignition point *)
	END_STRUCT;
	Perm_Struct : 	STRUCT
		MFB50 : tMFB50; (*Permanent Data for MFB50 Contr*)
		Opt : tOptimizer; (* Optimizer structure for pi_bal task *)
		Skip : tSkip; (* Skip structure for skip_zde task *)
		FS : tFastStart; (* Fast start structure *)
		PI : tPortInjection; (* port injection structure *)
		PUSL : tPUSL; (* power unit safety layer *)
		Gen1 : tGen1; (* Gen1 - old controller structure *)
		Gen2 : tGen2; (* Gen2 - new controller structure *)
		Filt : tFilter; (* all Filters *)
		WG : tWasteGate; (* Wastegate *)
		EG : tExhaustGas; (* Exhaust gas *)
		IG : tIgnition; (* Ignition *)
		Misc : tMisc; (* Miscellaneous *)
		RKS : tRKS_Perm; (* RKS with SAFI *)
		Sync : tSync_Perm;
		LEANOX_Drift : tLeanoxDrift;
		LX2 : tLX2_PERM;
		LX2_aux : tLX2_Perm_aux;
		Spare : tSparePerm_typ; (* Spare Parameter *)
		PCGVmon : tPCGVmon_PERM;
		DAI : DAI_Perm_Bus;
		SyncPrM : tFSyPrM_PERM;
		TrStRed : TrStRed_PERM_Bus;
	END_STRUCT;
	tIgnition : 	STRUCT
		rPnorm_ref_IP_P_x1 : REAL; (* normalized engine load reference for ITP interpolation end point *)
		refPoint_IP_N : ARRAY[0..2]OF lcrCurveByPoints_TabEntry_type;
		rPnorm_ref_IP_P_HC_x1 : REAL; (* normalized engine load reference for ITP interpolation point - J9 HC interim em. sol. *)
		rPnorm_ref_IP_P_HC_x2 : REAL; (* normalized engine load reference for ITP interpolation point - J9 HC interim em. sol. *)
		rCA_ref_IP_P_HC_y1 : REAL; (* ITP at intermediate load point - J9 HC interim em. sol.*)
	END_STRUCT;
	tRKS_Perm : 	STRUCT
		bEna : BOOL; (* Enables RKS Knock Control *)
		iTable : ARRAY[0..15]OF USINT; (* Logic Table *)
		rCA_IP_Red : REAL;
		rDur_Downset : REAL; (* Duration downset in [%] *)
		iNum_EngCyc_Limp_Recover : INT; (* amount of engine cycles without limphom to switch to PBC *)
	END_STRUCT;
	tMisc : 	STRUCT
		bNOx_Reached_Ena : BOOL; (* Show NOx Stuff *)
	END_STRUCT;
	tExhaustGas : 	STRUCT
		ti_Filt : TIME; (* Filter for EG Max, stock = 10s *)
		rP_LPR : REAL; (* Lower power range, stock = 0.4 *)
		rP_UPR : REAL; (* Upper power range, stock = 0.7 *)
		tiT_EG_LimMax : TIME; (* Time delay for A1049 *)
		iT_EG_HiHi : INT; (* trigger limit of A1049 without delay [K] *)
		iT_EG_Grad : INT; (* temp gradient to detect sensor failure [K/s] *)
		tiT_EG_LimMax_TrStRed : TIME; (* Extended time delay for A1049, while TrStRed function running *)
		iT_EG_HiHi_TrStRed : INT; (* trigger limit offset of A1049 without delay, while TrStRed function running  [K] *)
	END_STRUCT;
	tGen1 : 	STRUCT
		bType6_Update_Rel : BOOL; (* activates type6 controls update *)
		rLowerSyncPower : REAL;
		rLowerOilTemp : REAL;
		rHigherOilTemp : REAL;
		rLowerOilLambda : REAL;
		rHigherOilLambda : REAL;
		rLowerSyncLambda : REAL;
		rHigherSyncLambda : REAL;
		refPoint_Eta_Eng : ARRAY[0..9]OF lcrCurveByPoints_TabEntry_type; (* y = Eta Engine and x = pressure in [bar] *) (* OldName: InterP_Eta_Engine; Cycle: 2 *)
		refPoint_Eta_Gen : ARRAY[0..9]OF lcrCurveByPoints_TabEntry_type; (* y = Eta Generator and x = elec. power [kW] *) (* OldName: InterP_Eta_Gen; Cycle: 2 *)
		refPoint_CBV_FF_NetP : ARRAY[0..9]OF lcrCurveByPoints_TabEntry_type; (* y = CBV FF and x = power [kW] *)
		refPoint_CBV_FF_Island : ARRAY[0..9]OF lcrCurveByPoints_TabEntry_type; (* y = CBV FF and x = pressure in [bar] *)
		refPoint_FF_TV : ARRAY[0..9]OF lcrCurveByPoints_TabEntry_type;
		refPoint_TV_P_NetP : ARRAY[0..9]OF lcrCurveByPoints_TabEntry_type;
		refPoint_TV_I_NetP : ARRAY[0..9]OF lcrCurveByPoints_TabEntry_type;
		refPoint_TV_D_NetP : ARRAY[0..9]OF lcrCurveByPoints_TabEntry_type;
		refPoint_TV_N_NetP : ARRAY[0..9]OF lcrCurveByPoints_TabEntry_type;
		refPoint_FF_CBV : ARRAY[0..9]OF lcrCurveByPoints_TabEntry_type;
		refPoint_CBV_P_NetP : ARRAY[0..9]OF lcrCurveByPoints_TabEntry_type;
		refPoint_CBV_I_NetP : ARRAY[0..9]OF lcrCurveByPoints_TabEntry_type;
		refPoint_CBV_D_NetP : ARRAY[0..9]OF lcrCurveByPoints_TabEntry_type;
		refPoint_CBV_N_NetP : ARRAY[0..9]OF lcrCurveByPoints_TabEntry_type;
		refPoint_FF_LAMBDA : ARRAY[0..9]OF lcrCurveByPoints_TabEntry_type;
		refPoint_TV_P_Island : ARRAY[0..9]OF lcrCurveByPoints_TabEntry_type;
		refPoint_TV_I_Island : ARRAY[0..9]OF lcrCurveByPoints_TabEntry_type;
		refPoint_TV_D_Island : ARRAY[0..9]OF lcrCurveByPoints_TabEntry_type;
		refPoint_TV_N_Island : ARRAY[0..9]OF lcrCurveByPoints_TabEntry_type;
		refPoint_CBV_P_Island : ARRAY[0..9]OF lcrCurveByPoints_TabEntry_type;
		refPoint_CBV_I_Island : ARRAY[0..9]OF lcrCurveByPoints_TabEntry_type;
		refPoint_CBV_D_Island : ARRAY[0..9]OF lcrCurveByPoints_TabEntry_type;
		refPoint_CBV_N_Island : ARRAY[0..9]OF lcrCurveByPoints_TabEntry_type;
	END_STRUCT;
	tWasteGate : 	STRUCT
		rP_Rel_Norm : REAL; (* activation trigger value for the actual output of the waste gate control *) (* OldName: rP_IST_TRIG_WG; Cycle: 2 *)
		rGrad : REAL; (* gradient for increase/decrease of wastegate [1/s] *) (* OldName: rGRAD_WG; Cycle: 2 *)
		rGrad_ELR : REAL; (* gradient for increase at emergency-load-rejection of wastegate [1/s] *) (* OldName: rGRAD_ELR_WG; Cycle: 2 *)
		rGrad_Steady : REAL; (* gradient for steady increase/decrease of wastegate between the trigger levels [1/s] *) (* OldName: rGRAD_STEADY_WG; Cycle: 2 *)
		rGrad_Transient : REAL; (* gradient for fast decrease of wastegate at transient detection *)
		rPos_CBV_Hys : REAL; (* delta of position turbobypass valve for wastegate control *) (* OldName: rDPOS_TBPV_TRIG_WG; Cycle: 2 *)
		ti_Delay_ELR : TIME; (* turn on delay for TON of emergency load rejection [s] *) (* OldName: rTD_ELR_WG; Cycle: 2 *)
		ti_Check_Wait : TIME; (* waiting intervall between wastegate check [s] *) (* OldName: newPV; Cycle: 2 *)
		ti_Check_Open : TIME; (* open intervall while performing wastegate check [s] *) (* OldName: newPV; Cycle: 2 *)
		ti_Check_Close : TIME; (* close intervall while performing wastegate check [s] *) (* OldName: newPV; Cycle: 2 *)
		rPrDiff_WG_On : REAL; (* leanox deviation for WG transient activation *)
		rPrDiff_WG_Off : REAL; (* leanox deviation for WG transient deactivation *)
	END_STRUCT;
	tFilter : 	STRUCT
		bEna_IR_TC1 : BOOL; (* enables IR filter in task class 1 *)
		bEna_IR_TC2 : BOOL; (* enables IR filter in task class 2 *)
		bEna_PT1_TC1 : BOOL; (* enables PT1 filter in task class 1 *)
		iCycles_PT1_TC1 : UINT; (* filter cycles PT1 *)
		iBase_MAvg_TC2 : UINT; (* filter base moving average *)
		iNum_KnckFiltEngCyc : INT; (* Engine cycles for knock containment V2*) (* OldName: newPV; Cycle: 2;*)
		ti_CPP_Filt : TIME; (* Containment V3 Pmax *)
		tiSFIKW_OffDelay : TIME; (* Containment V3.1 Knock Knock *)
	END_STRUCT;
	tGen2 : 	STRUCT
		rLamOffsetLimInit : ARRAY[0..4]OF REAL; (*lambda offset compared to initial calibration at testcell*)
		rKeng_yInit_P : ARRAY[0..6]OF REAL; (*values of Ke depending on power*)
		rKeng_yInit : ARRAY[0..12]OF REAL; (*values of Ke depending on boost pressure*)
	END_STRUCT;
	tPUSL : 	STRUCT
		refPoint_Cyl_Limp_Max : ARRAY[0..1]OF lcrCurveByPoints_TabEntry_type; (* y = maximum number of cyl in limphome and x = pressure in [bar] *)
		tHC_Cyl : tHiCtrCyl_typ;
		tHC_Glob : tHiCtrGlob_typ;
		tCppInt : tCppIntPerm_typ; (* Permanent Data for Cylinder Peak Pressure Integrator *)
		refPoint_TupMFshape : ARRAY[0..10]OF lcrCurveByPoints_TabEntry_type;
		iNum_EngCyc_Limp_Warn : UINT; (*Warning threshold number of engine cycles, where a cylinder can be in LimpHome mode*)
		iNum_EngCyc_Limp_Max : UINT; (*Maximum number of engine cycles, where a cylinder can be in LimpHome mode*) (* Oldname: usLimpHomeEngCylLimit *)
		refPoint_P2s_MisfCycles : ARRAY[0..2]OF lcrCurveByPoints_TabEntry_type; (*Minimum cycles of cylinders misfireing *)
		refPoint_P2s_MisfMaxCyl : ARRAY[0..2]OF lcrCurveByPoints_TabEntry_type; (*Maximum number of cylinders misfireing *)
		iNum_MisfCycles2 : UINT; (* Minimum cycles of cylinders misfiring 2nd threshold *)
		iNum_MisfMaxCyl2 : UINT; (* Maximum number of cylinders misfiring 2nd threshold *)
	END_STRUCT;
	tPortInjection : 	STRUCT
		refPoint_ZVal : ARRAY[0..6]OF lcrCurveByPoints_TabEntry_type; (* y = ZValuePI and x = pressure in [bar] *) (* OldName: ssZWertStzPkt_BR9; Cycle: 2 *)
		refPoint_VE_N : ARRAY[0..6]OF lcrCurveByPoints_TabEntry_type; (* y = VE correction and x = revolutions in [rpm] *) (* OldName: LfgrdStzPkt; Cycle: 2 *)
		refPoint_VE_T : ARRAY[0..2]OF lcrCurveByPoints_TabEntry_type; (* y = VE correction and x = temperature in [deg.C] *) (* OldName: LfgrdStzPkt_t2s; Cycle: 2 *)
		refPoint_VE_Pr : ARRAY[0..5]OF lcrCurveByPoints_TabEntry_type; (* y = VE correction and x = pressure in [bar] *) (* OldName: LfgrdStzPkt_p2; Cycle: 2 *)
		rTi_Dur_Index : ARRAY[0..8]OF REAL;
		rPr_GR_P2s_Index : ARRAY[0..2]OF REAL;
		rDur_Corr : ARRAY[0..8,0..2]OF REAL; (* PI valve duration correction factors *)
		bSendDurWhenSkipping : BOOL; (* send PI duration during skipfire *)
		rDurGradLimitIsland : REAL; (* gradient limitation for PI openining duration in island operation *)
		rDurGradLimitNetP : REAL; (* gradient limitation for PI openining duration in grid operation *)
		LamCtrPBC : LamCtrPBC_PERM_Bus; (* Perms for lambda controller PBC *)
		iti_Lam_PBC : UINT; (* filter constant for lambda PBC *)
		rN_LamPBC_delay : REAL; (* delay of activating LamPBC calculation in rpm*)
	END_STRUCT;
	tFastStart : 	STRUCT
		bFS_Ena : BOOL; (* Enable Faststart *)
		bOnlyIdle : BOOL; (* Ignition point start offset enabled only in idle mode*)
		rT_ECW_Min : REAL; (* Engine Cooling Water temperature for fast start *)
		rT_EO_Min : REAL; (* Engine Oil temperature for fast start *)
		bRampVar_Ena : BOOL; (* Enable variable fast start ramp at power level threshold *)
		rP_Thrs_RampVar_Norm : REAL; (* load level at which variable fast start ramp is activated *)
		rP_Ramp_LL : REAL; (* variable fast start ramp lower limit *)
		rP_Ramp1_UL : REAL; (* variable fast start ramp 1 upper limit *)
		rP_Ramp2_UL : REAL; (* variable fast start ramp 2 upper limit *)
		rT_EO_Ramp : REAL; (* Engine oil temperature needed for highest ramp *)
		refPoint_Lam_N_Offs : ARRAY[0..2]OF lcrCurveByPoints_TabEntry_type;
		refPoint_IP_Pdev : ARRAY[0..1]OF lcrCurveByPoints_TabEntry_type;
		refPoint_IP_T3LP : ARRAY[0..1]OF lcrCurveByPoints_TabEntry_type;
		bEGTCtr_Ena : BOOL; (* Enable EGT Control over IP *)
		refPoint_IP_EGT : ARRAY[0..2]OF lcrCurveByPoints_TabEntry_type;
		rCA_IP_EGTCtr_LoLim : REAL; (* lower IP limit for EGTCtr *)
		EGTCtr : tEGTCtr_Perm; (* EGTCtr perm *)
		rCF_LamLim_Marg : REAL; (* low lambda limit margin factor *) (* OldName: rLamLimMargTexh; Cycle: 2 *)
		rN_CBV_Rel : REAL; (* Speed limit when CBV is closing during start up *)
		bGR_Scav_ena : BOOL; (* Gas rail scavenging enable *)
		bGR_Scav_H_Ext1 : BOOL; (* Gas rail scavenging 4 cylinder instead of 2 extended 1 *)
		bGR_Scav_H_Ext2 : BOOL; (* Gas rail scavenging 4 cylinder instead of 2 extended 2 *)
		rTi_GR_Scav : REAL; (* Gas rail scavenging duration [s]*)
		rTi_GR_Scav_Ext1 : REAL; (* Gas rail scavenging duration extended 1 [s]*)
		rTi_GR_Scav_Ext2 : REAL; (* Gas rail scavenging duration extended 2 [s]*)
		rCA_GR_Scav : REAL; (* Gas rail scavenging  PI opening duration [CA]*)
		rCA_GR_Scav_Ext1 : REAL; (* Gas rail scavenging  PI opening duration extended 1 [CA]*)
		rCA_GR_Scav_Ext2 : REAL; (* Gas rail scavenging  PI opening duration extended 2 [CA]*)
		iDT_GR_Scav_Th1 : UDINT; (* Time difference threshold for gas scavenging extended 1 [hours]*)
		iDT_GR_Scav_Th2 : UDINT; (* Time difference threshold for gas scavenging extended 2 [hours]*)
		rN_GR_Scav_max : REAL; (* Gas rail scavenging speed limit [rpm] *)
		rLamSlewRate : REAL; (* slew rate to ramp back to zero offset [1/s] *)
		rTi_idle : REAL; (* ramp back to zero offset after X sec in idle mode [s] *)
		rLamLoLim_N_x : ARRAY[0..2]OF REAL; (* Lower lambda limit lookup depending on engine speed [rpm] *)
		rLamLoLim_N_y : ARRAY[0..2]OF REAL; (* Lower lambda limit lookup depending on engine speed [-] *)
		rLam_Offs_Rej : REAL; (* lammbda offset for load rejections *)
		rLam_Offs_Acc : REAL; (* lammbda offset for load acceptance *)
	END_STRUCT;
	tSkip : 	STRUCT
		bExT_Ena : BOOL; (* Enables Exhaust temperature protection *)
		bExT_NetP_Ena : BOOL; (* Enables Exhaust temperature protection in NetP mode *)
		bExT_Island_Ena : BOOL; (* Enables Exhaust temperature protection in Island mode *)
		iNum_SkipCylExT_Max : USINT; (* maximum number of skipping cylinders for exhaust temp protection *)
		rT_ExH_Hys : REAL; (* exhaust temperature protection hysteresis *)
		rT_ExH_Start : REAL; (* exhaust temperature protection start delta *)
		iNum_SkipCyl_Cold : USINT;
		iNum_SkipCyl_Warm : USINT;
		rT_Cold : REAL;
		rT_Warm : REAL;
		ti_SkipRotation : TIME;
		bExT_II_Ena : BOOL;
		rT_EG_Deadband : REAL;
		rP_Disable_Norm : REAL; (* disable skipping above this power *)
		refPoint_SCRTCtr_SkipF_Lim : ARRAY[0..4]OF lcrCurveByPoints_TabEntry_type; (* skip limit for SCR inlet temperature controller over normed power *)
	END_STRUCT;
	tOptimizer : 	STRUCT
		iFilt_Pr : UINT; (* filter cycles for pressure signals *)
		bOptimizer_Ena : BOOL; (* enable optimizer *) (* OldName: bSW7; Cycle: 2 *)
		bTransient_Ena : BOOL; (* enable active transient balancing (State 3)*) (* OldName: bSW4; Cycle: 2 *)
		bState4_Ena : BOOL; (* enable PID1 steady state balancer *) (* OldName: bSW8; Cycle: 2 *)
		bP49_Source : BOOL; (* select P49 source, 0=Map, 1=Measurement *) (* OldName: bSW5; Cycle: 2 *)
		bP49_Median_Ena : BOOL; (* use P49 median as source: 0=aritmetic mean, 1=median *)
		bPmax_Median_Ena : BOOL; (* use Pmax median as setpoint: 0=aritmetic mean, 1=median *)
		rPmax_Offset_Coef_a : REAL; (* coefficient for the pmax offset calculation*)
		rPmax_Offset_Coef_b : REAL; (* coefficient for the pmax offset calculation*)
		rPr_P2s_PtP : REAL; (* P2s Peak to Peak  *) (* OldName: rPtP_P2s; Cycle: 2 *)
		rT_T2s_PtP : REAL; (* T2s Peak to Peak *) (* OldName: rPtP_T2s; Cycle: 2 *)
		rP_Pel_PtP : REAL; (* Pel Peak to Peak *) (* OldName: rPtP_Pel; Cycle: 2 *)
		rPr_P2s_Map : ARRAY[0..15]OF REAL; (* pressure quantization *) (* OldName: rPower_Index; Cycle: 2 *)
		rT_T2s_Map : ARRAY[0..10]OF REAL; (* temperatur quantization *) (* OldName: rCHTemp_Index; Cycle: 2 *)
		rPmaxOffset_UL : REAL; (* upper PMax Offset Limit from P49/MFB50 *)
		rPmaxOffset_LL : REAL; (* lower PMax Offset Limit from P49/MFB50 *)
		ti_P49_Filt_PID1 : TIME; (* filter time constant for P49 values *)
		ti_P49_Filt_PID2 : TIME; (* filter time constant for P49 values *)
		ti_Pmax_Filt_PID1 : TIME; (* filter time constant for Pmax values *)
		ti_Pmax_Filt_PID2 : TIME; (* filter time constant for Pmax values *)
		ti_IHR_Filt : TIME; (* filter time constant for IHR values *)
		rLim_PID1_Hi : REAL; (* upper PID1 Limit *)
		rLim_PID1_Lo : REAL; (* lower PID1 Limit *)
		rLim_PID1_Com_Hi : REAL; (* upper PID1 Limit during commisioning *)
		rLim_PID1_Com_Lo : REAL; (* lower PID1 Limit during commisioning *)
		rLim_PID2_Hi : REAL; (* upper PID2 Limit *)
		rLim_PID2_Lo : REAL; (* lower PID2 Limit *)
		rTnPart_PID1 : REAL; (* integrator time constant for PID1 *)
		rTnPart_PID2 : REAL; (* integrator time constant for PID2 *)
		refPoint_KpMap_PID1 : ARRAY[0..4]OF lcrCurveByPoints_TabEntry_type;
		refPoint_KpMap_PID2 : ARRAY[0..4]OF lcrCurveByPoints_TabEntry_type;
		refPoint_Crit_On : ARRAY[0..1]OF lcrCurveByPoints_TabEntry_type;
		refPoint_Crit_Off : ARRAY[0..1]OF lcrCurveByPoints_TabEntry_type;
		rDur_Lim_Hi : REAL; (* upper limit for optimizer *)
		rDur_Lim_Lo : REAL; (* lower limit for balancer *)
		bAdvKnck_En : BOOL; (* Enables Optimizer Offset from knock integrator *)
		refPoint_AdvKnck : ARRAY[0..1]OF lcrCurveByPoints_TabEntry_type;
		refPoint_Coef_c : ARRAY[0..2]OF lcrCurveByPoints_TabEntry_type;
		refPoint_Coef_d : ARRAY[0..2]OF lcrCurveByPoints_TabEntry_type;
		refPoint_Coef_e : ARRAY[0..2]OF lcrCurveByPoints_TabEntry_type;
		rPmax_Offset_Coef_d : REAL; (* coefficient for the pmax offset calculation due exhaust gas temperature deviation *)
		rPmax_Offset_Coef_e : REAL; (* coefficient for the pmax offset calculation due exhaust gas temperature limit *)
		bErrSumCorr_Ena : BOOL; (* enable sum correction for Optimizer Input *)
		rPmax_Offset_Coef_b_IP : REAL; (* coefficient for the pmax offset calculation*)
		rPmax_Offset_Coef_c : REAL; (* coefficient for the pmax offset calculation*)
		rPmax_Offset_d_PosLim : REAL; (* positiv limit for d offset *) (* OldName: rPmaxOffLimPosTexh; Cycle: 2 *)
		rPmax_Offset_d_NegLim : REAL; (* negative limit for d offset *) (* OldName: rPmaxOffLimNegTexh; Cycle: 2 *)
		rMisf_Int_Thrs : REAL; (* Misfire Integrator Treshold *) (* OldName: rMFIntThrTexh; Cycle: 2 *)
		rT_EG_LamMarg : REAL; (* exhaust gas temperature margin *) (* OldName: rTexhLamMarg; Cycle: 2 *)
		iFilt_IP : UINT; (* filter cycles for ignition point signals *)
		rKsum : REAL; (* sum correction gain *)
		iFilt_MFBvar : UINT; (* filter cycles for MFBvar signals *)
		rLim_PID2_Margin : REAL; (* Margin to PID2 limit when W2471 is triggered*)
		tiLim_PID2 : TIME; (* Time delay before W2471 is triggered *)
		tBaseMap : ARRAY[0..24,0..15]OF REAL;
		bLimpHome_minDur : BOOL; (* Limp home downset cylinder to minimum opening duration *)
		rDur_Off_CL_Crit_On : REAL; (* max PID output of cylinder criteria for automatic map save on *)
		rDur_Off_CL_Crit_Hy : REAL; (* max PID output of cylinder hysteresis for automatic map save  *)
		tiDelay_Opt_Req : TIME; (* time delay to request automatic balancing *)
		rFAR_dev_lim : REAL; (* deviation FAR limit to lock optimization *)
		bAut_Opt_Ena : BOOL; (* enable automatic optimization *)
		bAut_Opt_Act : BOOL; (* automatic optimization activated by HMI *)
	END_STRUCT;
	tHiCtrCyl_typ : 	STRUCT
		scMethodType : SINT;
		rGIGain : REAL; (*Gain for glow ignition acting on port injection [%*100cycles/events]*)
		rWCScaling : REAL; (*Scaling relative to Pmax at full load for weak combustion acting on Pmax stability layer offset in optimizer [%/bar]*)
		rGIPowGain : REAL; (*Gain for glow ignition acting on power reduction [%Pnom*100cycles/events]*)
		rMFGain : REAL; (*Gain for misfire acting on port injection [%*100cycles /events]*)
		rWCGain : REAL; (*Gain for weak combustion acting on Pmax stability layer offset in optimizer [bar*100cycles /events]*)
		rPmaxLimReaHys : REAL; (*Hysteresis for detection bit of Pmax limits reached [bar]*)
		rPmaxStdevFact : REAL; (*Factor for standard deviation for Pmax limiting control*)
		rGIThSkipReset : REAL; (*Reset threshold for glow ignition acting on skip-fire [events/100cycles]*)
		rMFThPIDUR : REAL; (*Threshold for misfire acting on port injection duration [events/100cycles]*)
		rMFThSkip : REAL; (*Threshold for misfire acting on skip fire [events/100cycles]*)
		rWCThPmax : REAL; (*Threshold for weak combustion acting on Pmax stability layer offset in optimizer [events/100cycles]*)
		rGIThPIDUR : REAL; (*Threshold for glow ignition acting on port injection [events/100cycles]*)
		rGIThSkip : REAL; (*Threshold for glow ignition acting on skip-fire [events/100cycles]*)
		rGIThCount : REAL; (*Threshold for number of task cycles showing glow ignition to activate power reduction [number of task cycles]*)
		ssTdownGI : INT; (*Time constant for emptying of glow ignition integrator [s]*)
		ssTupGI : INT; (*Time constant for filling of glow ignition integrator [s]*)
		ssTdownMF : INT; (*Time constant for emptying of misfire integrator [s]*)
		rPmaxContrLimMin : REAL; (*Minimum PIDUR offset set by Pmax limiting controller [%PIDUR]*)
		rMFPIDURLimMax : REAL; (*Maximum limit for misfire acting on port injection [%PIDURglobal]*)
		rWCPmaxLimMax : REAL; (*Maximum limit for weak combustion acting on Pmax stability layer offset in optimizer [%ofPmax]*)
		rGIPIDURLimMin : REAL; (*Minimum limit for glow ignition acting on port injection [%ofPIDURglobal]*)
		ssTupWC : INT; (*Time constant for filling of weak combustion integrator [s]*)
		ssTupMF : INT; (*Time constant for filling of misfire integrator [s]*)
		ssTdownWC : INT; (*Time constant for emptying of weak combustion integrator [s]*)
		rPmaxSDLimMar : REAL; (*Margin to Pmax shut down limit set in Diane [bar]*)
		rPmaxContrGain : REAL; (*Control gain of Pmax limiting controller [%PIDUR/bar]*)
		rMFThSkipOff : REAL;
		rMFGSkipTdown : REAL;
	END_STRUCT;
	tHiCtrGlob_typ : 	STRUCT
		scMethodType : SINT;
		rSkipToPowRedGain : REAL; (*Gain for skipped cylinders leading to power reduction [%Pnom/%skippedcylinder]*)
		rKPredPmaxLim : REAL; (*Gain for gobal power reduction depending on Pmax limitation [%Pnom/events*100cycles]*)
		rKITPmaxLim : REAL; (*Gain for global IT retardment depending on Pmax limitation [CAD/events*100cycles]*)
		ssNCylPmaxTh : INT; (*Threshold for number of cylinders being in Pmax limits before power reduction*)
		rPmaxLimPowTh : REAL; (*Threshold for Pmax limitation integrator before power reduction [events/100cycles]*)
		ssTdownPmax : INT; (*Integrator emptying time constant [s]*)
		ssTupPmax : INT; (*Integrator filling time constant for ignition retardment in case of Pmax limits reached*)
		rITPmaxLimMax : REAL; (*Max IT retardment in case of Pmax limitation [CAD]*)
		rPredPmaxLimMax : REAL; (*Max power reduction in case of Pmax limitation [% of Pnom]*)
		rSkipRefRedLimMax : REAL; (*Maximum value for power reference reduction due to skip fired cylinders [%Pnom]*)
		rMaxCylSkipBefPowRed : REAL; (*Maximum percentage of skipped cylinders before power reduction starts*)
		rMaxSkipDurBefRefRed : REAL; (*Maximum duration with skip-fired cylinders until power reduction [cycles]*)
		rSkipCountLimMax : REAL; (*Maximum value of skip counter [cycles], default = 1e5, must be always higher than MaxSkipDurBefRefRed*)
		rSkipRefRedLimMin : REAL; (*Minimum value for power reference reduction due to skip fired cylinders [%Pnom]*)
		rMaxSkipDurBefStop : REAL; (*Maximum duration for overall steady skip-fired operation and reduced ref power limit until engine shut down [s]*)
		rSkipOvCountLimMax : REAL; (*Maximum value of overall skip-fire counter*)
		rMaxCylSkipBefStop : REAL; (*Maximum percentage of skipped cylinders before engine shut down*)
	END_STRUCT;
	tLeanoxDrift : 	STRUCT
		iOpH_Leanox_Adjust : DINT; (*operational hours for leanox adjustment*)
		iOpH_CompChamb_Clean : DINT; (*operational hours for combustion chamber cleaning*)
	END_STRUCT;
	tCppIntPerm_typ : 	STRUCT  (* Struct - CppInt Permanent Data *)
		rInt_Dec : REAL; (* CPP Integrator Decent per Cycle Factor [%/Cycle] *)
		rInt_Power : REAL; (* CPP Integrator Weighting Function Power Factor *)
		rPI_Dur_IntLimLo : REAL; (* CPP Integrator Level Limit for Port Injection Duration reduction Low [%]*)
		rPI_Dur_IntLimHi : REAL; (* CPP Integrator Level Limit for Port Injection Duration reduction High [%] *)
		rIgn_IntLimLo : REAL; (* CPP Integrator Level Limit for Ignition Point Timing reduction Low [%] *)
		rIgn_IntLimHi : REAL; (* CPP Integrator Level Limit for Ignition Point Timing reduction High [%] *)
		tiInt_NonEmpty : TIME; (* CPP Integrator Nonempty Time until Shutdown [s] *)
		rNum_IntLimHi : REAL; (* CPP Integrator Level Limit for Multiple Cylinder [%] *)
		iCnt_IntLimHi : USINT; (* Count of CPP Integrator at Level above Limit [#] *)
		tiP_Red_delay : TIME; (* Power Reduction by CPP Integrator off delay [s] *)
		rP_Red_Ramp_Norm : REAL; (* Power Reduction by CPP Integrator ramp [%/100/s] *)
	END_STRUCT;
	tSparePerm_typ : 	STRUCT
		bit : ARRAY[0..9]OF tSpareBit_typ; (*Permanent saved spare variable*)
		single : ARRAY[0..9]OF tSpareSingle_typ; (*Permanent saved spare variable*)
		refPoint : ARRAY[0..5]OF tSpareMap_typ; (*Permanent saved spare variable*)
	END_STRUCT;
	tSpareBit_typ : 	STRUCT
		name : STRING[21];
		data : BOOL;
	END_STRUCT;
	tSpareSingle_typ : 	STRUCT
		name : STRING[21];
		data : REAL;
	END_STRUCT;
	tSpareMap_typ : 	STRUCT
		name : STRING[21];
		refPoint : ARRAY[0..4]OF lcrCurveByPoints_TabEntry_type;
	END_STRUCT;
	_tSAFImdatas : 	STRUCT
		data1 : UINT;
		data2 : UINT;
		data3 : UINT;
	END_STRUCT;
	_tSAFImdatasExtend : 	STRUCT
		data1 : UINT;
		data2 : UINT;
		data3 : UINT;
		data4 : USINT;
	END_STRUCT;
	_SAFIError : 	STRUCT
		Error : ARRAY[0..5]OF USINT;
	END_STRUCT;
	tMFB50 : 	STRUCT
		uMax : LREAL; (* upper control limit for IT offset in [CADbfTDC] *)
		uMin : LREAL; (* lower control limit for IT offset in [CADbfTDC] *)
		deadbandPos : LREAL; (* positive controller deadband in [CADafTDC] *)
		deadbandNeg : LREAL; (* negative controller deadband in [CADafTDC] *)
		MapPoP2sx : ARRAY[0..1]OF LREAL; (* p2s values for map in [mbar] *)
		MapPoP2sy : ARRAY[0..1]OF LREAL; (* proportional gain values for map in [CADbfTDC / CADafTDC] *)
		MapIoP2sx : ARRAY[0..1]OF LREAL; (* p2s values for map in [mbar] *)
		MapIoP2sy : ARRAY[0..1]OF LREAL; (* integral gain values for map in [CADbfTDC / s / CADafTDC] *)
		T1_PT1 : LREAL; (* First order time constant for PT1 filter in [s] *)
		init_PT1 : ARRAY[0..20]OF LREAL; (* Initial values for PT1 filter for each cylinder in [CADafTDC] *)
		MapMFB50oT3HPx : ARRAY[0..1]OF LREAL; (* T3HP values for map in [deg.C] *)
		MapMFB50oT3HPy : ARRAY[0..1]OF LREAL; (* MFB50 offset values for map in [CADafTDC] *)
		MapMFB50oP2sx : ARRAY[0..1]OF LREAL; (* p2s values for map in [mbar] *)
		MapMFB50oP2sy : ARRAY[0..1]OF LREAL; (* MFB50 offset values for map in [CADafTDC] *)
		MFB50EnSpdTh : LREAL; (* speed threshold for MFB50 control release in [rpm] *)
		MFB50ContrEn : BOOL; (* activate MFB50 control if = 1 [boolean], if 0, main control code will not be executed (case loop) *)
		MFB50RefOffsetAllCyl : ARRAY[0..20]OF LREAL; (* External offset on reference MFB50 for each cylinder in [CADafTDC] *)
		MFB50MedianEn : BOOL; (* Switch to decide between different MFB50 references [boolean], 0 = global reference, 1 = median *)
		MFB50GlobRefExt : LREAL; (* Global REFERENCE for MFB50 in [CADafTDC] *)
		LoadEnabled : BOOL; (*If 1, MFB50 control is enabled above load threshold*)
		MFB50EnPowTh : LREAL; (*Load threshold for MFB50 control release in [% of  nom load]*)
		bAdvKnck_En : BOOL; (* Enables MFB50 Offset from knock integrator *)
	END_STRUCT;
	tStat_VAR_LR : 	STRUCT
		rP_Act_LR_Base_Norm : REAL; (*base load before opening the GCB*)
		rPr_Eng_P2s_Base : REAL;
		rN_max : REAL; (* negative gradient of engine speed *)
		day : UINT;
		month : UINT;
		year : UINT;
		hour : UINT;
		minute : UINT;
	END_STRUCT;
	tStat_VAR : 	STRUCT
		rN_Grad_RunOut : REAL; (* negative gradient of engine speed *)
		day : UINT;
		month : UINT;
		year : UINT;
		hour : UINT;
		minute : UINT;
	END_STRUCT;
	tBank_AB : 	STRUCT
		Avg : REAL; (* Bank (A+B)/2 *)
		A : REAL; (* Bank A *)
		B : REAL; (* Bank A *)
	END_STRUCT;
	tSync_Perm : 	STRUCT
		bSpeedSet_ena : BOOL; (*Select the setpoint (1: constant speed, 0: grid frequency)*)
		iCtrSel : SINT; (*Control selection. 1-Std skip firing. 2-Time optimal 3-Time optimal with constraints. 4-Fuel and time optimal. 5-Modified skip f*)
		rN_SetTol : REAL; (*Speed band for speed regulation (rpm, valid only for standard approach)*)
		iSkipCounterLimit : UINT; (*Dwell time for skip firing (in number of 10ms, valid only for the standard approach)*)
		rAngleSetDeg : REAL; (*Electric angle setpoint (in deg, tuning parameter)*)
		rRelaxAngleDeg : REAL; (*Relaxation band for the electric angle setpoint (in deg, tuning parameter)*)
		rWeightFuel : REAL; (*Weighting (high->time, low->fuel)*)
		rHystOptimal : REAL; (*Band around switching surface (nonnegative >=0)*)
		iNum_SkipMax : USINT; (*Maximum cylinders skipped (<=20)*)
		iNum_SkipMin : USINT; (*Minimum number of cylinders (>0)*)
		rTi_FiltF : REAL; (*Filter constant for grid frequency [s]*)
		rN_enableNorm : REAL; (*Engine speed normalized to enable fast sync controller [-]*)
		rN_idleNorm : REAL; (*Engine speed normalized to enable fast sync controller [-]*)
		rTi_FastSync : REAL; (*switch over to standard controller after this time [s]*)
		bF_act_ena : BOOL; (*use generator frequency as actual value*)
		rT_Cold : REAL;
		rT_Warm : REAL;
		iNum_SkipCyl_Cold : USINT;
		iNum_SkipCyl_Warm : USINT;
		rGain_P : REAL; (*Gain for P-part [NumSkippedCyl/rpm]*)
		iNum_SkipCylLim_P : SINT; (*Limit for P-part [NumSkippedCyl]*)
		bStdCtrl : BOOL; (*Standard controller enabled in AutoCode*)
	END_STRUCT;
```
